(* IEC 61131-3 sources: Explicit_MPC_on_PLC/Quad-Tank/MATLAB_Files/Used Files/plcsrc, 1 file *)

(* ---- sim_mixed.st ---- *)
(*
 *
 * File: sim_mixed.st
 *
 * IEC 61131-3 Structured Text (ST) code generated for subsystem "sim_mixed/Explicit Controller"
 *
 * Model name                      : sim_mixed
 * Model version                   : 1.163
 * Model creator                   : andrewralea
 * Model last modified by          : andrewralea
 * Model last modified on          : Mon May 24 20:24:12 2021
 * Model sample time               : 0s
 * Subsystem name                  : sim_mixed/Explicit Controller
 * Subsystem sample time           : 0.01s
 * Simulink PLC Coder version      : 3.3 (R2020b) 29-Jul-2020
 * ST code generated on            : Fri May 28 16:37:33 2021
 *
 * Target IDE selection            : Beckhoff TwinCAT 3
 * Test Bench included             : No
 *
 *)
FUNCTION_BLOCK Explicit
VAR_INPUT
    ssMethodType: SINT;
    MeasuredTankOutputs: ARRAY [0..1] OF LREAL;
    ref: ARRAY [0..1] OF LREAL;
END_VAR
VAR_OUTPUT
    mv: ARRAY [0..1] OF LREAL;
END_VAR
VAR
    last_x_PreviousInput: ARRAY [0..5] OF LREAL;
    last_mv_DSTATE: ARRAY [0..1] OF LREAL;
    Explicit_b_M: ARRAY [0..11] OF LREAL := 3.14192233852028E-7,2.5115282232541673E-8,5.9723043350726878E-8,
        2.2534269604652875E-7,0.0099501247588661811,3.3026396230579933E-9,6.8756742676357756E-8,
        3.2698899289917904E-7,2.2408008895209797E-7,6.5568434535270065E-8,-3.3744504064209632E-9,
        0.0099501247490762831;
    Explicit_b_Cm: ARRAY [0..11] OF LREAL := 0.15299877600979192,0.0,0.0,0.15299877600979192,0.0,0.0,0.0,0.0,1.0,
        0.0,0.0,1.0;
    Explicit_b_thmin: ARRAY [0..9] OF LREAL := -12.5,-17.5,-3.260954352640991,-0.9466686383552787,-1.25,-1.25,-12.5,
        -17.5,-31.242868949193834,-63.580836957418676;
    Explicit_b_thmax: ARRAY [0..9] OF LREAL := 30.0,25.0,39.239045647359006,41.553331361644723,1.25,1.25,25.0,20.0,
        169.936,169.936;
    b_i1: ARRAY [0..100] OF INT := 1,25,48,71,91,114,137,158,178,199,221,242,262,283,304,324,343,364,383,403,423,
        445,467,485,506,517,537,556,577,597,616,638,656,668,689,708,727,747,767,786,807,827,847,867,886,908,927,947,
        967,989,1008,1019,1039,1055,1076,1098,1117,1136,1155,1171,1189,1211,1230,1246,1265,1284,1299,1318,1339,1357,
        1376,1396,1415,1435,1456,1476,1497,1517,1537,1556,1575,1595,1613,1633,1653,1671,1692,1711,1731,1747,1765,
        1784,1804,1823,1843,1862,1882,1902,1921,1940,1959;
    b_i2: ARRAY [0..100] OF INT := 24,47,70,90,113,136,157,177,198,220,241,261,282,303,323,342,363,382,402,422,444,
        466,484,505,516,536,555,576,596,615,637,655,667,688,707,726,746,766,785,806,826,846,866,885,907,926,946,966,
        988,1007,1018,1038,1054,1075,1097,1116,1135,1154,1170,1188,1210,1229,1245,1264,1283,1298,1317,1338,1356,
        1375,1395,1414,1434,1455,1475,1496,1516,1536,1555,1574,1594,1612,1632,1652,1670,1691,1710,1730,1746,1764,
        1783,1803,1822,1842,1861,1881,1901,1920,1939,1958,1978;
    Explicit_b_L: ARRAY [0..11] OF LREAL := 3.1403362819378811E-7,2.5755371121733541E-8,5.9629108064733625E-8,
        2.246853239956293E-7,0.0099501247588661551,3.3026395811602204E-9,6.9053788137012E-8,3.2695809528341482E-7,
        2.2372764502189584E-7,6.5377157634733646E-8,-3.3744504046873746E-9,0.0099501247490763074;
    Explicit_b_Bu: ARRAY [0..11] OF LREAL := 0.00020814878862012381,1.7089200517136452E-7,0.0,
        0.00011695983573308414,0.0,0.0,9.2113938270845919E-8,0.0002081617439639849,0.00011703862782711392,0.0,0.0,
        0.0;
    Explicit_b_A: ARRAY [0..35] OF LREAL := 0.9991963417969173,0.0,0.0,0.0,0.0,0.0,0.0,0.99932074257543357,0.0,0.0,
        0.0,0.0,0.0015722160273812986,0.0,0.99842715170590557,0.0,0.0,0.0,0.0,0.0029162188726435975,0.0,
        0.99708278976438092,0.0,0.0,0.0,0.0,0.0,0.0,1.0,0.0,0.0,0.0,0.0,0.0,0.0,1.0;
    Explicit_c_K: ARRAY [0..1977] OF LREAL := 150.27277651970425,150.27276024869144,150.1745002542759,
        150.17446124607031,0.0,0.0,0.0,0.0,30.0,25.0,39.239045647359006,41.553331361644723,1.25,1.25,25.0,20.0,12.5,
        17.5,3.260954352640991,0.9466686383552787,1.25,1.25,12.5,17.5,-150.27277651970428,150.27276094028818,
        0.00896851306694222,0.0092486718565456469,150.17446243836258,-6.9159822683988875E-7,-1.1922963395590097E-6,
        30.0,25.0,39.239045647359006,41.553331361644723,1.25,1.25,20.0,169.936,12.5,17.5,3.260954352640991,
        0.9466686383552787,1.25,1.25,12.5,17.5,-150.27276024869144,150.27277721130108,0.0089700423139607143,
        150.17450136627906,0.0092502663373971762,-6.915983020343374E-7,-1.1120067688561992E-6,30.0,25.0,
        39.239045647359006,41.553331361644723,1.25,1.25,25.0,169.936,12.5,17.5,3.260954352640991,0.9466686383552787,
        1.25,1.25,12.5,17.5,-150.1745002542759,150.30349143296371,150.27276061960174,150.25280880838065,
        -6.4025688321438744E-7,30.0,25.0,39.239045647359006,41.553331361644723,1.25,1.25,25.0,12.5,17.5,
        3.260954352640991,0.9466686383552787,1.25,1.25,17.5,63.580836957418676,0.0,150.27276024868996,
        150.17446124606624,0.0,0.0,0.0,0.0,30.0,25.0,39.239045647359006,41.553331361644723,1.25,1.25,25.0,20.0,12.5,
        17.5,3.260954352640991,0.9466686383552787,1.25,1.25,17.5,31.242868949193834,0.0,150.2727765197028,
        150.17450025427226,0.0,0.0,0.0,0.0,30.0,25.0,39.239045647359006,41.553331361644723,1.25,1.25,25.0,20.0,12.5,
        17.5,3.260954352640991,0.9466686383552787,1.25,1.25,12.5,63.580836957418676,0.0,150.27276024869022,
        150.174461246067,0.0,0.0,0.0,30.0,25.0,39.239045647359006,41.553331361644723,1.25,1.25,20.0,12.5,17.5,
        3.260954352640991,0.9466686383552787,1.25,1.25,12.5,17.5,0.0,150.27277651970292,0.0,0.0,0.0,30.0,25.0,
        39.239045647359006,41.553331361644723,1.25,1.25,25.0,12.5,17.5,3.260954352640991,0.9466686383552787,1.25,
        1.25,12.5,17.5,-150.2727772113011,-150.27276094028815,0.00899229717151725,0.0089972026991569677,
        0.0092719269187978466,30.0,25.0,39.239045647359006,41.553331361644723,1.25,1.25,169.936,169.936,12.5,17.5,
        3.260954352640991,0.9466686383552787,1.25,1.25,12.5,17.5,-0.0092486718537731459,-150.3142337225209,
        150.27276094028818,150.17446243836227,-6.91598518490273E-7,-1.1922968442958055E-6,30.0,25.0,
        39.239045647359006,41.553331361644723,1.25,1.25,25.0,20.0,169.936,12.5,17.5,3.260954352640991,
        0.9466686383552787,1.25,1.25,17.5,-150.2727765197028,12.5,-150.31423372345185,6.915984886602121E-7,
        0.010088924529484842,-2.7160393645102115E-5,30.0,25.0,39.239045647359006,41.553331361644723,1.25,1.25,20.0,
        169.936,12.5,17.5,3.260954352640991,0.9466686383552787,1.25,1.25,63.580836957418676,-150.27277651970294,
        1.192296339559001E-6,0.0089685130647667952,0.0092486718548978036,-7.9526503793109085E-7,30.0,25.0,
        39.239045647359006,41.553331361644723,1.25,1.25,169.936,12.5,17.5,3.260954352640991,0.9466686383552787,1.25,
        1.25,12.5,17.5,-150.31422855929941,-0.0089700423151911571,150.27277721130105,150.17450136627863,
        0.010090749420623041,-6.91598601136511E-7,-1.1120072501316056E-6,30.0,25.0,39.239045647359006,
        41.553331361644723,1.25,1.25,25.0,169.936,12.5,17.5,3.260954352640991,1.25,1.25,12.5,-150.27276024868993,
        -2.3784105123531843E-5,17.5,-150.314228558367,6.9159864144958721E-7,30.0,25.0,39.239045647359006,
        41.553331361644723,1.25,1.25,25.0,20.0,169.936,12.5,17.5,3.260954352640991,0.9466686383552787,1.25,1.25,
        31.242868949193834,-150.27276024869022,1.112006768856199E-6,0.0089700423159589249,0.0092502663388704057,
        -8.1826648506024674E-7,30.0,25.0,39.239045647359006,41.553331361644723,1.25,1.25,169.936,12.5,17.5,
        3.260954352640991,0.9466686383552787,1.25,1.25,12.5,17.5,-0.0084253602440059385,-0.0084317458919612974,
        150.31423400479244,150.31422879473305,30.0,25.0,39.239045647359006,41.553331361644723,1.25,1.25,25.0,20.0,
        17.5,3.260954352640991,0.9466686383552787,1.25,1.25,31.242868949193834,63.580836957418676,0.0,0.0,0.0,0.0,
        0.0,30.0,25.0,39.239045647359006,41.553331361644723,1.25,1.25,25.0,20.0,12.5,17.5,3.260954352640991,
        0.9466686383552787,1.25,1.25,31.242868949193834,63.580836957418676,0.0,0.0,150.27276024868965,0.0,30.0,25.0,
        39.239045647359006,41.553331361644723,1.25,1.25,12.5,17.5,3.260954352640991,0.9466686383552787,1.25,1.25,
        17.5,31.242868949193834,63.580836957418676,0.0,0.0,0.0,0.0,0.0,30.0,25.0,39.239045647359006,
        41.553331361644723,1.25,1.25,25.0,12.5,17.5,3.260954352640991,0.9466686383552787,1.25,1.25,17.5,
        31.242868949193834,0.0,17.5,0.0,0.0,0.0,30.0,25.0,39.239045647359006,41.553331361644723,1.25,1.25,20.0,12.5,
        17.5,3.260954352640991,0.9466686383552787,1.25,1.25,12.5,63.580836957418676,0.0,150.27277651970246,
        150.17450025427149,0.0,0.0,0.0,30.0,25.0,39.239045647359006,41.553331361644723,1.25,1.25,25.0,20.0,12.5,
        17.5,3.260954352640991,0.9466686383552787,1.25,1.25,12.5,63.580836957418676,0.0,150.27276024868988,
        150.17446124606604,0.0,0.0,0.0,30.0,25.0,39.239045647359006,41.553331361644723,1.25,1.25,20.0,169.936,12.5,
        17.5,3.260954352640991,0.9466686383552787,1.25,1.25,12.5,17.5,0.0,0.0,0.0,0.0,30.0,25.0,39.239045647359006,
        41.553331361644723,1.25,1.25,12.5,17.5,3.260954352640991,0.9466686383552787,1.25,1.25,12.5,17.5,0.0,
        150.2727765197026,150.17450025427178,0.0,0.0,0.0,30.0,25.0,39.239045647359006,41.553331361644723,1.25,1.25,
        25.0,12.5,17.5,3.260954352640991,0.9466686383552787,1.25,1.25,12.5,17.5,-150.31423409213582,
        -150.27276094028815,-0.0089922971720828356,0.0089972027095938083,0.0101105928744509,30.0,25.0,
        39.239045647359006,41.553331361644723,1.25,1.25,-0.008997202709492582,-150.27277721130102,
        -150.31422888114486,0.0089922971840448781,30.0,25.0,39.239045647359006,41.553331361644723,1.25,1.25,20.0,
        169.936,169.936,12.5,17.5,3.260954352640991,0.9466686383552787,1.25,1.25,12.5,-0.0092486718560890989,
        -150.3142337225205,1.1922968442958055E-6,-7.9526537103502364E-7,30.0,25.0,39.239045647359006,
        41.553331361644723,1.25,1.25,25.0,169.936,12.5,17.5,3.260954352640991,0.9466686383552787,1.25,1.25,17.5,
        -150.27277651970238,3.2277787241348325E-7,2.6103247877849398E-5,0.0089685130647338546,0.00924867185486637,
        30.0,25.0,39.239045647359006,41.553331361644723,1.25,1.25,169.936,12.5,17.5,3.260954352640991,
        0.9466686383552787,1.25,1.25,12.5,17.5,63.580836957418676,-150.2727765197026,7.9526503793110049E-7,
        0.0089685130647458953,0.0092486718548779323,-3.2277787241348331E-7,30.0,25.0,39.239045647359006,
        41.553331361644723,1.25,1.25,169.936,12.5,17.5,3.260954352640991,0.9466686383552787,1.25,1.25,12.5,17.5,
        -150.20363326125491,150.27277704995686,150.31422855929944,150.17450110707583,0.0084101003282759639,
        -5.3025423494204181E-7,-8.5280395478764181E-7,30.0,25.0,39.239045647359006,41.553331361644723,1.25,1.25,
        25.0,1.25,1.25,12.5,17.5,31.242868949193834,-150.3142285583674,-4.5713461310450266E-7,150.272777211301,
        150.17450136627863,-6.9159864144958721E-7,-1.1120073155610654E-6,30.0,25.0,39.239045647359006,
        41.553331361644723,1.25,1.25,25.0,20.0,169.936,12.5,17.5,3.260954352640991,0.9466686383552787,1.25,1.25,
        12.5,-150.3142285592991,-0.0089700423152055762,1.1120072501316007E-6,0.010090749420522883,
        -8.182668401829975E-7,30.0,25.0,39.239045647359006,41.553331361644723,1.25,1.25,169.936,12.5,17.5,
        3.260954352640991,1.25,1.25,12.5,-150.27276024868971,4.8112884150133535E-7,2.3255062955056014E-5,
        0.0089700423159182838,-2.4842396974108378E-5,25.0,39.239045647359006,41.553331361644723,1.25,1.25,17.5,
        31.242868949193834,-150.27276024868988,2.1668353413129541E-5,0.0089700423138394814,0.00925026633727334,
        -3.6868395525815943E-7,30.0,25.0,39.239045647359006,41.553331361644723,1.25,1.25,169.936,169.936,12.5,17.5,
        3.260954352640991,0.9466686383552787,1.25,1.25,12.5,17.5,-150.20366731447805,-0.0084317458833884553,
        150.31423400572388,150.31422879473305,0.0084253602346650771,30.0,25.0,39.239045647359006,41.553331361644723,
        1.25,1.25,20.0,12.5,17.5,3.260954352640991,0.9466686383552787,1.25,1.25,63.580836957418676,
        -150.20363403920774,-0.0084253602429266682,150.31423400479244,150.31422879566506,0.0084317458959346555,30.0,
        25.0,39.239045647359006,41.553331361644723,1.25,1.25,25.0,12.5,17.5,3.260954352640991,0.9466686383552787,
        1.25,1.25,31.242868949193834,-150.31423400479247,-4.57772250744983E-7,-3.8232338890894953E-7,
        150.31422888114494,30.0,25.0,39.239045647359006,41.553331361644723,1.25,1.25,25.0,20.0,169.936,17.5,
        3.260954352640991,0.9466686383552787,1.25,1.25,31.242868949193834,63.580836957418676,0.0,0.0,0.0,0.0,0.0,
        30.0,25.0,39.239045647359006,41.553331361644723,1.25,1.25,20.0,12.5,17.5,3.260954352640991,
        0.9466686383552787,1.25,1.25,31.242868949193834,63.580836957418676,0.0,0.0,0.0,0.0,0.0,30.0,25.0,
        39.239045647359006,41.553331361644723,1.25,1.25,25.0,12.5,17.5,3.260954352640991,1.25,1.25,
        31.242868949193834,63.580836957418676,0.0,150.27276024868991,0.0,0.0,0.0,30.0,25.0,39.239045647359006,
        41.553331361644723,1.25,1.25,25.0,20.0,12.5,17.5,3.260954352640991,0.9466686383552787,1.25,1.25,17.5,
        31.242868949193834,0.0,17.5,0.0,0.0,30.0,25.0,39.239045647359006,41.553331361644723,1.25,1.25,20.0,12.5,
        17.5,3.260954352640991,0.9466686383552787,1.25,1.25,12.5,31.242868949193834,63.580836957418676,0.0,0.0,0.0,
        0.0,0.0,30.0,25.0,39.239045647359006,41.553331361644723,1.25,1.25,25.0,12.5,17.5,3.260954352640991,
        0.9466686383552787,1.25,1.25,17.5,31.242868949193834,0.0,0.0,0.0,0.0,0.0,30.0,25.0,39.239045647359006,
        41.553331361644723,1.25,1.25,25.0,12.5,17.5,3.260954352640991,0.9466686383552787,1.25,1.25,17.5,
        31.242868949193834,0.0,0.0,0.0,0.0,30.0,25.0,39.239045647359006,41.553331361644723,1.25,1.25,169.936,12.5,
        17.5,3.260954352640991,0.9466686383552787,1.25,1.25,12.5,17.5,0.0,0.0,150.27277651970238,150.17450025427129,
        0.0,0.0,30.0,25.0,39.239045647359006,41.553331361644723,1.25,1.25,25.0,12.5,17.5,3.260954352640991,
        0.9466686383552787,1.25,1.25,12.5,17.5,63.580836957418676,0.0,0.0,0.0,0.0,30.0,25.0,39.239045647359006,
        41.553331361644723,1.25,1.25,20.0,12.5,17.5,3.260954352640991,0.9466686383552787,1.25,1.25,12.5,
        63.580836957418676,0.0,0.0,0.0,0.0,30.0,25.0,39.239045647359006,41.553331361644723,1.25,1.25,169.936,12.5,
        17.5,3.260954352640991,0.9466686383552787,1.25,1.25,12.5,17.5,63.580836957418676,0.0,0.0,0.0,0.0,30.0,25.0,
        39.239045647359006,41.553331361644723,1.25,1.25,20.0,169.936,12.5,17.5,3.260954352640991,0.9466686383552787,
        1.25,1.25,12.5,63.580836957418676,0.0,0.0,150.27276024868965,150.17446124606542,0.0,0.0,30.0,25.0,
        39.239045647359006,41.553331361644723,1.25,1.25,20.0,12.5,17.5,3.260954352640991,0.9466686383552787,1.25,
        1.25,12.5,17.5,31.242868949193834,-150.17450025427178,4.253152391505125E-7,150.30349143296283,
        150.25280880837818,-1.7296307093690735E-7,30.0,25.0,39.239045647359006,41.553331361644723,1.25,1.25,25.0,
        12.5,17.5,3.260954352640991,0.9466686383552787,1.25,1.25,17.5,-150.27276075599735,-150.20366755066993,
        150.31423409213579,0.0089899947598349236,0.00843045541435082,30.0,25.0,39.239045647359006,
        41.553331361644723,1.25,1.25,-150.27276094028815,17.5,-150.31423409120444,-150.31422888114497,30.0,25.0,
        39.239045647359006,41.553331361644723,1.25,1.25,25.0,20.0,169.936,169.936,17.5,3.260954352640991,
        0.9466686383552787,1.25,1.25,31.242868949193834,-150.27277704995686,-150.20363432127169,150.31422888207695,
        0.00898677805621705,0.0084393742662072935,30.0,25.0,39.239045647359006,41.553331361644723,1.25,1.25,169.936,
        1.25,1.25,12.5,17.5,-150.25280880838059,150.31423372252087,150.27276075599735,150.17446212183043,
        -5.0730746847704375E-7,-8.7576436608860627E-7,30.0,25.0,39.239045647359006,41.553331361644723,1.25,1.25,
        25.0,20.0,12.5,17.5,3.260954352640991,0.9466686383552787,1.25,1.25,17.5,-150.31423372252044,
        -4.57021496831135E-7,6.91598518490273E-7,-2.7160394808446411E-5,-2.7688874260814198E-5,30.0,25.0,
        39.239045647359006,41.553331361644723,1.25,1.25,25.0,20.0,169.936,17.5,3.260954352640991,0.9466686383552787,
        1.25,1.25,17.5,31.242868949193834,63.580836957418676,-150.1745002542726,6.4025688321438437E-7,
        150.303491432963,150.25280880837869,-4.2531523915050832E-7,30.0,25.0,39.239045647359006,41.553331361644723,
        1.25,1.25,25.0,12.5,17.5,3.260954352640991,0.9466686383552787,1.25,1.25,17.5,-150.30349143296283,
        -0.0092486718560926464,7.9526530580585218E-7,0.0084080843735949169,-3.2277798170283768E-7,30.0,25.0,
        39.239045647359006,41.553331361644723,1.25,1.25,169.936,12.5,17.5,3.260954352640991,0.9466686383552787,1.25,
        1.25,17.5,-150.20366653652189,5.0730744361467508E-7,150.31423372345185,0.00840878705982342,
        -1.9952445451383883E-5,30.0,25.0,39.239045647359006,41.553331361644723,1.25,1.25,20.0,12.5,17.5,
        3.260954352640991,0.9466686383552787,1.25,1.25,63.580836957418676,-150.27277651970246,4.4094945298300684E-7,
        2.7688862477194338E-5,0.0089685130647387656,-2.6103247877849368E-5,30.0,25.0,39.239045647359006,
        41.553331361644723,1.25,1.25,1.25,1.25,12.5,17.5,63.580836957418676,-150.3142337225203,
        3.2277800799099981E-7,30.0,25.0,39.239045647359006,41.553331361644723,1.25,1.25,25.0,169.936,12.5,17.5,
        3.260954352640991,0.9466686383552787,1.25,1.25,17.5,63.580836957418676,-0.0084101003242163189,
        150.27277704995686,150.31422855836743,150.17450110707577,-5.3025426854081661E-7,-8.528040093195823E-7,30.0,
        25.0,39.239045647359006,41.553331361644723,1.25,1.25,25.0,20.0,12.5,17.5,3.260954352640991,
        0.9466686383552787,1.25,1.25,12.5,63.580836957418676,-150.20363326125155,5.302542349420417E-7,
        150.31422855929904,0.0084101003218975314,-1.78419540761567E-5,30.0,25.0,39.239045647359006,
        41.553331361644723,1.25,1.25,25.0,12.5,17.5,3.260954352640991,0.9466686383552787,1.25,1.25,
        31.242868949193834,-150.2036332612509,2.8227211141446421E-7,1.9111227183265134E-5,150.31422855929898,
        0.0084101003281506683,30.0,25.0,39.239045647359006,41.553331361644723,1.25,1.25,1.25,1.25,12.5,17.5,
        31.242868949193834,-150.31422855836709,-4.5713461315188076E-7,3.7104855832596717E-9,-8.1826688808031187E-7,
        30.0,25.0,39.239045647359006,41.553331361644723,1.25,1.25,20.0,169.936,12.5,17.5,3.260954352640991,
        0.9466686383552787,1.25,1.25,12.5,-150.31422855929895,-0.0089700423152052188,4.81129049402035E-7,
        2.3255073031969076E-5,0.010090749420478901,-2.4842407822217915E-5,25.0,39.239045647359006,
        41.553331361644723,1.25,1.25,169.936,12.5,17.5,3.260954352640991,0.9466686383552787,1.25,1.25,
        31.242868949193834,-150.20363326125218,8.5280395478765081E-7,150.31422855929912,0.008410100321918695,
        -6.2813598573044263E-7,30.0,25.0,39.239045647359006,41.553331361644723,1.25,1.25,1.25,1.25,12.5,17.5,
        -150.31422855929904,-0.0089700423159724645,2.1668362719146114E-5,0.010090749414219103,
        -3.6868411405625081E-7,30.0,25.0,39.239045647359006,41.553331361644723,1.25,1.25,169.936,169.936,12.5,17.5,
        3.260954352640991,1.25,1.25,12.5,-150.27276024868965,3.6868395525815943E-7,2.2497959692190342E-9,
        0.008970042313820821,0.00925026633725427,30.0,25.0,39.239045647359006,41.553331361644723,1.25,1.25,169.936,
        12.5,17.5,3.260954352640991,0.9466686383552787,1.25,1.25,12.5,17.5,31.242868949193834,-150.20366731447808,
        -150.20363403920777,150.31423400572388,150.31422879566503,0.0084253602409406526,0.0084317458833884553,30.0,
        25.0,39.239045647359006,41.553331361644723,1.25,1.25,12.5,17.5,3.260954352640991,0.9466686383552787,1.25,
        1.25,-150.314228794733,-150.20366755066965,-0.01011239497184554,150.31423409213585,0.008430455426884231,
        30.0,25.0,39.239045647359006,41.553331361644723,1.25,1.25,20.0,169.936,12.5,17.5,3.260954352640991,
        0.9466686383552787,1.25,1.25,-0.0084087870624481986,5.0730746847704364E-7,150.31423372252041,
        -1.9952446420993245E-5,-2.0375796427188149E-5,30.0,25.0,39.239045647359006,41.553331361644723,1.25,1.25,
        25.0,20.0,17.5,3.260954352640991,0.9466686383552787,1.25,1.25,31.242868949193834,63.580836957418676,
        -150.3142340047925,-150.20363432127149,-0.010105497708264473,150.31422888207695,0.008439374278734136,30.0,
        25.0,39.239045647359006,41.553331361644723,1.25,1.25,25.0,169.936,17.5,3.260954352640991,0.9466686383552787,
        1.25,1.25,31.242868949193834,-0.0084101003242149728,5.3025426854081651E-7,150.31422855836706,
        -1.7841955234048227E-5,30.0,25.0,39.239045647359006,41.553331361644723,1.25,1.25,25.0,20.0,12.5,17.5,
        3.260954352640991,0.9466686383552787,1.25,1.25,31.242868949193834,63.580836957418676,-150.31423400572393,
        0.010105497701810977,-150.27277704995686,-0.0084393742662072935,150.31422888114494,30.0,25.0,
        39.239045647359006,41.553331361644723,1.25,1.25,20.0,169.936,12.5,17.5,3.260954352640991,0.9466686383552787,
        1.25,1.25,12.5,63.580836957418676,4.8112907714119855E-7,25.0,-150.31422855836695,3.6868413507214106E-7,30.0,
        25.0,39.239045647359006,41.553331361644723,1.25,1.25,20.0,169.936,12.5,17.5,3.260954352640991,
        0.9466686383552787,1.25,1.25,12.5,31.242868949193834,0.0,0.0,0.0,0.0,0.0,30.0,25.0,39.239045647359006,
        41.553331361644723,1.25,1.25,25.0,12.5,17.5,3.260954352640991,0.9466686383552787,1.25,1.25,17.5,
        31.242868949193834,63.580836957418676,0.0,0.0,0.0,0.0,30.0,25.0,39.239045647359006,41.553331361644723,1.25,
        1.25,169.936,12.5,17.5,3.260954352640991,0.9466686383552787,1.25,1.25,12.5,17.5,31.242868949193834,0.0,0.0,
        0.0,0.0,0.0,30.0,25.0,39.239045647359006,41.553331361644723,1.25,1.25,25.0,12.5,17.5,3.260954352640991,
        0.9466686383552787,1.25,1.25,31.242868949193834,63.580836957418676,0.0,0.0,0.0,30.0,25.0,39.239045647359006,
        41.553331361644723,1.25,1.25,25.0,12.5,17.5,3.260954352640991,0.9466686383552787,1.25,1.25,12.5,17.5,
        31.242868949193834,-0.50109411185443054,1.7296307093690733E-7,150.30349143296272,150.25280880837795,30.0,
        25.0,39.239045647359006,41.553331361644723,1.25,1.25,25.0,12.5,17.5,3.260954352640991,0.9466686383552787,
        1.25,1.25,17.5,63.580836957418676,0.0,0.0,0.0,0.0,30.0,25.0,39.239045647359006,41.553331361644723,1.25,1.25,
        169.936,169.936,12.5,17.5,3.260954352640991,0.9466686383552787,1.25,1.25,12.5,17.5,-150.25280880837818,
        5.8219085145699086E-7,150.31423372252033,-2.3636600485157802E-7,30.0,25.0,39.239045647359006,
        41.553331361644723,1.25,1.25,25.0,12.5,17.5,3.260954352640991,0.9466686383552787,1.25,1.25,17.5,
        -150.27276075599735,-0.00843045541720925,150.31423409120438,0.00898999476192504,30.0,25.0,
        39.239045647359006,41.553331361644723,1.25,1.25,25.0,169.936,12.5,17.5,3.260954352640991,0.9466686383552787,
        1.25,1.25,17.5,31.242868949193834,-150.31423409213585,-150.31422888114491,-1.2217120684816844E-6,
        -4.5846079178133877E-7,4.5800301307963309E-5,30.0,25.0,39.239045647359006,41.553331361644723,1.25,1.25,20.0,
        169.936,169.936,12.5,17.5,3.260954352640991,0.9466686383552787,1.25,1.25,-150.25280880837866,
        8.7576436608860257E-7,150.31423372252044,-5.82190851456982E-7,30.0,25.0,39.239045647359006,
        41.553331361644723,1.25,1.25,25.0,12.5,17.5,3.260954352640991,0.9466686383552787,1.25,1.25,17.5,
        -150.31423372252033,-4.5702149683232403E-7,4.4094963796295432E-7,-1.1821419161471384E-7,30.0,25.0,
        39.239045647359006,41.553331361644723,1.25,1.25,25.0,20.0,169.936,17.5,3.260954352640991,0.9466686383552787,
        1.25,1.25,17.5,31.242868949193834,63.580836957418676,-150.31423372252036,-7.6145930516505814E-7,
        3.9783223815065124E-9,-3.2277800799099981E-7,30.0,25.0,39.239045647359006,41.553331361644723,1.25,1.25,25.0,
        169.936,12.5,17.5,3.260954352640991,0.9466686383552787,1.25,1.25,17.5,-150.31423372345176,
        -0.0089685130660916157,4.4094961895705287E-7,0.010088924529470659,-2.6103257691860455E-5,30.0,25.0,
        39.239045647359006,41.553331361644723,1.25,1.25,20.0,169.936,12.5,17.5,3.260954352640991,0.9466686383552787,
        1.25,1.25,63.580836957418676,-150.20363326125141,1.657318047106699E-5,150.31422855929904,
        0.0084101003281674778,-2.8227211141446421E-7,30.0,25.0,39.239045647359006,41.553331361644723,1.25,1.25,
        169.936,1.25,1.25,12.5,17.5,-150.20363326125104,3.6877592925547954E-7,1.7841954076156706E-5,
        150.31422855929898,0.0084101003218820559,-1.9111227183265138E-5,25.0,39.239045647359006,41.553331361644723,
        1.25,1.25,12.5,17.5,3.260954352640991,0.9466686383552787,1.25,1.25,31.242868949193834,-150.31422855929895,
        -1.2188190344585731E-6,3.6868411405625075E-7,2.2497969516602169E-9,4.5713456671592212E-5,30.0,25.0,
        39.239045647359006,41.553331361644723,1.25,1.25,169.936,12.5,17.5,3.260954352640991,1.25,1.25,12.5,
        31.242868949193834,-3.8099721031245746E-7,2.8227212893007557E-7,1.7307655422208259E-9,150.31422855836695,
        30.0,25.0,39.239045647359006,41.553331361644723,1.25,1.25,20.0,12.5,17.5,3.260954352640991,
        0.9466686383552787,1.25,1.25,12.5,31.242868949193834,63.580836957418676,-0.0084101003298609166,
        8.5280400931958431E-7,150.31422855836712,-6.2813602565029217E-7,30.0,25.0,39.239045647359006,
        41.553331361644723,1.25,1.25,20.0,12.5,17.5,3.260954352640991,0.9466686383552787,1.25,1.25,12.5,
        63.580836957418676,-150.314228558367,-4.5713461315331108E-7,9.8156217007103415E-10,-3.6868413507214106E-7,
        30.0,25.0,39.239045647359006,41.553331361644723,1.25,1.25,20.0,169.936,169.936,12.5,17.5,3.260954352640991,
        0.9466686383552787,1.25,1.25,12.5,-150.314228794733,-3.8189390365081248E-7,-4.5811520781545546E-7,
        150.31423409120436,30.0,25.0,39.239045647359006,41.553331361644723,1.25,1.25,25.0,20.0,169.936,17.5,
        3.260954352640991,0.9466686383552787,1.25,1.25,31.242868949193834,-0.00840878706245568,3.22858662019215E-7,
        150.3142337225203,-1.9105604561403706E-5,30.0,25.0,39.239045647359006,41.553331361644723,1.25,1.25,25.0,
        20.0,17.5,3.260954352640991,0.9466686383552787,1.25,1.25,17.5,31.242868949193834,63.580836957418676,
        -0.00841010032985721,3.6877595237458659E-7,150.31422855836698,-1.9111228421220846E-5,30.0,25.0,
        39.239045647359006,41.553331361644723,1.25,1.25,25.0,20.0,12.5,17.5,3.260954352640991,0.9466686383552787,
        1.25,1.25,31.242868949193834,63.580836957418676,-0.75164095173259382,2.3636600485157802E-7,
        1.7304765244832798E-9,150.31423372252024,30.0,25.0,39.239045647359006,41.553331361644723,1.25,1.25,25.0,
        12.5,17.5,3.260954352640991,0.9466686383552787,1.25,1.25,17.5,63.580836957418676,-150.31422879566506,
        -0.00898999476239346,-0.0084304554265223746,150.31423409120438,0.010112394966153392,30.0,25.0,
        39.239045647359006,41.553331361644723,1.25,1.25,25.0,169.936,17.5,3.260954352640991,0.9466686383552787,1.25,
        1.25,31.242868949193834,-150.20366653652124,3.2285864617841143E-7,150.31423372345174,0.0084087870598116,
        -1.910560364578063E-5,30.0,25.0,39.239045647359006,41.553331361644723,1.25,1.25,20.0,12.5,17.5,
        3.260954352640991,0.9466686383552787,1.25,1.25,63.580836957418676,-0.0084101003298601585,
        1.657318154892557E-5,150.31422855836703,-2.8227212893007557E-7,30.0,25.0,39.239045647359006,
        41.553331361644723,1.25,1.25,20.0,169.936,12.5,17.5,3.260954352640991,0.9466686383552787,1.25,1.25,12.5,
        63.580836957418676;
    Explicit_g_H: ARRAY [0..19779] OF LREAL := -0.0029153681735618136,-3.0076549641322347E-6,-0.00485576775256503,
        -4.294484498891456E-6,0.0029153681735618136,3.0076549641322347E-6,0.00485576775256503,4.2944844988914552E-6,
        1.0,0.0,0.0,0.0,0.0,0.0,0.0,0.0,-1.0,-0.0,-0.0,-0.0,-0.0,-0.0,-0.0,-0.0,0.002915368173561814,
        -3.0076683814890018E-6,-0.10733105865380493,-0.10732396454285037,-4.29450763004578E-6,3.0076683814890018E-6,
        4.2945076300457788E-6,1.0,0.0,0.0,0.0,0.0,0.0,0.0,0.0,-1.0,-0.0,-0.0,-0.0,-0.0,-0.0,-0.0,-0.0,
        3.0076549641322347E-6,-0.0029153681735756267,-7.9117024960378933E-5,-0.0048557677525871683,
        -7.1206870222596425E-5,0.0029153681735756267,0.0048557677525871683,1.0,0.0,0.0,0.0,0.0,0.0,0.0,0.0,-1.0,
        -0.0,-0.0,-0.0,-0.0,-0.0,-0.0,-0.0,0.0048557677525650289,-0.0019439782274928883,-3.0076669572476592E-6,
        -0.0034008125243717886,4.2945052010659752E-6,1.0,0.0,0.0,0.0,0.0,0.0,0.0,-1.0,-0.0,-0.0,-0.0,-0.0,-0.0,-0.0,
        -0.0,-0.002915368173561814,-3.0076683814890018E-6,-4.29450763004578E-6,3.0076683814890018E-6,
        0.10733105865380499,0.10732396454285044,4.2945076300457788E-6,1.0,0.0,0.0,0.0,0.0,0.0,0.0,0.0,-1.0,-0.0,
        -0.0,-0.0,-0.0,-0.0,-0.0,-0.0,-3.0076549641322347E-6,-0.0029153681735756267,-0.0048557677525871683,
        0.0029153681735756267,7.9117024960378879E-5,0.0048557677525871683,7.1206870222596425E-5,1.0,0.0,0.0,0.0,0.0,
        0.0,0.0,0.0,-1.0,-0.0,-0.0,-0.0,-0.0,-0.0,-0.0,-0.0,-0.0048557677525650289,-3.0076669572476592E-6,
        -4.2945052010659761E-6,3.0076669572476592E-6,0.0034008125243717912,4.2945052010659752E-6,1.0,0.0,0.0,0.0,
        0.0,0.0,0.0,-1.0,-0.0,-0.0,-0.0,-0.0,-0.0,-0.0,-0.0,-4.294484498891456E-6,-0.0029153681735731604,
        0.0043710401679979711,3.6517411636309943E-6,0.0048557677525832323,1.0,0.0,0.0,0.0,0.0,0.0,0.0,-1.0,-0.0,
        -0.0,-0.0,-0.0,-0.0,-0.0,-0.0,0.0029153681735756276,3.0076683814890018E-6,-0.10733105865317544,
        -7.9117551884579521E-5,-0.10732396454229656,1.0,0.0,0.0,0.0,0.0,0.0,0.0,0.0,-1.0,-0.0,-0.0,-0.0,-0.0,-0.0,
        -0.0,-0.0,0.10732396454285041,0.0014580885500697777,-3.0076718320980626E-6,-4.2945136019776164E-6,
        3.0076718320980626E-6,4.2945136019776156E-6,1.0,0.0,0.0,0.0,0.0,0.0,0.0,0.0,0.0,-1.0,-0.0,-0.0,-0.0,-0.0,
        -0.0,-0.0,0.0029153681735756276,-0.0,0.0014580885008721898,-3.0076715148347656E-6,-0.10730267567315248,
        7.9117675509431345E-5,1.0,0.0,0.0,0.0,0.0,0.0,0.0,0.0,-1.0,-0.0,-0.0,-0.0,-0.0,-0.0,-0.0,
        0.0029153681735731608,-4.2945076300457788E-6,-0.10733105865319877,-0.10732396454231756,
        3.6517565921765204E-6,1.0,0.0,0.0,0.0,0.0,0.0,0.0,-1.0,-0.0,-0.0,-0.0,-0.0,-0.0,-0.0,-0.0,
        1.9335719862715687E-6,7.911702496037896E-5,-0.0029153681735782583,-0.0048557677525913855,
        -4.7481728551617291E-5,0.0029153681735782583,0.0048557677525913855,1.0,0.0,0.0,0.0,0.0,0.0,0.0,0.0,-1.0,
        -0.0,-0.0,-0.0,-0.0,-0.0,3.0076683814890014E-6,0.10733105865317549,-0.0,1.93357827010103E-6,
        -0.0029153681735784474,1.0,0.0,0.0,0.0,0.0,0.0,0.0,0.0,0.0,-1.0,-0.0,-0.0,-0.0,-0.0,-0.0,-0.0,
        3.0076669572476588E-6,-0.0048557677525871675,-7.911749629991159E-5,-7.1207351835982E-5,
        0.0034008125243881219,1.0,0.0,0.0,0.0,0.0,0.0,0.0,-1.0,-0.0,-0.0,-0.0,-0.0,-0.0,-0.0,-0.0,
        0.10730267565345167,4.7482357791108478E-5,-0.00145808855007754,-1.9335790357216359E-6,1.0,0.0,0.0,0.0,0.0,
        0.0,0.0,0.0,-0.0,-0.0,-0.0,-0.0,-0.0,-0.0,-0.0,-0.0029153681735756276,-3.0076683814890018E-6,
        7.9117551884579453E-5,0.10732396454229663,7.1207407399672182E-5,1.0,0.0,0.0,0.0,0.0,0.0,0.0,0.0,-1.0,-0.0,
        -0.0,-0.0,-0.0,-0.0,-0.0,-0.0,-0.0014580885008648144,-0.10733105865380498,-3.0076715148347656E-6,
        0.10730267567349637,1.0,0.0,0.0,0.0,0.0,0.0,-1.0,-0.0,-0.0,-0.0,-0.0,-0.0,-0.0,-0.0,-0.0,
        -0.0029153681735731608,-4.2945076300457788E-6,0.10733105865319882,3.6517565921765204E-6,0.10732396454231762,
        1.0,0.0,0.0,0.0,0.0,0.0,0.0,-1.0,-0.0,-0.0,-0.0,-0.0,-0.0,-0.0,-0.0,-1.93357760066366E-6,-0.0,
        -3.0076669572476588E-6,-0.0048557677525871675,0.0034008125243881219,1.0,0.0,0.0,0.0,0.0,0.0,0.0,-1.0,-0.0,
        -0.0,-0.0,-0.0,-0.0,-0.0,-0.0,-2.3633187068778728E-6,-0.0029153681735777726,-0.0048557677525906144,
        0.0029153681735777726,9.4939976476330723E-5,0.0048557677525906144,1.0,0.0,0.0,0.0,0.0,0.0,0.0,0.0,-1.0,-0.0,
        -0.0,-0.0,-0.0,-0.0,-0.0,-0.0,-0.10730267565385768,-3.007670044425248E-6,-4.2945105315273461E-6,
        0.001458088550069777,3.007670044425248E-6,4.2945105315273452E-6,1.0,0.0,0.0,0.0,0.0,0.0,0.0,0.0,-1.0,-0.0,
        -0.0,-0.0,-0.0,-0.0,-0.0,-0.0,-0.0048557677525832323,-4.2945052010659752E-6,0.0034008125243852232,
        3.6517549158460084E-6,1.0,0.0,0.0,0.0,0.0,0.0,-1.0,-0.0,-0.0,-0.0,-0.0,-0.0,-0.0,-0.0,
        -3.6517411636309939E-6,-0.0029153681735763757,-0.0048557677525883705,0.0029153681735763757,
        1.9335720080464048E-6,0.0048557677525883705,1.0,0.0,0.0,0.0,0.0,0.0,0.0,-1.0,-0.0,-0.0,-0.0,-0.0,-0.0,-0.0,
        -0.0,0.0014580885008721898,3.0076715148347656E-6,0.10733105865317542,-7.911767550943144E-5,
        -0.10730267567315266,1.0,0.0,0.0,0.0,0.0,0.0,7.9117675509431413E-5,0.0029153681735784474,
        1.9335782701010309E-6,-0.10733105865298566,1.0,0.0,0.0,0.0,0.0,0.0,0.0,0.0,0.0,-1.0,-0.0,-0.0,-0.0,-0.0,
        -0.0,-0.0,0.10732396454231755,0.0014580885500758141,-4.2945136019776147E-6,3.6517605334388514E-6,1.0,0.0,
        0.0,0.0,0.0,0.0,0.0,0.0,-1.0,-0.0,-0.0,-0.0,-0.0,-0.0,-0.0,0.0029153681735784474,-1.9335782701010317E-6,
        -9.4940482891343363E-5,-0.10733105865298566,-0.10732396454212995,1.0,0.0,0.0,0.0,0.0,0.0,0.0,-1.0,-0.0,-0.0,
        -0.0,-0.0,-0.0,-0.0,-0.0,-0.0,0.0029153681735763757,-3.6517565921765191E-6,-0.10733105865305877,
        -0.10732396454219448,1.9335782701010321E-6,1.0,0.0,0.0,0.0,0.0,0.0,0.0,-1.0,-0.0,-0.0,-0.0,-0.0,-0.0,-0.0,
        -0.0,4.0803944641294937E-6,-0.0029153681735761866,-1.9335719862715696E-6,-0.0048557677525880661,
        -4.7481714139195562E-5,0.0029153681735761866,0.0048557677525880661,1.0,0.0,0.0,0.0,0.0,0.0,0.0,-0.0,-0.0,
        -0.0,-0.0,-0.0,1.9335720080464023E-6,2.1510336565440439E-9,-0.0029153681735784465,-0.0048557677525916908,
        0.0029153681735784465,0.0048557677525916908,1.0,0.0,0.0,0.0,0.0,0.0,0.0,0.0,0.0,-1.0,-0.0,-0.0,-0.0,-0.0,
        -0.0,-0.0,1.9335775788885903E-6,7.9117496299911522E-5,-0.0048557677525913837,-4.7482240979621922E-5,
        0.003400812524391244,1.0,0.0,0.0,0.0,0.0,0.0,0.0,-1.0,-0.0,-0.0,-0.0,-0.0,-0.0,3.0076711049122026E-6,
        -0.0019439782275025074,-0.10732396454229662,-7.9117659047139367E-5,0.10734524358329479,0.0,0.0,0.0,0.0,0.0,
        -0.0,-0.0,3.0076700444252484E-6,-0.10730267565351387,-7.9117617963562125E-5,-7.1207475890096032E-5,
        0.0014580885500771522,1.0,0.0,0.0,0.0,0.0,0.0,0.0,0.0,-1.0,-0.0,-0.0,-0.0,-0.0,-0.0,-0.0,-0.0,
        0.0043710401680026635,4.7482344040746464E-5,-0.0014580885008725773,-1.9335788864753624E-6,
        -0.10730267565345189,1.0,0.0,0.0,0.0,0.0,0.0,0.0,-1.0,-0.0,-0.0,-0.0,-0.0,-0.0,-0.0,4.0804175883443991E-6,
        0.10730267565346296,-0.0014580885500774404,-1.9335790139465064E-6,-4.7482357791108593E-5,1.0,0.0,0.0,0.0,
        0.0,0.0,0.0,-1.0,-0.0,-0.0,-0.0,-0.0,-0.0,-0.0,0.0014580885500775395,4.8607390528308585E-6,
        2.1510651883718012E-9,-1.9335798739413384E-6,1.0,0.0,0.0,0.0,0.0,0.0,0.0,0.0,0.0,-0.0,-0.0,-0.0,-0.0,-0.0,
        -0.0,-0.0,-0.0019439782275025078,-3.0076711049122035E-6,-0.10732396454229663,0.10734524358329482,
        7.9117659047139217E-5,1.0,0.0,0.0,0.0,0.0,0.0,0.0,-1.0,-0.0,-0.0,-0.0,-0.0,-0.0,-0.0,-0.0,
        -0.0029153681735777726,-2.3633272615211667E-6,-7.1207407399672209E-5,9.49404828913434E-5,
        0.10732396454216137,1.0,0.0,0.0,0.0,0.0,0.0,0.0,-1.0,-0.0,-0.0,-0.0,-0.0,-0.0,-0.0,-0.0043710401679813533,
        -3.00766972716206E-6,3.00766972716206E-6,0.10730267565385779,4.2945099842947386E-6,1.0,0.0,0.0,0.0,0.0,0.0,
        0.0,0.0,-1.0,-0.0,-0.0,-0.0,-0.0,-0.0,-0.0,-0.0,-1.9335798739413388E-6,-0.0,-0.0014580885500771513,
        -3.0076718320980626E-6,1.0,0.0,0.0,0.0,0.0,0.0,0.0,-1.0,-0.0,-0.0,-0.0,-0.0,-0.0,-0.0,-0.0,-0.0,
        -0.0029153681735763757,-3.6517565921765191E-6,1.9335782701010321E-6,0.10733105865305884,0.10732396454219453,
        1.0,0.0,0.0,0.0,0.0,0.0,0.0,-1.0,-0.0,-0.0,-0.0,-0.0,-0.0,-0.0,-0.0,-0.0019439782275007787,
        -4.2945123409764109E-6,2.3633289900036141E-6,0.10734524358332284,3.6517597006641474E-6,1.0,0.0,0.0,0.0,0.0,
        0.0,0.0,-1.0,-0.0,-0.0,-0.0,-0.0,-0.0,-0.0,-0.0,-0.0048557677525883714,-4.7482226567215337E-5,
        1.93357760066366E-6,0.0034008125243890257,1.0,0.0,0.0,0.0,0.0,0.0,0.0,-1.0,-0.0,-0.0,-0.0,-0.0,-0.0,-0.0,
        -0.0,-1.9335720080464035E-6,-8.5991207447538975E-9,-0.0029153681735784465,-0.0048557677525916908,
        0.0029153681735784465,0.0048557677525916908,1.0,0.0,0.0,0.0,0.0,0.0,0.0,-1.0,-0.0,-0.0,-0.0,-0.0,-0.0,-0.0,
        -0.0,-0.0,-1.9335775788885911E-6,-0.0048557677525913837,0.003400812524391244,4.7482240979622037E-5,1.0,0.0,
        0.0,0.0,0.0,0.0,0.0,-1.0,-0.0,-0.0,-0.0,-0.0,-0.0,-0.0,-0.0,-1.9335790357216355E-6,-8.5991721612054924E-9,
        -4.860738314554515E-6,0.0014580885500786493,1.0,0.0,0.0,0.0,0.0,0.0,0.0,-1.0,-0.0,-0.0,-0.0,-0.0,-0.0,-0.0,
        -0.0,-0.0,-3.0076700444252484E-6,-0.10730267565351387,0.0014580885500771522,7.9117617963562058E-5,1.0,0.0,
        0.0,0.0,0.0,0.0,0.0,0.0,-1.0,-0.0,-0.0,-0.0,-0.0,-0.0,-0.0,-0.0,-0.001458088550069777,-0.10730267567349638,
        -3.0076718320980626E-6,-4.2945136019776164E-6,3.0076718320980626E-6,4.2945136019776156E-6,1.0,0.0,0.0,0.0,
        0.0,0.0,0.0,-1.0,-0.0,-0.0,-0.0,-0.0,-0.0,-0.0,-0.0,-0.0,0.0048557677525883714,-3.6517549158460076E-6,
        -0.0019439782275030254,-0.0034008125243890231,1.933577600663661E-6,1.0,0.0,0.0,0.0,0.0,0.0,0.0,-1.0,-0.0,
        -0.0,-0.0,-0.0,-0.0,-0.0,3.00766972716206E-6,0.0043710401680015594,-0.0014580885008721894,
        -7.9117605590559628E-5,-0.10730267565351385,1.0,0.0,0.0,0.0,0.0,0.0,3.0076718320980626E-6,-0.0,
        0.0014580885500786506,1.9335798739413379E-6,1.0,0.0,0.0,0.0,0.0,0.0,0.0,0.0,0.0,0.0,-0.0,-0.0,-0.0,-0.0,
        -0.0,-0.0,0.0029153681735761866,4.08041502905828E-6,-1.9335782483259365E-6,-0.1073310586530794,
        -4.7482282067983659E-5,1.0,0.0,0.0,0.0,0.0,0.0,0.0,-0.0,-0.0,-0.0,-0.0,0.0034008125243717882,
        -0.0014580885500697779,-3.007670044425248E-6,-4.2945105315273461E-6,3.007670044425248E-6,
        4.2945105315273452E-6,1.0,0.0,0.0,0.0,0.0,0.0,0.0,0.0,-1.0,-0.0,-0.0,-0.0,-0.0,-0.0,-0.0,
        0.0014580885500771524,4.8607390528298328E-6,-3.0076718320980622E-6,7.91176878824381E-5,
        7.1207546828773829E-5,1.0,0.0,0.0,0.0,0.0,0.0,0.0,0.0,0.0,-0.0,-0.0,-0.0,-0.0,-0.0,-0.0,-0.0,-0.0,
        0.0048557677525832323,-4.2945052010659752E-6,-0.0019439782275007791,-0.0034008125243852206,
        3.6517549158460084E-6,1.0,0.0,0.0,0.0,0.0,0.0,0.0,-1.0,-0.0,-0.0,-0.0,-0.0,-0.0,-0.0,0.001943978227503025,
        0.10732396454219449,-3.6517597006641465E-6,-0.10734524358314684,1.9335795383227379E-6,1.0,0.0,0.0,0.0,0.0,
        0.0,0.0,-1.0,-0.0,-0.0,-0.0,-0.0,-0.0,-0.0,0.0043710401680015594,-3.00766972716206E-6,
        -0.0014580885008721894,-0.10730267565351391,7.911760559055956E-5,1.0,0.0,0.0,0.0,0.0,0.0,0.0,-1.0,-0.0,-0.0,
        -0.0,-0.0,-0.0,-0.0,0.0029153681735777726,-2.3633272615211667E-6,-7.1207407399672209E-5,
        -0.10733105865302138,9.49404828913434E-5,1.0,0.0,0.0,0.0,0.0,0.0,-0.0,-0.0,-0.0,-0.0,-0.0,
        0.0014580885500786503,-1.9335798739413384E-6,1.0,0.0,0.0,0.0,0.0,0.0,0.0,0.0,-1.0,-0.0,-0.0,-0.0,-0.0,-0.0,
        -0.0,-0.0,4.7481714139195575E-5,-0.0029153681735763757,-1.933572008046404E-6,-0.0048557677525883705,
        0.0029153681735763757,0.0048557677525883705,1.0,0.0,0.0,0.0,0.0,0.0,0.0,0.0,-1.0,-0.0,-0.0,-0.0,-0.0,-0.0,
        -0.0,-0.0,4.08041502905828E-6,-0.0029153681735761866,-1.9335782483259365E-6,-4.7482282067983659E-5,
        0.10732396454221274,1.0,0.0,0.0,0.0,0.0,0.0,0.0,-1.0,-0.0,-0.0,-0.0,-0.0,-0.0,-0.0,4.0804203244432527E-6,
        -0.0014580885500774393,-0.10734524358317282,-1.9335798521661753E-6,-4.7482431788502411E-5,1.0,0.0,0.0,0.0,
        0.0,0.0,-0.0,-0.0,-0.0,-0.0,-0.0,1.9335776006636597E-6,2.1510568707557297E-9,-1.6202461970817254E-5,
        0.0034008125243914678,1.0,0.0,0.0,0.0,0.0,0.0,0.0,0.0,-1.0,-0.0,-0.0,-0.0,-0.0,-0.0,-0.0,
        1.9335795165475876E-6,7.9117659047139339E-5,-0.0019439782275043384,-0.10732396454214821,
        -4.7482414627862796E-5,0.10734524358308199,0.0,0.0,0.0,0.0,0.0,0.0,-1.0,-0.0,-0.0,-0.0,-0.0,-0.0,-0.0,
        4.0804128508300446E-6,-0.0048557677525880643,-1.9335775788885915E-6,-4.748222656721529E-5,
        0.0034008125243888041,1.0,0.0,0.0,0.0,0.0,0.0,-0.0,-0.0,-0.0,-0.0,1.933579013946506E-6,
        7.9117617963562125E-5,-0.10730267565342244,-4.74823722035114E-5,0.0014580885500785517,1.0,0.0,0.0,0.0,0.0,
        0.0,0.0,0.0,-1.0,-0.0,-0.0,-0.0,-0.0,-0.0,3.0076718320980626E-6,-0.0014580885500771511,
        -9.7214812475719144E-6,-7.9117687882438126E-5,-7.12075468287738E-5,1.0,0.0,0.0,0.0,0.0,0.0,0.0,-1.0,-0.0,
        -0.0,-0.0,-0.0,-0.0,-0.0,-0.0,-0.0,0.0043710401680023868,4.0804171032462154E-6,-0.0014580885008724769,
        -1.9335788647002392E-6,-0.10730267565346287,-4.7482344040746457E-5,1.0,0.0,0.0,0.0,0.0,0.0,-1.0,-0.0,-0.0,
        -0.0,-0.0,-0.0,1.9335788864753615E-6,0.0043710401680056906,4.7482358453149714E-5,-0.001458088500873688,
        -0.1073026756534111,1.0,0.0,0.0,0.0,0.0,0.0,0.0,0.0,-1.0,-0.0,-0.0,-0.0,-0.0,-0.0,0.10730267565351388,
        -3.0076700444252476E-6,-0.0014580885500771531,7.9117617963562058E-5,7.1207475890096072E-5,1.0,0.0,0.0,0.0,
        0.0,0.0,0.0,0.0,-0.0,-0.0,-0.0,-0.0,-0.0,-0.0,-0.0,0.0014580885500774415,4.0804203244432527E-6,
        0.10730267567310167,-1.9335798521661745E-6,-4.7482431788502546E-5,1.0,0.0,0.0,0.0,0.0,0.0,0.0,0.0,-0.0,-0.0,
        -0.0,-0.0,-0.0,-0.0,4.7482282067983856E-5,-0.0029153681735763757,-1.9335782701010321E-6,0.10732396454219453,
        1.0,0.0,0.0,0.0,0.0,0.0,0.0,0.0,-1.0,-0.0,-0.0,-0.0,-0.0,-0.0,-0.0,-0.0,0.0014580885008725769,
        -0.10730267567309039,0.0029153681735763757,4.7482282067983849E-5,-1.9335782701010313E-6,1.0,0.0,0.0,0.0,0.0,
        0.0,0.0,0.0,-1.0,-0.0,-0.0,-0.0,-0.0,-0.0,-0.0,-0.0,-0.0019439782275044689,0.0,1.9335798739413379E-6,
        -0.001458088550078649,1.0,0.0,0.0,0.0,0.0,0.0,0.0,0.0,-1.0,-0.0,-0.0,-0.0,-0.0,-0.0,-0.0,-0.0,
        -0.0029153681735784474,-1.9335782701010317E-6,-9.4940482891343363E-5,0.10733105865298573,
        0.10732396454213002,1.0,0.0,0.0,0.0,0.0,0.0,0.0,-1.0,-0.0,-0.0,-0.0,-0.0,-0.0,-0.0,-0.0,-0.0,
        -0.0014580885500775386,-9.7214812475745351E-6,-2.1510651883718012E-9,1.9335798739413392E-6,1.0,0.0,0.0,0.0,
        0.0,0.0,0.0,-1.0,-0.0,-0.0,-0.0,-0.0,-0.0,-0.0,-0.0,-0.0,-0.0019439782275039968,-2.3633289900036145E-6,
        -7.1207517308923953E-5,0.10734524358310082,9.4940584559599059E-5,1.0,0.0,0.0,0.0,0.0,0.0,0.0,-1.0,-0.0,-0.0,
        -0.0,-0.0,-0.0,-0.0,-0.0,-4.0804128508300438E-6,-0.0048557677525880643,1.9335775788885924E-6,1.0,0.0,0.0,
        0.0,0.0,0.0,0.0,-1.0,-0.0,-0.0,-0.0,-0.0,-0.0,-0.0,-0.0,-0.0,1.6202461970817257E-5,-1.93357760066366E-6,
        -0.0019439782275044698,-0.0034008125243914626,1.0,0.0,0.0,0.0,0.0,0.0,0.0,-1.0,-0.0,-0.0,-0.0,-0.0,-0.0,
        -0.0,-0.0,-0.10730267565345171,-4.748235779110858E-5,0.001458088550077539,1.9335790357216359E-6,1.0,0.0,0.0,
        0.0,0.0,0.0,0.0,0.0,-1.0,-0.0,-0.0,-0.0,-0.0,-0.0,-0.0,-0.0,0.0034008125243890218,-3.651758466558632E-6,
        -0.00145808855007754,1.9335790357216364E-6,1.0,0.0,0.0,0.0,0.0,0.0,0.0,-1.0,-0.0,-0.0,-0.0,-0.0,-0.0,-0.0,
        3.0076700444252484E-6,0.10730267565351383,-0.0014580885500771531,-7.9117617963562125E-5,1.0,0.0,0.0,0.0,0.0,
        0.0,0.0,0.0,-1.0,-0.0,-0.0,-0.0,-0.0,-0.0,-0.0,-0.0,0.0014580885008736878,1.9335797246950135E-6,
        1.4582219314857481E-5,2.1510655448475862E-9,-0.00048607385598572941,1.0,0.0,0.0,0.0,0.0,0.0,0.0,0.0,0.0,
        -1.0,-0.0,-0.0,-0.0,-0.0,-0.0,0.0034008125243852206,-4.2945105315273461E-6,-0.0014580885500758134,
        3.6517584665586341E-6,1.0,0.0,0.0,0.0,0.0,0.0,0.0,-1.0,-0.0,-0.0,-0.0,-0.0,-0.0,-0.0,0.0014580885500782884,
        4.8607390528328906E-6,-2.3633294499635062E-6,4.299588718831751E-7,1.0,0.0,0.0,0.0,0.0,0.0,0.0,0.0,0.0,-0.0,
        -0.0,-0.0,-0.0,-0.0,-0.0,-0.0,-0.0,0.0014580885500775395,9.7214812475745182E-6,-1.8267965878074558E-8,
        1.9335798739413384E-6,1.0,0.0,0.0,0.0,0.0,0.0,0.0,0.0,-1.0,-0.0,-0.0,-0.0,-0.0,-0.0,-0.0,
        0.0014580885008733254,0.10733105865302135,-2.3633292478225708E-6,-0.10730267567306921,9.4940600341471287E-5,
        1.0,0.0,0.0,0.0,0.0,0.0,0.0,0.0,-1.0,-0.0,-0.0,-0.0,-0.0,-0.0,-0.0,4.0804175883444E-6,-0.10730267565346309,
        -1.9335790139465055E-6,-4.748235779110841E-5,0.0014580885500774404,1.0,0.0,0.0,0.0,0.0,0.0,0.0,-0.0,-0.0,
        -0.0,-0.0,4.0804192061118553E-6,-0.0019439782275028953,-0.10732396454221274,-1.9335795165475888E-6,
        -4.7482400215460934E-5,0.10734524358317275,0.0,0.0,0.0,0.0,0.0,-1.0,-0.0,-0.0,-0.0,-0.0,-0.0,-0.0,
        1.9335798521661749E-6,1.0750244040852593E-8,-0.0014580885500785506,-9.7214812475805728E-6,
        -2.1510659495834055E-7,1.0,0.0,0.0,0.0,0.0,0.0,0.0,-1.0,-0.0,-0.0,-0.0,-0.0,-0.0,-0.0,2.1510651883718025E-9,
        -0.0014580885500775382,-9.7214812475745487E-6,-1.9335798739413375E-6,1.0,0.0,0.0,0.0,0.0,0.0,0.0,-1.0,-0.0,
        -0.0,-0.0,-0.0,-0.0,-0.0,-0.0,-0.0,4.7482226567215236E-5,-0.0048557677525883714,-1.9335776006636593E-6,
        0.0034008125243890257,1.0,0.0,0.0,0.0,0.0,0.0,0.0,-1.0,-0.0,-0.0,-0.0,-0.0,-0.0,-0.0,-0.0,
        1.9335790357216347E-6,2.151062815512053E-9,-4.8607383145545141E-6,0.0014580885500786495,1.0,0.0,0.0,0.0,0.0,
        0.0,0.0,0.0,0.0,-1.0,-0.0,-0.0,-0.0,-0.0,-0.0,-0.0,1.9335790357216347E-6,4.8607383145545243E-6,
        2.1510628155120546E-9,-0.001458088550078651,1.0,0.0,0.0,0.0,0.0,0.0,0.0,0.0,0.0,-0.0,-0.0,-0.0,-0.0,-0.0,
        -0.0,0.10730267565343037,-2.3633283044492367E-6,-0.0014580885500782882,9.49405441466369E-5,1.0,0.0,0.0,0.0,
        0.0,0.0,0.0,0.0,-0.0,-0.0,-0.0,-0.0,-0.0,-0.0,-0.0,-0.0,4.7482400215460934E-5,-0.001943978227503025,
        -1.933579538322737E-6,0.10734524358314687,1.0,0.0,0.0,0.0,0.0,0.0,0.0,0.0,-1.0,-0.0,-0.0,-0.0,-0.0,-0.0,
        -0.0,-0.0,1.7012593526672186E-5,-1.9335790357216355E-6,-8.5991721612054841E-9,-0.0014580885500786501,1.0,
        0.0,0.0,0.0,0.0,0.0,0.0,-1.0,-0.0,-0.0,-0.0,-0.0,-0.0,-0.0,-0.0,1.933579013946506E-6,7.9117617963562125E-5,
        0.10730267565342247,-0.0014580885500785515,-4.7482372203511207E-5,1.0,0.0,0.0,0.0,0.0,0.0,0.0,0.0,-0.0,-0.0,
        -0.0,-0.0,-0.0,-0.0,0.0043710401680047061,-2.3633281023083708E-6,-0.0014580885008733248,
        -0.10730267565343046,9.494053246254531E-5,1.0,0.0,0.0,0.0,0.0,0.0,0.0,-1.0,-0.0,-0.0,-0.0,-0.0,-0.0,-0.0,
        4.7482357791108451E-5,-0.10730267565345164,-1.9335790357216359E-6,0.0014580885500775384,1.0,0.0,0.0,0.0,0.0,
        0.0,0.0,0.0,-1.0,-0.0,-0.0,-0.0,-0.0,-0.0,-0.0,-0.0,-5.5781067902885632E-6,-0.0029166379626661808,
        -7.9656733204749716E-6,-0.0048578821565158263,5.5781067902885632E-6,0.0029166379626661808,
        7.9656733204749716E-6,0.0048578821565158263,0.0,1.0,0.0,0.0,0.0,0.0,0.0,0.0,-0.0,-1.0,-0.0,-0.0,-0.0,-0.0,
        -0.0,-0.0,5.5781067902885632E-6,-0.002916637962691824,-0.00014679953284411136,-0.00013212894189010106,
        -0.0048578821565599525,0.002916637962691824,0.0048578821565599525,0.0,1.0,0.0,0.0,0.0,0.0,0.0,0.0,-0.0,-1.0,
        -0.0,-0.0,-0.0,-0.0,-0.0,-0.0,0.0029166379626661808,-5.57812021349215E-6,-0.10736632614517246,
        -7.9656949033694517E-6,-0.10736031682307962,5.57812021349215E-6,7.9656949033694517E-6,0.0,1.0,0.0,0.0,0.0,
        0.0,0.0,0.0,-0.0,-1.0,-0.0,-0.0,-0.0,-0.0,-0.0,-0.0,7.96567332047497E-6,-4.3826144576171757E-6,
        -0.0029166379626858318,-6.7727808307423184E-6,0.00485788215654968,0.0,1.0,0.0,0.0,0.0,0.0,0.0,-0.0,-1.0,
        -0.0,-0.0,-0.0,-0.0,-0.0,-0.0,-5.5781067902885632E-6,-0.002916637962691824,-0.0048578821565599525,
        0.002916637962691824,0.00014679953284411142,0.00013212894189010114,0.0048578821565599525,0.0,1.0,0.0,0.0,
        0.0,0.0,0.0,0.0,-0.0,-1.0,-0.0,-0.0,-0.0,-0.0,-0.0,-0.0,-0.0029166379626661808,-5.57812021349215E-6,
        -7.9656949033694517E-6,5.57812021349215E-6,0.10736632614517246,7.9656949033694517E-6,0.10736031682307967,
        0.0,1.0,0.0,0.0,0.0,0.0,0.0,0.0,-0.0,-1.0,-0.0,-0.0,-0.0,-0.0,-0.0,-0.0,-7.96567332047497E-6,
        -0.0029166379626858318,-0.00485788215654968,0.0029166379626858318,6.7727808307423209E-6,0.00485788215654968,
        0.0,1.0,0.0,0.0,0.0,0.0,0.0,-0.0,-1.0,-0.0,-0.0,-0.0,-0.0,-0.0,-0.0,-0.0048578821565158281,
        -5.5781196549432766E-6,7.5683539998422573E-6,0.0034022935815205772,7.96569403167477E-6,0.0,1.0,0.0,0.0,0.0,
        0.0,0.0,-0.0,-1.0,-0.0,-0.0,-0.0,-0.0,-0.0,-0.0,5.5781202134921511E-6,0.0029166379626918235,
        -0.00014679999446733945,-0.10736632614478582,-0.00013212939324542828,0.0,1.0,0.0,0.0,0.0,0.0,0.0,0.0,-0.0,
        -1.0,-0.0,-0.0,-0.0,-0.0,-0.0,-0.0,0.00013212894189010104,3.5853869352593028E-6,-0.0029166379626963646,
        -0.0048578821565677952,0.0029166379626963646,0.0048578821565677952,0.0,1.0,0.0,0.0,0.0,0.0,0.0,0.0,0.0,-0.0,
        -1.0,-0.0,-0.0,-0.0,-0.0,-0.0,5.5781202134921511E-6,-0.0,3.5853940506334835E-6,-0.0029166379626961035,
        -8.8129233469058372E-5,0.10736632614469463,0.0,1.0,0.0,0.0,0.0,0.0,0.0,0.0,-0.0,-1.0,-0.0,-0.0,-0.0,-0.0,
        -0.0,5.5781196549432774E-6,-0.0048578821565599534,-0.00014679997713426275,-0.00013212937592219681,
        0.00340229358155005,0.0,1.0,0.0,0.0,0.0,0.0,0.0,-0.0,-1.0,-0.0,-0.0,-0.0,-0.0,-0.0,-0.0,
        0.0014587235451840523,0.10736632614517241,-5.5781237935757988E-6,-7.9657006639635273E-6,
        -0.10734228894828789,5.5781237935757988E-6,7.9657006639635273E-6,0.0,1.0,0.0,0.0,0.0,0.0,0.0,0.0,-0.0,-1.0,
        -0.0,-0.0,-0.0,-0.0,0.0029166379626918244,0.00014679999446733951,-0.0,0.0014587235944407036,
        -5.5781242224138721E-6,0.0,1.0,0.0,0.0,0.0,0.0,0.0,0.0,0.0,-0.0,-1.0,-0.0,-0.0,-0.0,-0.0,-0.0,
        0.0029166379626858318,-7.96569490336945E-6,-0.10736632614482629,-0.10736031682276148,6.7727967124435443E-6,
        0.0,1.0,0.0,0.0,0.0,0.0,0.0,-0.0,-1.0,-0.0,-0.0,-0.0,-0.0,-0.0,-0.0,8.8129282461975545E-5,
        0.1073422889303401,-3.5853953767303946E-6,-0.0014587235944407545,0.0,1.0,0.0,0.0,0.0,0.0,0.0,0.0,-1.0,-0.0,
        -0.0,-0.0,-0.0,-0.0,-0.0,-5.5781202134921511E-6,-0.0029166379626918235,0.10736632614478582,
        0.00013212939324542836,0.1073603168227252,0.0,1.0,0.0,0.0,0.0,0.0,0.0,0.0,-0.0,-1.0,-0.0,-0.0,-0.0,-0.0,
        -0.0,-0.0,-3.5853868948616202E-6,-0.00014679953284411131,-0.0029166379626961044,8.8128812909480433E-5,0.0,
        1.0,0.0,0.0,0.0,0.0,-0.0,-1.0,-0.0,-0.0,-0.0,-0.0,-0.0,-0.0,-0.0,-5.5781196549432774E-6,
        -0.0048578821565599534,0.0001467999771342628,0.00340229358155005,0.00013212937592219689,0.0,1.0,0.0,0.0,0.0,
        0.0,0.0,-0.0,-1.0,-0.0,-0.0,-0.0,-0.0,-0.0,-0.0,-0.0014587235944378964,-0.0,-0.0029166379626858318,
        -7.96569490336945E-6,6.7727967124435443E-6,0.0,1.0,0.0,0.0,0.0,0.0,0.0,-0.0,-1.0,-0.0,-0.0,-0.0,-0.0,-0.0,
        -0.0,-0.0019448249244416718,-5.5781234578900866E-6,-7.96570013580131E-6,5.5781234578900866E-6,
        0.10737834481916497,7.96570013580131E-6,0.0,1.0,0.0,0.0,0.0,0.0,0.0,0.0,-0.0,-1.0,-0.0,-0.0,-0.0,-0.0,-0.0,
        -0.0,-8.8128786203203676E-5,-0.0029166379626919731,-0.0048578821565602656,3.5853869352593007E-6,
        0.0029166379626919731,0.0048578821565602656,0.0,1.0,0.0,0.0,0.0,0.0,0.0,0.0,-0.0,-1.0,-0.0,-0.0,-0.0,-0.0,
        -0.0,-0.0,-7.9656940316747675E-6,-0.00485788215654968,6.772796075194699E-6,0.0034022935815431017,0.0,1.0,
        0.0,0.0,0.0,0.0,-0.0,-1.0,-0.0,-0.0,-0.0,-0.0,-0.0,-0.0,-0.0034022935815205789,-5.5781226566483114E-6,
        -7.96569884454493E-6,5.5781226566483114E-6,0.0014587235944287249,7.96569884454493E-6,0.0,1.0,0.0,0.0,0.0,
        0.0,0.0,-0.0,-1.0,-0.0,-0.0,-0.0,-0.0,-0.0,-0.0,3.5853940506334839E-6,0.0029166379626961035,
        0.00014679999446733945,-0.10736632614469459,-8.8129233469058183E-5,0.0,1.0,0.0,0.0,0.0,0.0,
        0.10736632614469463,5.578124222413873E-6,0.0014587235944407021,-0.00014680013327850644,0.0,1.0,0.0,0.0,0.0,
        0.0,0.0,0.0,0.0,-0.0,-1.0,-0.0,-0.0,-0.0,-0.0,-0.0,0.00013212937592219689,3.5853937677987673E-6,
        -0.0048578821565677943,0.0034022935815552356,0.0,1.0,0.0,0.0,0.0,0.0,0.0,0.0,-0.0,-1.0,-0.0,-0.0,-0.0,-0.0,
        -0.0,5.578124222413873E-6,-0.0014587235944407021,-0.10737834481871872,-0.00014680013327850644,
        -0.00013212952863946446,0.0,1.0,0.0,0.0,0.0,0.0,0.0,-0.0,-1.0,-0.0,-0.0,-0.0,-0.0,-0.0,-0.0,-0.0,
        5.5781226566483131E-6,-0.0034022935815500518,-0.00014680007971837686,-0.00013212947610804457,
        0.0014587235944407036,0.0,1.0,0.0,0.0,0.0,0.0,0.0,-0.0,-1.0,-0.0,-0.0,-0.0,-0.0,-0.0,-0.0,
        0.0043729436145978759,-5.5781222278103542E-6,-0.0014587235451840519,-7.9656981485267E-6,
        -0.10734228893062275,5.5781222278103542E-6,7.9656981485267E-6,0.0,1.0,0.0,0.0,0.0,0.0,0.0,-0.0,-0.0,-0.0,
        -0.0,-0.0,0.001458723594428726,4.8628574262462892E-6,-5.5781242224138721E-6,-7.96570135998195E-6,
        5.5781242224138721E-6,7.96570135998195E-6,0.0,1.0,0.0,0.0,0.0,0.0,0.0,0.0,0.0,-0.0,-1.0,-0.0,-0.0,-0.0,-0.0,
        -0.0,0.0014587235451932238,0.10736632614482625,-7.9657006639635256E-6,-0.10734228894806333,
        6.7728009630617377E-6,0.0,1.0,0.0,0.0,0.0,0.0,0.0,-0.0,-1.0,-0.0,-0.0,-0.0,-0.0,0.0029166379626951724,
        -4.3826237958274972E-6,-0.00013212939324542831,-0.10736632614470672,0.0001761469804713228,1.0,0.0,0.0,0.0,
        0.0,-0.0,-0.0,0.0029166379626919727,-8.81292067627653E-5,-0.10736632614473689,-0.10736031682267945,
        3.5853940910313566E-6,0.0,1.0,0.0,0.0,0.0,0.0,0.0,0.0,-0.0,-1.0,-0.0,-0.0,-0.0,-0.0,-0.0,-0.0,
        7.5683583927445344E-6,0.1073422889303461,-3.5853953363324838E-6,-0.0014587235944406305,
        -8.8129282461975368E-5,0.0,1.0,0.0,0.0,0.0,0.0,0.0,-0.0,-1.0,-0.0,-0.0,-0.0,-0.0,-0.0,0.0043729436146373712,
        8.81292687047112E-5,-3.5853951531698713E-6,-0.0014587235451960796,-0.10734228893034015,0.0,1.0,0.0,0.0,0.0,
        0.0,0.0,-0.0,-1.0,-0.0,-0.0,-0.0,-0.0,-0.0,3.5853953767303946E-6,3.9921984431992029E-9,
        4.8628566874294387E-6,-0.0014587235944428152,0.0,1.0,0.0,0.0,0.0,0.0,0.0,0.0,0.0,-1.0,-0.0,-0.0,-0.0,-0.0,
        -0.0,-0.0,-4.382623795827498E-6,-0.0029166379626951715,-0.00013212939324542831,0.0001761469804713228,
        0.10736632614470674,0.0,1.0,0.0,0.0,0.0,0.0,0.0,-0.0,-1.0,-0.0,-0.0,-0.0,-0.0,-0.0,-0.0,
        -5.5781234578900866E-6,-0.00194482492445803,-0.10736031682272522,0.10737834481871866,0.00013212950321312466,
        0.0,1.0,0.0,0.0,0.0,0.0,0.0,-0.0,-1.0,-0.0,-0.0,-0.0,-0.0,-0.0,-7.5683351098736605E-6,
        -0.0029166379626917129,0.0029166379626917129,8.812878620320373E-5,0.0048578821565598181,0.0,1.0,0.0,0.0,0.0,
        0.0,0.0,0.0,-0.0,-1.0,-0.0,-0.0,-0.0,-0.0,-0.0,-0.0,-0.0014587235944428139,-0.0,-3.5853940910313566E-6,
        -0.0029166379626963642,0.0,1.0,0.0,0.0,0.0,0.0,0.0,-0.0,-1.0,-0.0,-0.0,-0.0,-0.0,-0.0,-0.0,-0.0,
        -5.5781226566483131E-6,-0.0034022935815500518,0.0014587235944407036,0.00014680007971837694,
        0.00013212947610804465,0.0,1.0,0.0,0.0,0.0,0.0,0.0,-0.0,-1.0,-0.0,-0.0,-0.0,-0.0,-0.0,-0.0,
        -4.382623394054422E-6,-0.0048578821565657317,0.0019448249244601577,0.00017614696311855576,
        0.0034022935815538713,0.0,1.0,0.0,0.0,0.0,0.0,0.0,-0.0,-1.0,-0.0,-0.0,-0.0,-0.0,-0.0,-0.0,
        -7.9656988445449321E-6,-0.10734228893039816,0.0014587235944378966,6.7727996274547443E-6,0.0,1.0,0.0,0.0,0.0,
        0.0,0.0,-0.0,-1.0,-0.0,-0.0,-0.0,-0.0,-0.0,-0.0,-0.001458723594428726,-9.7257170977077227E-6,
        -5.5781242224138721E-6,-7.96570135998195E-6,5.5781242224138721E-6,7.96570135998195E-6,0.0,1.0,0.0,0.0,0.0,
        0.0,0.0,-0.0,-1.0,-0.0,-0.0,-0.0,-0.0,-0.0,-0.0,-0.0,-0.0014587235451932238,-7.9657006639635256E-6,
        6.7728009630617377E-6,0.10734228894806358,0.0,1.0,0.0,0.0,0.0,0.0,0.0,-0.0,-1.0,-0.0,-0.0,-0.0,-0.0,-0.0,
        -0.0,-0.0014587235944407539,-9.7257170977957972E-6,-3.9921988676707509E-9,3.5853962153152245E-6,0.0,1.0,0.0,
        0.0,0.0,0.0,0.0,-0.0,-1.0,-0.0,-0.0,-0.0,-0.0,-0.0,-0.0,-0.0,-0.0029166379626919727,-8.81292067627653E-5,
        3.5853940910313566E-6,0.10736632614473689,0.0,1.0,0.0,0.0,0.0,0.0,0.0,0.0,-0.0,-1.0,-0.0,-0.0,-0.0,-0.0,
        -0.0,-0.0,-3.5853869352593015E-6,-8.8128812909480257E-5,-0.0029166379626963646,-0.0048578821565677952,
        0.0029166379626963646,0.0048578821565677952,0.0,1.0,0.0,0.0,0.0,0.0,0.0,-0.0,-1.0,-0.0,-0.0,-0.0,-0.0,-0.0,
        -0.0,-0.0,7.9656988445449321E-6,-0.0034022935815431021,-4.3826254890315264E-6,-6.7727996274547417E-6,
        0.0014587235944378966,0.0,1.0,0.0,0.0,0.0,0.0,0.0,-0.0,-1.0,-0.0,-0.0,-0.0,-0.0,-0.0,0.0029166379626917134,
        7.5683547934316421E-6,-3.5853940506334814E-6,-0.10736632614474596,-8.8129206762765054E-5,0.0,1.0,0.0,0.0,
        0.0,0.0,0.0029166379626963642,-0.0,3.5853962153152266E-6,0.0014587235944428139,0.0,1.0,0.0,0.0,0.0,0.0,0.0,
        0.0,0.0,0.0,-1.0,-0.0,-0.0,-0.0,-0.0,-0.0,5.578122227810355E-6,0.0043729436146371257,-0.0014587235451960297,
        -0.00014680006459902122,-0.10734228893037383,0.0,1.0,0.0,0.0,0.0,0.0,0.0,-0.0,-0.0,-0.0,-0.0,
        6.7727808307423184E-6,-3.5853869352593024E-6,-0.0029166379626919731,-0.0048578821565602656,
        0.0029166379626919731,0.0048578821565602656,0.0,1.0,0.0,0.0,0.0,0.0,0.0,0.0,-0.0,-1.0,-0.0,-0.0,-0.0,-0.0,
        -0.0,3.585394091031357E-6,3.9921950140726025E-9,-0.0029166379626963637,0.10736632614468547,
        0.10736031682263265,0.0,1.0,0.0,0.0,0.0,0.0,0.0,0.0,0.0,-1.0,-0.0,-0.0,-0.0,-0.0,-0.0,-0.0,-0.0,
        7.9656940316747675E-6,-0.00485788215654968,-4.3826233940544228E-6,-6.7727960751946965E-6,
        0.0034022935815431017,0.0,1.0,0.0,0.0,0.0,0.0,0.0,-0.0,-1.0,-0.0,-0.0,-0.0,-0.0,-0.0,4.3826254890315255E-6,
        0.00013212947610804468,-0.0034022935815538747,-0.00017614707050012452,0.0014587235944422637,0.0,1.0,0.0,0.0,
        0.0,0.0,0.0,-0.0,-1.0,-0.0,-0.0,-0.0,-0.0,-0.0,7.5683547934316421E-6,-0.0029166379626917125,
        -3.5853940506334814E-6,-8.8129206762765257E-5,0.10736632614474599,0.0,1.0,0.0,0.0,0.0,0.0,0.0,-0.0,-1.0,
        -0.0,-0.0,-0.0,-0.0,-0.0,5.5781234578900866E-6,-0.00194482492445803,-0.10736031682272522,
        -0.00014680010716724076,0.10737834481871866,0.0,1.0,0.0,0.0,0.0,0.0,-0.0,-0.0,-0.0,-0.0,-0.0,
        3.5853962153152266E-6,-0.001458723594442813,0.0,1.0,0.0,0.0,0.0,0.0,0.0,0.0,-0.0,-1.0,-0.0,-0.0,-0.0,-0.0,
        -0.0,-0.0,0.10734228893062278,-5.5781226566483114E-6,-0.0014587235944287249,-7.96569884454493E-6,
        5.5781226566483114E-6,7.96569884454493E-6,0.0,1.0,0.0,0.0,0.0,0.0,0.0,0.0,-0.0,-1.0,-0.0,-0.0,-0.0,-0.0,
        -0.0,-0.0,0.0043729436146371257,-5.5781222278103542E-6,-0.0014587235451960297,-0.10734228893037363,
        0.00013212946132927787,0.0,1.0,0.0,0.0,0.0,0.0,0.0,-0.0,-1.0,-0.0,-0.0,-0.0,-0.0,-0.0,0.0043729436146440828,
        -3.5853951531698696E-6,-0.00017614705469946,-0.0014587235451981424,-0.10734228893030787,0.0,1.0,0.0,0.0,0.0,
        0.0,-0.0,-0.0,-0.0,-0.0,-0.0,0.0014587235944378964,4.8628574262843667E-6,-2.6579519435852128E-8,
        6.7728014725786294E-6,0.0,1.0,0.0,0.0,0.0,0.0,0.0,0.0,-0.0,-1.0,-0.0,-0.0,-0.0,-0.0,-0.0,
        0.0014587235451975907,0.10736632614470673,-4.3826262842811432E-6,-0.00013212951386069361,
        -0.10734228894798679,0.00017614711031739875,1.0,0.0,0.0,0.0,0.0,0.0,-0.0,-1.0,-0.0,-0.0,-0.0,-0.0,-0.0,
        0.0043729436146279586,-7.9656981485266989E-6,-0.0014587235451932229,-0.1073422889303981,
        6.772799117937994E-6,0.0,1.0,0.0,0.0,0.0,0.0,-0.0,-0.0,-0.0,-0.0,0.0014587235451960802,0.10736632614473685,
        -8.8129318150789929E-5,-0.10734228894800538,3.5853959917546394E-6,0.0,1.0,0.0,0.0,0.0,0.0,0.0,0.0,-0.0,-1.0,
        -0.0,-0.0,-0.0,-0.0,0.0029166379626963642,-3.5853940910313553E-6,-1.5952356250788457E-8,
        -0.10736632614468547,-0.10736031682263257,0.0,1.0,0.0,0.0,0.0,0.0,0.0,-0.0,-1.0,-0.0,-0.0,-0.0,-0.0,-0.0,
        -0.0,-0.0,7.5683577588589512E-6,0.0043729436146369739,-3.5853951127719673E-6,-0.0014587235451959575,
        -8.8129268704711E-5,-0.10734228893034628,0.0,1.0,0.0,0.0,0.0,0.0,-0.0,-1.0,-0.0,-0.0,-0.0,-0.0,
        0.0014587235944406316,7.5683606848681651E-6,0.1073422889480115,-3.5853961749172934E-6,
        -8.8129331908057959E-5,0.0,1.0,0.0,0.0,0.0,0.0,0.0,0.0,-0.0,-1.0,-0.0,-0.0,-0.0,-0.0,8.8129206762765474E-5,
        -0.0029166379626919727,-3.5853940910313579E-6,0.10736632614473685,0.10736031682267955,0.0,1.0,0.0,0.0,0.0,
        0.0,0.0,0.0,-1.0,-0.0,-0.0,-0.0,-0.0,-0.0,-0.0,3.5853951531698713E-6,0.0043729436146440846,
        8.8129295411006457E-5,-0.0014587235451981398,-0.10734228893030738,0.0,1.0,0.0,0.0,0.0,0.0,0.0,0.0,-1.0,-0.0,
        -0.0,-0.0,-0.0,-0.0,0.10734228893037383,-5.5781226566483106E-6,-0.0014587235944407036,
        0.00013212947610804473,0.0,1.0,0.0,0.0,0.0,0.0,0.0,0.0,-0.0,-1.0,-0.0,-0.0,-0.0,-0.0,-0.0,-0.0,
        3.5853953363324867E-6,-8.8129309168270936E-5,5.5781226566483131E-6,0.10734228893037383,
        -0.0014587235944407036,0.0,1.0,0.0,0.0,0.0,0.0,0.0,0.0,-0.0,-1.0,-0.0,-0.0,-0.0,-0.0,-0.0,-0.0,
        -4.3826265793617967E-6,0.0,0.0014587235944428149,-3.5853962153152249E-6,0.0,1.0,0.0,0.0,0.0,0.0,0.0,0.0,
        -0.0,-1.0,-0.0,-0.0,-0.0,-0.0,-0.0,-0.0,-5.578124222413873E-6,-0.0014587235944407021,-0.10737834481871872,
        0.00014680013327850652,0.00013212952863946454,0.0,1.0,0.0,0.0,0.0,0.0,0.0,-0.0,-1.0,-0.0,-0.0,-0.0,-0.0,
        -0.0,-0.0,-0.0,-3.5853953767303937E-6,-1.5952364404071241E-8,-4.8628566874294387E-6,0.0014587235944428152,
        0.0,1.0,0.0,0.0,0.0,0.0,0.0,-0.0,-1.0,-0.0,-0.0,-0.0,-0.0,-0.0,-0.0,-0.0,-4.3826260449574541E-6,
        -0.0019448249244601575,-0.10736031682265219,0.00017614709863668606,0.10737834481862853,0.0,1.0,0.0,0.0,0.0,
        0.0,0.0,-0.0,-1.0,-0.0,-0.0,-0.0,-0.0,-0.0,-0.0,-0.0043729436146279586,-7.9656981485266989E-6,
        0.0014587235451932229,0.0,1.0,0.0,0.0,0.0,0.0,0.0,-0.0,-1.0,-0.0,-0.0,-0.0,-0.0,-0.0,-0.0,-0.0,
        2.6579519435852128E-8,-0.0014587235944378964,-4.3826265793617976E-6,-6.7728014725786269E-6,0.0,1.0,0.0,0.0,
        0.0,0.0,0.0,-0.0,-1.0,-0.0,-0.0,-0.0,-0.0,-0.0,-0.0,-8.8129282461975545E-5,-0.10734228893034033,
        3.5853953767303929E-6,0.0014587235944407545,0.0,1.0,0.0,0.0,0.0,0.0,0.0,0.0,-0.0,-1.0,-0.0,-0.0,-0.0,-0.0,
        -0.0,-0.0,6.7727996274547409E-6,-0.0034022935815501616,-3.5853953767303946E-6,0.0014587235944407543,0.0,1.0,
        0.0,0.0,0.0,0.0,0.0,-0.0,-1.0,-0.0,-0.0,-0.0,-0.0,-0.0,0.0029166379626919727,8.81292067627653E-5,
        -3.5853940910313583E-6,-0.10736632614473689,0.0,1.0,0.0,0.0,0.0,0.0,0.0,0.0,-0.0,-1.0,-0.0,-0.0,-0.0,-0.0,
        -0.0,-0.0,3.5853961749172947E-6,0.0014587235944426909,1.9944569314633716E-8,4.8628574263039366E-6,
        -3.9922002781882362E-7,0.0,1.0,0.0,0.0,0.0,0.0,0.0,0.0,0.0,-0.0,-1.0,-0.0,-0.0,-0.0,-0.0,
        6.7727960751946948E-6,-0.0048578821565602656,-3.5853937677987677E-6,0.0034022935815501611,0.0,1.0,0.0,0.0,
        0.0,0.0,0.0,-0.0,-1.0,-0.0,-0.0,-0.0,-0.0,-0.0,3.5853958053010422E-6,3.99219962433586E-9,
        -0.001944824924460911,0.00048628580559873565,0.0,1.0,0.0,0.0,0.0,0.0,0.0,0.0,0.0,-1.0,-0.0,-0.0,-0.0,-0.0,
        -0.0,-0.0,-0.0,3.5853953767303946E-6,1.5952364404071224E-8,-1.7020005141606009E-5,0.0014587235944428134,0.0,
        1.0,0.0,0.0,0.0,0.0,0.0,0.0,-0.0,-1.0,-0.0,-0.0,-0.0,-0.0,-0.0,3.5853957649031212E-6,0.00014680010716724078,
        -0.0019448249244607453,-8.8129335242261085E-5,0.10737834481861454,0.0,1.0,0.0,0.0,0.0,0.0,0.0,0.0,-0.0,-1.0,
        -0.0,-0.0,-0.0,-0.0,-0.0,0.00437294361463737,-8.81292687047114E-5,-0.0014587235451960804,
        -0.10734228893034034,3.5853951531698705E-6,0.0,1.0,0.0,0.0,0.0,0.0,0.0,-0.0,-0.0,-0.0,-0.0,
        0.0043729436146422536,-4.3826251939509524E-6,-0.0001321294613292779,-0.00145872354519759,
        -0.10734228893032162,0.00017614705469946011,1.0,0.0,0.0,0.0,0.0,-0.0,-1.0,-0.0,-0.0,-0.0,-0.0,-0.0,
        0.0014587235451981413,1.4588573537945144E-5,-3.5853959917546364E-6,-1.5952368010052985E-8,
        -0.0004862856933051914,0.0,1.0,0.0,0.0,0.0,0.0,0.0,-0.0,-1.0,-0.0,-0.0,-0.0,-0.0,-0.0,4.8628566874294463E-6,
        -3.5853953767303925E-6,-1.5952364404071234E-8,-0.0014587235944428143,0.0,1.0,0.0,0.0,0.0,0.0,0.0,-0.0,-1.0,
        -0.0,-0.0,-0.0,-0.0,-0.0,-0.0,-0.0,0.10734228893039793,-7.9656988445449321E-6,-0.0014587235944378966,
        6.7727996274547443E-6,0.0,1.0,0.0,0.0,0.0,0.0,0.0,-0.0,-1.0,-0.0,-0.0,-0.0,-0.0,-0.0,-0.0,
        0.0014587235944407541,4.8628574262962057E-6,-3.9921988676707517E-9,3.5853962153152254E-6,0.0,1.0,0.0,0.0,
        0.0,0.0,0.0,0.0,0.0,-0.0,-1.0,-0.0,-0.0,-0.0,-0.0,-0.0,0.0014587235944407539,3.99219886767076E-9,
        4.862857426296204E-6,-3.5853962153152254E-6,0.0,1.0,0.0,0.0,0.0,0.0,0.0,0.0,0.0,-1.0,-0.0,-0.0,-0.0,-0.0,
        -0.0,8.8129308535964311E-5,-0.0019448249244580964,-3.5853958053010409E-6,0.10737834481866426,0.0,1.0,0.0,
        0.0,0.0,0.0,0.0,0.0,-1.0,-0.0,-0.0,-0.0,-0.0,-0.0,-0.0,-0.0,0.10734228893032166,-4.3826254890315247E-6,
        -0.001458723594442264,0.0001761470705001243,0.0,1.0,0.0,0.0,0.0,0.0,0.0,0.0,-0.0,-1.0,-0.0,-0.0,-0.0,-0.0,
        -0.0,-0.0,3.3880996868665913E-8,-0.0014587235944407532,-9.725717097795804E-6,-3.5853962153152254E-6,0.0,1.0,
        0.0,0.0,0.0,0.0,0.0,-0.0,-1.0,-0.0,-0.0,-0.0,-0.0,-0.0,-0.0,0.0014587235451960802,0.10736632614473685,
        8.8129318150790078E-5,-3.58539599175464E-6,-0.10734228894800538,0.0,1.0,0.0,0.0,0.0,0.0,0.0,0.0,-1.0,-0.0,
        -0.0,-0.0,-0.0,-0.0,7.5683595662360549E-6,-0.0019448249244579309,-3.5853957649031187E-6,
        -8.8129308535964148E-5,0.10737834481867461,0.0,1.0,0.0,0.0,0.0,0.0,0.0,-0.0,-1.0,-0.0,-0.0,-0.0,-0.0,-0.0,
        0.10734228893034023,-8.8129282461975639E-5,-0.0014587235944407545,3.5853953767303946E-6,0.0,1.0,0.0,0.0,0.0,
        0.0,0.0,0.0,-0.0,-1.0,-0.0,-0.0,-0.0,-0.0,-0.0,-0.0,-1.0694098357603545E-5,-1.2158262884725835E-8,
        -1.90851108625298E-5,-1.7891460877206116E-8,1.0694098357603545E-5,1.2158262884725835E-8,1.90851108625298E-5,
        1.7891460877206119E-8,0.0,0.0,1.0,0.0,0.0,0.0,0.0,0.0,-0.0,-0.0,-1.0,-0.0,-0.0,-0.0,-0.0,-0.0,
        1.0694098357603547E-5,-1.2158312102019979E-8,-0.00045000707549025732,-0.00046403965892872541,
        -1.7891545726468563E-8,1.2158312102019979E-8,1.7891545726468567E-8,0.0,0.0,1.0,0.0,0.0,0.0,0.0,0.0,-0.0,
        -0.0,-1.0,-0.0,-0.0,-0.0,-0.0,-0.0,1.2158262884725835E-8,-1.0694098357659397E-5,-3.482890192621146E-7,
        -1.9085110862619308E-5,-3.1720226087564254E-7,1.0694098357659397E-5,1.9085110862619308E-5,0.0,0.0,1.0,0.0,
        0.0,0.0,0.0,0.0,-0.0,-0.0,-1.0,-0.0,-0.0,-0.0,-0.0,-0.0,1.9085110862529796E-5,-6.4936804961928115E-6,
        -1.215831002246988E-8,-1.2220370768088023E-5,1.7891542245038322E-8,0.0,0.0,1.0,0.0,0.0,0.0,0.0,-0.0,-0.0,
        -1.0,-0.0,-0.0,-0.0,-0.0,-0.0,-1.0694098357603547E-5,-1.2158312102019979E-8,-1.7891545726468563E-8,
        1.2158312102019979E-8,0.00045000707549025732,0.00046403965892872568,1.7891545726468567E-8,0.0,0.0,1.0,0.0,
        0.0,0.0,0.0,0.0,-0.0,-0.0,-1.0,-0.0,-0.0,-0.0,-0.0,-0.0,-1.2158262884725835E-8,-1.0694098357659397E-5,
        -1.9085110862619308E-5,1.0694098357659397E-5,3.482890192621146E-7,1.9085110862619308E-5,
        3.1720226087564292E-7,0.0,0.0,1.0,0.0,0.0,0.0,0.0,0.0,-0.0,-0.0,-1.0,-0.0,-0.0,-0.0,-0.0,-0.0,
        -1.9085110862529796E-5,-1.215831002246988E-8,-1.7891542245038319E-8,1.215831002246988E-8,
        1.2220370768088023E-5,1.7891542245038322E-8,0.0,0.0,1.0,0.0,0.0,0.0,0.0,-0.0,-0.0,-1.0,-0.0,-0.0,-0.0,-0.0,
        -0.0,-1.7891460877206123E-8,-1.0694098357650832E-5,1.6798000806374784E-5,1.4858518965579076E-8,
        1.908511086260566E-5,0.0,0.0,1.0,0.0,0.0,0.0,0.0,-0.0,-0.0,-1.0,-0.0,-0.0,-0.0,-0.0,-0.0,
        1.0694098357659397E-5,1.2158312102019977E-8,-0.00045000707548754654,-3.4829095211474026E-7,
        -0.00046403965892620019,0.0,0.0,1.0,0.0,0.0,0.0,0.0,0.0,-0.0,-0.0,-1.0,-0.0,-0.0,-0.0,-0.0,-0.0,
        0.00046403965892872562,4.5837370187707789E-6,-1.2158326735673334E-8,-1.7891571051804073E-8,
        1.2158326735673334E-8,1.7891571051804076E-8,0.0,0.0,1.0,0.0,0.0,0.0,0.0,0.0,0.0,-0.0,-0.0,-1.0,-0.0,-0.0,
        -0.0,-0.0,1.0694098357659397E-5,-0.0,4.583736786695908E-6,-1.2158325239203021E-8,-0.00050612620476577636,
        3.482914704367846E-7,0.0,0.0,1.0,0.0,0.0,0.0,0.0,0.0,-0.0,-0.0,-1.0,-0.0,-0.0,-0.0,-0.0,
        1.0694098357650832E-5,-1.7891545726468567E-8,-0.00045000707548770532,-0.00046403965892636103,
        1.4858575560277749E-8,0.0,0.0,1.0,0.0,0.0,0.0,0.0,-0.0,-0.0,-1.0,-0.0,-0.0,-0.0,-0.0,-0.0,
        7.4296346241351735E-9,3.4828901926211455E-7,-1.0694098357670986E-5,-1.9085110862637885E-5,
        -2.2396290183101041E-7,1.0694098357670986E-5,1.9085110862637885E-5,0.0,0.0,1.0,0.0,0.0,0.0,0.0,0.0,-0.0,
        -0.0,-1.0,-0.0,-0.0,-0.0,1.2158312102019979E-8,0.00045000707548754654,-0.0,7.4296576972040107E-9,
        -1.0694098357671877E-5,0.0,0.0,1.0,0.0,0.0,0.0,0.0,0.0,0.0,-0.0,-0.0,-1.0,-0.0,-0.0,-0.0,-0.0,
        1.215831002246988E-8,-1.90851108626193E-5,-3.4829087181474928E-7,-3.1720415380863539E-7,
        1.222037076815406E-5,0.0,0.0,1.0,0.0,0.0,0.0,0.0,-0.0,-0.0,-1.0,-0.0,-0.0,-0.0,-0.0,-0.0,
        0.00050612623031172149,2.2396533833596886E-7,-4.5837370188029509E-6,-7.4296618647694421E-9,0.0,0.0,1.0,0.0,
        0.0,0.0,0.0,0.0,-0.0,-1.0,-0.0,-0.0,-0.0,-0.0,-0.0,-1.0694098357659397E-5,-1.2158312102019977E-8,
        3.4829095211474026E-7,0.00046403965892620046,3.1720423133770447E-7,0.0,0.0,1.0,0.0,0.0,0.0,0.0,0.0,-0.0,
        -0.0,-1.0,-0.0,-0.0,-0.0,-0.0,-0.0,-4.5837367866660932E-6,-0.00045000707549025721,-1.2158325239203022E-8,
        0.000506126204767691,0.0,0.0,1.0,0.0,0.0,0.0,-0.0,-0.0,-1.0,-0.0,-0.0,-0.0,-0.0,-0.0,-0.0,
        -1.0694098357650832E-5,-1.7891545726468567E-8,0.00045000707548770532,1.4858575560277749E-8,
        0.0004640396589263613,0.0,0.0,1.0,0.0,0.0,0.0,0.0,-0.0,-0.0,-1.0,-0.0,-0.0,-0.0,-0.0,-0.0,
        -7.4296567080780895E-9,-0.0,-1.215831002246988E-8,-1.90851108626193E-5,1.222037076815406E-5,0.0,0.0,1.0,0.0,
        0.0,0.0,0.0,-0.0,-0.0,-1.0,-0.0,-0.0,-0.0,-0.0,-0.0,-9.2877109939620273E-9,-1.0694098357668958E-5,
        -1.9085110862634669E-5,1.0694098357668958E-5,4.1047291851531906E-7,1.9085110862634669E-5,0.0,0.0,1.0,0.0,
        0.0,0.0,0.0,0.0,-0.0,-0.0,-1.0,-0.0,-0.0,-0.0,-0.0,-0.0,-0.00050612623031389846,-1.2158321115834916E-8,
        -1.7891561399347412E-8,4.58373701877078E-6,1.2158321115834916E-8,1.7891561399347416E-8,0.0,0.0,1.0,0.0,0.0,
        0.0,0.0,0.0,-0.0,-0.0,-1.0,-0.0,-0.0,-0.0,-0.0,-0.0,-1.9085110862605657E-5,-1.7891542245038322E-8,
        1.2220370768144006E-5,1.4858573017288605E-8,0.0,0.0,1.0,0.0,0.0,0.0,-0.0,-0.0,-1.0,-0.0,-0.0,-0.0,-0.0,-0.0,
        -1.4858518965579084E-8,-1.0694098357663917E-5,-1.9085110862626572E-5,1.0694098357663917E-5,
        7.42963472685374E-9,1.9085110862626572E-5,0.0,0.0,1.0,0.0,0.0,0.0,0.0,-0.0,-0.0,-1.0,-0.0,-0.0,-0.0,-0.0,
        -0.0,4.583736786695908E-6,1.2158325239203021E-8,0.00045000707548754654,-3.4829147043678449E-7,
        -0.00050612620476577636,0.0,0.0,1.0,0.0,0.0,0.0,3.482914704367846E-7,1.0694098357671877E-5,
        7.4296576972040074E-9,-0.00045000707548677323,0.0,0.0,1.0,0.0,0.0,0.0,0.0,0.0,0.0,-0.0,-0.0,-1.0,-0.0,-0.0,
        -0.0,-0.0,0.00046403965892636114,4.5837370187959315E-6,-1.7891571051804073E-8,1.4858592273877606E-8,0.0,0.0,
        1.0,0.0,0.0,0.0,0.0,0.0,-0.0,-0.0,-1.0,-0.0,-0.0,-0.0,-0.0,1.0694098357671877E-5,-7.42965769720401E-9,
        -4.1047477613646406E-7,-0.00045000707548677323,-0.000464039658925489,0.0,0.0,1.0,0.0,0.0,0.0,0.0,-0.0,-0.0,
        -1.0,-0.0,-0.0,-0.0,-0.0,-0.0,-0.0,1.0694098357663919E-5,-1.4858575560277748E-8,-0.00045000707548710468,
        -0.00046403965892580158,7.4296576972040115E-9,0.0,0.0,1.0,0.0,0.0,0.0,0.0,-0.0,-0.0,-1.0,-0.0,-0.0,-0.0,
        -0.0,-0.0,1.6881176041613733E-8,-1.0694098357663022E-5,-7.4296346241351752E-9,-1.9085110862625132E-5,
        -2.2396285275354031E-7,1.0694098357663022E-5,1.9085110862625132E-5,0.0,0.0,1.0,0.0,0.0,0.0,0.0,-0.0,-0.0,
        -0.0,-0.0,-0.0,7.4296347268537432E-9,1.0146044686053521E-11,-1.0694098357671876E-5,-1.9085110862639325E-5,
        1.0694098357671876E-5,1.9085110862639325E-5,0.0,0.0,1.0,0.0,0.0,0.0,0.0,0.0,0.0,-0.0,-0.0,-1.0,-0.0,-0.0,
        -0.0,-0.0,7.4296566053585975E-9,3.4829087181474923E-7,-1.9085110862637885E-5,-2.239649158778049E-7,
        1.2220370768167794E-5,0.0,0.0,1.0,0.0,0.0,0.0,0.0,-0.0,-0.0,-1.0,-0.0,-0.0,-0.0,1.2158323877361851E-8,
        -6.4936804962317056E-6,-0.00046403965892620024,-3.482914154565164E-7,0.00042193634306069019,0.0,1.0,0.0,0.0,
        0.0,-0.0,-0.0,1.2158321115834916E-8,-0.0005061262303119843,-3.4829130899681562E-7,-3.1720459958052633E-7,
        4.5837370188005953E-6,0.0,0.0,1.0,0.0,0.0,0.0,0.0,0.0,-0.0,-0.0,-1.0,-0.0,-0.0,-0.0,-0.0,-0.0,
        1.6798000806393893E-5,2.2396527347813675E-7,-4.583736786698261E-6,-7.4296611608032738E-9,
        -0.0005061262303117203,0.0,0.0,1.0,0.0,0.0,0.0,0.0,-0.0,-0.0,-1.0,-0.0,-0.0,-0.0,-0.0,1.6881265332338726E-8,
        0.00050612623031177472,-4.5837370188024867E-6,-7.4296617620497334E-9,-2.2396533833596886E-7,0.0,0.0,1.0,0.0,
        0.0,0.0,0.0,-0.0,-0.0,-1.0,-0.0,-0.0,-0.0,-0.0,4.5837370188029534E-6,2.2927176733783571E-8,
        1.0146164063978877E-11,-7.4296644998485515E-9,0.0,0.0,1.0,0.0,0.0,0.0,0.0,0.0,0.0,-0.0,-1.0,-0.0,-0.0,-0.0,
        -0.0,-0.0,-6.4936804962317056E-6,-1.2158323877361849E-8,-0.0004640396589262003,0.00042193634306069067,
        3.4829141545651656E-7,0.0,0.0,1.0,0.0,0.0,0.0,0.0,-0.0,-0.0,-1.0,-0.0,-0.0,-0.0,-0.0,-0.0,
        -1.0694098357668962E-5,-9.2877423739426452E-9,-3.1720423133770447E-7,4.1047477613646422E-7,
        0.00046403965892562475,0.0,0.0,1.0,0.0,0.0,0.0,0.0,-0.0,-0.0,-1.0,-0.0,-0.0,-0.0,-0.0,
        -1.6798000806305527E-5,-1.2158319619365041E-8,1.2158319619365041E-8,0.00050612623031389889,
        1.7891558818155705E-8,0.0,0.0,1.0,0.0,0.0,0.0,0.0,0.0,-0.0,-0.0,-1.0,-0.0,-0.0,-0.0,-0.0,-0.0,
        -7.4296644998485515E-9,-0.0,-4.5837370188005944E-6,-1.2158326735673331E-8,0.0,0.0,1.0,0.0,0.0,0.0,0.0,-0.0,
        -0.0,-1.0,-0.0,-0.0,-0.0,-0.0,-0.0,-0.0,-1.0694098357663919E-5,-1.4858575560277748E-8,7.4296576972040115E-9,
        0.00045000707548710468,0.00046403965892580185,0.0,0.0,1.0,0.0,0.0,0.0,0.0,-0.0,-0.0,-1.0,-0.0,-0.0,-0.0,
        -0.0,-0.0,-6.4936804962256934E-6,-1.7891566095252494E-8,9.28774984743106E-9,0.00042193634306084149,
        1.4858589000533567E-8,0.0,0.0,1.0,0.0,0.0,0.0,0.0,-0.0,-0.0,-1.0,-0.0,-0.0,-0.0,-0.0,-0.0,
        -1.9085110862626568E-5,-2.2396486680039542E-7,7.4296567080780895E-9,1.2220370768159488E-5,0.0,0.0,1.0,0.0,
        0.0,0.0,0.0,-0.0,-0.0,-1.0,-0.0,-0.0,-0.0,-0.0,-0.0,-7.4296347268537432E-9,-3.7178292219660892E-11,
        -1.0694098357671876E-5,-1.9085110862639325E-5,1.0694098357671876E-5,1.9085110862639325E-5,0.0,0.0,1.0,0.0,
        0.0,0.0,0.0,-0.0,-0.0,-1.0,-0.0,-0.0,-0.0,-0.0,-0.0,-0.0,-7.4296566053585975E-9,-1.9085110862637885E-5,
        1.2220370768167794E-5,2.2396491587780615E-7,0.0,0.0,1.0,0.0,0.0,0.0,0.0,-0.0,-0.0,-1.0,-0.0,-0.0,-0.0,-0.0,
        -0.0,-7.4296618647694413E-9,-3.7178490738895427E-11,-2.2927174412894674E-8,4.58373701880722E-6,0.0,0.0,1.0,
        0.0,0.0,0.0,0.0,-0.0,-0.0,-1.0,-0.0,-0.0,-0.0,-0.0,-0.0,-0.0,-1.2158321115834916E-8,-0.0005061262303119843,
        4.5837370188005953E-6,3.4829130899681562E-7,0.0,0.0,1.0,0.0,0.0,0.0,0.0,0.0,-0.0,-0.0,-1.0,-0.0,-0.0,-0.0,
        -0.0,-0.0,-4.5837370187707789E-6,-0.00050612620476769106,-1.2158326735673334E-8,-1.7891571051804073E-8,
        1.2158326735673334E-8,1.7891571051804076E-8,0.0,0.0,1.0,0.0,0.0,0.0,0.0,-0.0,-0.0,-1.0,-0.0,-0.0,-0.0,-0.0,
        -0.0,-0.0,1.9085110862626568E-5,-1.4858573017288606E-8,-6.4936804962348371E-6,-1.2220370768159488E-5,
        7.429656708078092E-9,0.0,0.0,1.0,0.0,0.0,0.0,0.0,-0.0,-0.0,-1.0,-0.0,-0.0,-0.0,-0.0,1.2158319619365039E-8,
        1.6798000806387232E-5,-4.5837367866959046E-6,-3.4829125063572129E-7,-0.00050612623031198246,0.0,0.0,1.0,0.0,
        0.0,0.0,1.2158326735673331E-8,-0.0,4.5837370188072216E-6,7.4296644998485515E-9,0.0,0.0,1.0,0.0,0.0,0.0,0.0,
        0.0,0.0,0.0,-0.0,-1.0,-0.0,-0.0,-0.0,-0.0,1.0694098357663024E-5,1.688125147749625E-8,-7.4296575944844856E-9,
        -0.00045000707548718789,-2.2396493601855318E-7,0.0,0.0,1.0,0.0,0.0,0.0,0.0,-0.0,-0.0,-0.0,-0.0,
        1.2220370768088018E-5,-4.58373701877078E-6,-1.2158321115834916E-8,-1.7891561399347412E-8,
        1.2158321115834916E-8,1.7891561399347416E-8,0.0,0.0,1.0,0.0,0.0,0.0,0.0,0.0,-0.0,-0.0,-1.0,-0.0,-0.0,-0.0,
        -0.0,4.5837370188005944E-6,2.2927176733777311E-8,-1.2158326735673331E-8,3.48291528797896E-7,
        3.1720482258753326E-7,0.0,0.0,1.0,0.0,0.0,0.0,0.0,0.0,0.0,-0.0,-1.0,-0.0,-0.0,-0.0,-0.0,-0.0,-0.0,
        1.9085110862605657E-5,-1.7891542245038322E-8,-6.4936804962256925E-6,-1.2220370768144006E-5,
        1.4858573017288605E-8,0.0,0.0,1.0,0.0,0.0,0.0,0.0,-0.0,-0.0,-1.0,-0.0,-0.0,-0.0,-0.0,6.4936804962348362E-6,
        0.00046403965892580164,-1.4858589000533565E-8,-0.00042193634306016711,7.4296631806500488E-9,0.0,0.0,1.0,0.0,
        0.0,0.0,0.0,-0.0,-0.0,-1.0,-0.0,-0.0,-0.0,-0.0,1.6798000806387232E-5,-1.2158319619365039E-8,
        -4.5837367866959046E-6,-0.00050612623031198365,3.4829125063572129E-7,0.0,0.0,1.0,0.0,0.0,0.0,0.0,-0.0,-0.0,
        -1.0,-0.0,-0.0,-0.0,-0.0,1.0694098357668962E-5,-9.2877423739426452E-9,-3.1720423133770447E-7,
        -0.00045000707548691982,4.1047477613646422E-7,0.0,0.0,1.0,0.0,0.0,0.0,-0.0,-0.0,-0.0,-0.0,-0.0,
        4.5837370188072216E-6,-7.4296644998485515E-9,0.0,0.0,1.0,0.0,0.0,0.0,0.0,0.0,-0.0,-0.0,-1.0,-0.0,-0.0,-0.0,
        -0.0,-0.0,2.2396285275353962E-7,-1.0694098357663917E-5,-7.4296347268537432E-9,-1.9085110862626572E-5,
        1.0694098357663917E-5,1.9085110862626572E-5,0.0,0.0,1.0,0.0,0.0,0.0,0.0,0.0,-0.0,-0.0,-1.0,-0.0,-0.0,-0.0,
        -0.0,-0.0,1.688125147749625E-8,-1.0694098357663024E-5,-7.4296575944844856E-9,-2.2396493601855318E-7,
        0.000464039658925878,0.0,0.0,1.0,0.0,0.0,0.0,0.0,-0.0,-0.0,-1.0,-0.0,-0.0,-0.0,-0.0,1.688127393370768E-8,
        -4.5837370188024859E-6,-0.00042193634306026285,-7.4296643971287352E-9,-2.2396557095858857E-7,0.0,0.0,1.0,
        0.0,0.0,0.0,-0.0,-0.0,-0.0,-0.0,-0.0,7.4296567080780878E-9,1.0146135927197276E-11,-6.3682160827337868E-8,
        1.2220370768168861E-5,0.0,0.0,1.0,0.0,0.0,0.0,0.0,0.0,-0.0,-0.0,-1.0,-0.0,-0.0,-0.0,-0.0,
        7.4296630779302881E-9,3.4829141545651646E-7,-6.493680496239771E-6,-0.00046403965892556534,
        -2.2396549593349934E-7,0.00042193634305989894,0.0,1.0,0.0,0.0,0.0,0.0,-0.0,-0.0,-1.0,-0.0,-0.0,-0.0,-0.0,
        1.6881248308706442E-8,-1.9085110862625125E-5,-7.4296566053585983E-9,-2.2396486680039341E-7,
        1.2220370768158434E-5,0.0,0.0,1.0,0.0,0.0,0.0,-0.0,-0.0,-0.0,-0.0,7.4296617620497334E-9,
        3.4829130899681573E-7,-0.00050612623031152687,-2.2396538741336503E-7,4.5837370188067541E-6,0.0,0.0,1.0,0.0,
        0.0,0.0,0.0,0.0,-0.0,-0.0,-1.0,-0.0,-0.0,-0.0,1.2158326735673331E-8,-4.5837370188005944E-6,
        -3.8211718654778936E-8,-3.4829152879789592E-7,-3.1720482258753289E-7,0.0,0.0,1.0,0.0,0.0,0.0,0.0,-0.0,-0.0,
        -1.0,-0.0,-0.0,-0.0,-0.0,-0.0,-0.0,1.6798000806392572E-5,1.6881263044223225E-8,-4.5837367866978011E-6,
        -7.4296610580835949E-9,-0.00050612623031177516,-2.2396527347813746E-7,0.0,0.0,1.0,0.0,0.0,0.0,-0.0,-0.0,
        -1.0,-0.0,-0.0,-0.0,7.4296611608032722E-9,1.6798000806405521E-5,2.2396532255553607E-7,
        -4.5837367867025318E-6,-0.000506126230311472,0.0,0.0,1.0,0.0,0.0,0.0,0.0,0.0,-0.0,-0.0,-1.0,-0.0,-0.0,-0.0,
        0.00050612623031198343,-1.2158321115834914E-8,-4.5837370188005944E-6,3.4829130899681573E-7,
        3.1720459958052686E-7,0.0,0.0,1.0,0.0,0.0,0.0,0.0,0.0,-0.0,-1.0,-0.0,-0.0,-0.0,-0.0,-0.0,
        4.5837370188024867E-6,1.688127393370768E-8,0.00050612620476556743,-7.4296643971287319E-9,
        -2.2396557095858762E-7,0.0,0.0,1.0,0.0,0.0,0.0,0.0,0.0,-0.0,-1.0,-0.0,-0.0,-0.0,-0.0,2.2396493601855255E-7,
        -1.0694098357663915E-5,-7.4296576972040082E-9,0.000464039658925802,0.0,0.0,1.0,0.0,0.0,0.0,0.0,0.0,-0.0,
        -0.0,-1.0,-0.0,-0.0,-0.0,-0.0,-0.0,4.5837367866982678E-6,-0.00050612620476551441,1.0694098357663919E-5,
        2.2396493601855321E-7,-7.4296576972040082E-9,0.0,0.0,1.0,0.0,0.0,0.0,0.0,0.0,-0.0,-0.0,-1.0,-0.0,-0.0,-0.0,
        -0.0,-0.0,-6.4936804962403843E-6,0.0,7.4296644998485506E-9,-4.5837370188072174E-6,0.0,0.0,1.0,0.0,0.0,0.0,
        0.0,0.0,-0.0,-0.0,-1.0,-0.0,-0.0,-0.0,-0.0,-0.0,-1.0694098357671877E-5,-7.42965769720401E-9,
        -4.1047477613646406E-7,0.00045000707548677323,0.00046403965892548928,0.0,0.0,1.0,0.0,0.0,0.0,0.0,-0.0,-0.0,
        -1.0,-0.0,-0.0,-0.0,-0.0,-0.0,-0.0,-4.5837370188029534E-6,-3.821171865479442E-8,-1.0146164063978909E-11,
        7.4296644998485515E-9,0.0,0.0,1.0,0.0,0.0,0.0,0.0,-0.0,-0.0,-1.0,-0.0,-0.0,-0.0,-0.0,-0.0,-0.0,
        -6.4936804962383413E-6,-9.28774984743106E-9,-3.1720470655542463E-7,0.00042193634305996963,
        4.1047521572237433E-7,0.0,0.0,1.0,0.0,0.0,0.0,0.0,-0.0,-0.0,-1.0,-0.0,-0.0,-0.0,-0.0,-0.0,
        -1.6881248308706442E-8,-1.9085110862625125E-5,7.4296566053585983E-9,0.0,0.0,1.0,0.0,0.0,0.0,0.0,-0.0,-0.0,
        -1.0,-0.0,-0.0,-0.0,-0.0,-0.0,-0.0,6.3682160827337868E-8,-7.4296567080780911E-9,-6.4936804962403843E-6,
        -1.2220370768168856E-5,0.0,0.0,1.0,0.0,0.0,0.0,0.0,-0.0,-0.0,-1.0,-0.0,-0.0,-0.0,-0.0,-0.0,
        -0.00050612623031172257,-2.2396533833597008E-7,4.5837370188029509E-6,7.4296618647694454E-9,0.0,0.0,1.0,0.0,
        0.0,0.0,0.0,0.0,-0.0,-0.0,-1.0,-0.0,-0.0,-0.0,-0.0,-0.0,1.2220370768159481E-5,-1.4858585776305598E-8,
        -4.5837370188029509E-6,7.4296618647694413E-9,0.0,0.0,1.0,0.0,0.0,0.0,0.0,-0.0,-0.0,-1.0,-0.0,-0.0,-0.0,-0.0,
        1.2158321115834916E-8,0.00050612623031198322,-4.5837370188005953E-6,-3.4829130899681562E-7,0.0,0.0,1.0,0.0,
        0.0,0.0,0.0,0.0,-0.0,-0.0,-1.0,-0.0,-0.0,-0.0,-0.0,-0.0,4.5837367867025351E-6,7.4296637958821772E-9,
        6.113889073992857E-8,1.0146164889050167E-11,-2.292717440851893E-6,0.0,0.0,1.0,0.0,0.0,0.0,0.0,0.0,0.0,-0.0,
        -0.0,-1.0,-0.0,-0.0,-0.0,1.2220370768144007E-5,-1.7891561399347416E-8,-4.5837370187959307E-6,
        1.4858585776305595E-8,0.0,0.0,1.0,0.0,0.0,0.0,0.0,-0.0,-0.0,-1.0,-0.0,-0.0,-0.0,-0.0,4.5837370188056546E-6,
        2.2927176733790933E-8,-9.2877516553713879E-9,1.8589253148948242E-9,0.0,0.0,1.0,0.0,0.0,0.0,0.0,0.0,0.0,-0.0,
        -1.0,-0.0,-0.0,-0.0,-0.0,-0.0,-0.0,4.5837370188029534E-6,3.821171865479442E-8,-7.433024541721736E-11,
        7.4296644998485481E-9,0.0,0.0,1.0,0.0,0.0,0.0,0.0,0.0,-0.0,-0.0,-1.0,-0.0,-0.0,-0.0,-0.0,
        4.5837367867009707E-6,0.00045000707548692004,-9.2877507019112439E-9,-0.00050612620476536555,
        4.104752685697449E-7,0.0,0.0,1.0,0.0,0.0,0.0,0.0,0.0,-0.0,-0.0,-1.0,-0.0,-0.0,-0.0,-0.0,
        1.6881265332338726E-8,-0.00050612623031177624,-7.4296617620497334E-9,-2.2396533833596814E-7,
        4.58373701880249E-6,0.0,0.0,1.0,0.0,0.0,0.0,0.0,-0.0,-0.0,-0.0,-0.0,1.6881269537940858E-8,
        -6.4936804962342221E-6,-0.000464039658925878,-7.4296630779302831E-9,-2.2396544685610481E-7,
        0.00042193634306026236,0.0,1.0,0.0,0.0,0.0,-0.0,-0.0,-1.0,-0.0,-0.0,-0.0,-0.0,7.4296643971287361E-9,
        4.7324675836111347E-11,-4.5837370188067558E-6,-3.8211718654817105E-8,-1.0146166798111696E-9,0.0,0.0,1.0,0.0,
        0.0,0.0,0.0,-0.0,-0.0,-1.0,-0.0,-0.0,-0.0,-0.0,1.0146164063978886E-11,-4.5837370188029492E-6,
        -3.8211718654794447E-8,-7.4296644998485515E-9,0.0,0.0,1.0,0.0,0.0,0.0,0.0,-0.0,-0.0,-1.0,-0.0,-0.0,-0.0,
        -0.0,-0.0,-0.0,2.239648668003942E-7,-1.9085110862626568E-5,-7.4296567080780895E-9,1.2220370768159488E-5,0.0,
        0.0,1.0,0.0,0.0,0.0,0.0,-0.0,-0.0,-1.0,-0.0,-0.0,-0.0,-0.0,-0.0,7.4296618647694421E-9,
        1.0146157288894191E-11,-2.2927174412894667E-8,4.5837370188072208E-6,0.0,0.0,1.0,0.0,0.0,0.0,0.0,0.0,0.0,
        -0.0,-0.0,-1.0,-0.0,-0.0,-0.0,-0.0,7.4296618647694413E-9,2.2927174412894674E-8,1.014615728889418E-11,
        -4.58373701880722E-6,0.0,0.0,1.0,0.0,0.0,0.0,0.0,0.0,0.0,-0.0,-1.0,-0.0,-0.0,-0.0,-0.0,
        0.00050612623031157176,-9.28774805426214E-9,-4.5837370188056563E-6,4.1047511029324503E-7,0.0,0.0,1.0,0.0,
        0.0,0.0,0.0,0.0,-0.0,-1.0,-0.0,-0.0,-0.0,-0.0,-0.0,-0.0,2.239654468561051E-7,-6.4936804962348328E-6,
        -7.4296631806500431E-9,0.00042193634306016646,0.0,0.0,1.0,0.0,0.0,0.0,0.0,0.0,-0.0,-0.0,-1.0,-0.0,-0.0,-0.0,
        -0.0,-0.0,6.11325085205292E-8,-7.4296618647694372E-9,-3.7178490738895453E-11,-4.58373701880722E-6,0.0,0.0,
        1.0,0.0,0.0,0.0,0.0,-0.0,-0.0,-1.0,-0.0,-0.0,-0.0,-0.0,-0.0,7.4296617620497334E-9,3.4829130899681578E-7,
        0.00050612623031152644,-4.5837370188067532E-6,-2.2396538741336503E-7,0.0,0.0,1.0,0.0,0.0,0.0,0.0,0.0,-0.0,
        -1.0,-0.0,-0.0,-0.0,-0.0,1.6798000806401259E-5,-9.2877471008022732E-9,-4.5837367867009664E-6,
        -0.00050612623031157425,4.1047505518161023E-7,0.0,0.0,1.0,0.0,0.0,0.0,0.0,-0.0,-0.0,-1.0,-0.0,-0.0,-0.0,
        -0.0,2.2396533833596926E-7,-0.00050612623031172279,-7.4296618647694454E-9,4.5837370188029509E-6,0.0,0.0,1.0,
        0.0,0.0,0.0,0.0,0.0,-0.0,-0.0,-1.0,-0.0,-0.0,-0.0,-0.0,-0.0,-4.1765326688254592E-8,-1.9820056068025643E-5,
        -6.1465931801342287E-8,-3.536830828564795E-5,4.1765326688254592E-8,1.9820056068025643E-5,
        6.1465931801342287E-8,3.536830828564795E-5,0.0,0.0,0.0,1.0,0.0,0.0,0.0,0.0,-0.0,-0.0,-0.0,-1.0,-0.0,-0.0,
        -0.0,-0.0,4.1765326688254592E-8,-1.9820056068217665E-5,-1.1968732734248517E-6,-1.0900855640273811E-6,
        -3.5368308285978367E-5,1.9820056068217665E-5,3.5368308285978367E-5,0.0,0.0,0.0,1.0,0.0,0.0,0.0,0.0,-0.0,
        -0.0,-0.0,-1.0,-0.0,-0.0,-0.0,-0.0,1.9820056068025643E-5,-4.1765417905831474E-8,-0.00083380391301686875,
        -6.1466078468218222E-8,-0.00085976636245109277,4.1765417905831474E-8,6.1466078468218222E-8,0.0,0.0,0.0,1.0,
        0.0,0.0,0.0,0.0,-0.0,-0.0,-0.0,-1.0,-0.0,-0.0,-0.0,-0.0,6.1465931801342287E-8,-3.1901445693811346E-8,
        -1.98200560681773E-5,-5.1041750564472194E-8,3.5368308285909229E-5,0.0,0.0,0.0,1.0,0.0,0.0,0.0,-0.0,-0.0,
        -0.0,-1.0,-0.0,-0.0,-0.0,-0.0,-4.1765326688254592E-8,-1.9820056068217665E-5,-3.5368308285978367E-5,
        1.9820056068217665E-5,1.1968732734248517E-6,1.0900855640273817E-6,3.5368308285978367E-5,0.0,0.0,0.0,1.0,0.0,
        0.0,0.0,0.0,-0.0,-0.0,-0.0,-1.0,-0.0,-0.0,-0.0,-0.0,-1.9820056068025643E-5,-4.1765417905831474E-8,
        -6.1466078468218222E-8,4.1765417905831474E-8,0.0008338039130168682,6.1466078468218222E-8,
        0.00085976636245109321,0.0,0.0,0.0,1.0,0.0,0.0,0.0,0.0,-0.0,-0.0,-0.0,-1.0,-0.0,-0.0,-0.0,-0.0,
        -6.1465931801342287E-8,-1.98200560681773E-5,-3.5368308285909229E-5,1.98200560681773E-5,
        5.1041750564472194E-8,3.5368308285909229E-5,0.0,0.0,0.0,1.0,0.0,0.0,0.0,-0.0,-0.0,-0.0,-1.0,-0.0,-0.0,-0.0,
        -0.0,-3.5368308285647957E-5,-4.1765420350690029E-8,5.7993732762902535E-8,2.2650033355952723E-5,
        6.1466082591352316E-8,0.0,0.0,0.0,1.0,0.0,0.0,0.0,-0.0,-0.0,-0.0,-1.0,-0.0,-0.0,-0.0,-0.0,
        4.1765417905831474E-8,1.9820056068217662E-5,-1.196876410390218E-6,-0.00083380391301358513,
        -1.0900886312173043E-6,0.0,0.0,0.0,1.0,0.0,0.0,0.0,0.0,-0.0,-0.0,-0.0,-1.0,-0.0,-0.0,-0.0,-0.0,
        1.0900855640273813E-6,2.5517427762228991E-8,-1.982005606825484E-5,-3.5368308286042586E-5,
        1.982005606825484E-5,3.5368308286042586E-5,0.0,0.0,0.0,1.0,0.0,0.0,0.0,0.0,0.0,-0.0,-0.0,-0.0,-1.0,-0.0,
        -0.0,-0.0,4.1765417905831474E-8,-0.0,2.5517476036470872E-8,-1.9820056068252563E-5,-7.698100353892288E-7,
        0.00083380391301294166,0.0,0.0,0.0,1.0,0.0,0.0,0.0,0.0,-0.0,-0.0,-0.0,-1.0,-0.0,-0.0,-0.0,
        4.1765420350690029E-8,-3.536830828597836E-5,-1.1968765081235836E-6,-1.0900887240413872E-6,
        2.2650033356173453E-5,0.0,0.0,0.0,1.0,0.0,0.0,0.0,-0.0,-0.0,-0.0,-1.0,-0.0,-0.0,-0.0,-0.0,
        8.4971497353658268E-6,0.00083380391301686864,-4.176544570866186E-8,-6.1466123204832153E-8,
        -0.00093763620100816871,4.176544570866186E-8,6.1466123204832153E-8,0.0,0.0,0.0,1.0,0.0,0.0,0.0,0.0,-0.0,
        -0.0,-0.0,-0.0,-0.0,-0.0,1.9820056068217665E-5,1.1968764103902187E-6,-0.0,8.49715016563479E-6,
        -4.1765449454567667E-8,0.0,0.0,0.0,1.0,0.0,0.0,0.0,0.0,0.0,-0.0,-0.0,-0.0,-1.0,-0.0,-0.0,-0.0,
        1.9820056068177296E-5,-6.1466078468218208E-8,-0.000833803913014142,-0.00085976636244831472,
        5.1041858488805809E-8,0.0,0.0,0.0,1.0,0.0,0.0,0.0,-0.0,-0.0,-0.0,-1.0,-0.0,-0.0,-0.0,-0.0,
        7.6981056413003323E-7,0.00093763624831117744,-2.5517488218346108E-8,-8.497150165637417E-6,0.0,0.0,0.0,1.0,
        0.0,0.0,0.0,0.0,-0.0,-0.0,-1.0,-0.0,-0.0,-0.0,-0.0,-4.1765417905831474E-8,-1.9820056068217662E-5,
        0.00083380391301358459,1.0900886312173049E-6,0.00085976636244771917,0.0,0.0,0.0,1.0,0.0,0.0,0.0,0.0,-0.0,
        -0.0,-0.0,-1.0,-0.0,-0.0,-0.0,-0.0,-2.55174274093182E-8,-1.1968732734248508E-6,-1.9820056068252566E-5,
        7.6980717747168429E-7,0.0,0.0,0.0,1.0,0.0,0.0,-0.0,-0.0,-0.0,-1.0,-0.0,-0.0,-0.0,-0.0,-0.0,
        -4.1765420350690029E-8,-3.536830828597836E-5,1.1968765081235836E-6,2.2650033356173453E-5,
        1.0900887240413878E-6,0.0,0.0,0.0,1.0,0.0,0.0,0.0,-0.0,-0.0,-0.0,-1.0,-0.0,-0.0,-0.0,-0.0,
        -8.497150165615882E-6,-0.0,-1.9820056068177296E-5,-6.1466078468218208E-8,5.1041858488805809E-8,0.0,0.0,0.0,
        1.0,0.0,0.0,0.0,-0.0,-0.0,-0.0,-1.0,-0.0,-0.0,-0.0,-0.0,-1.2036826344670679E-5,-4.1765443887723989E-8,
        -6.1466120370748321E-8,4.1765443887723989E-8,0.00078187032238078932,6.1466120370748321E-8,0.0,0.0,0.0,1.0,
        0.0,0.0,0.0,0.0,-0.0,-0.0,-0.0,-1.0,-0.0,-0.0,-0.0,-0.0,-7.6980700903258931E-7,-1.9820056068223588E-5,
        -3.5368308285989006E-5,2.5517427762228988E-8,1.9820056068223588E-5,3.5368308285989006E-5,0.0,0.0,0.0,1.0,
        0.0,0.0,0.0,0.0,-0.0,-0.0,-0.0,-1.0,-0.0,-0.0,-0.0,-0.0,-6.14660825913523E-8,-3.5368308285909229E-5,
        5.10418615532681E-8,2.2650033356126544E-5,0.0,0.0,0.0,1.0,0.0,0.0,-0.0,-0.0,-0.0,-1.0,-0.0,-0.0,-0.0,-0.0,
        -2.2650033355952723E-5,-4.17654403338918E-8,-6.1466114631994E-8,4.17654403338918E-8,8.4971501655451073E-6,
        6.1466114631994E-8,0.0,0.0,0.0,1.0,0.0,0.0,0.0,-0.0,-0.0,-0.0,-1.0,-0.0,-0.0,-0.0,-0.0,
        2.5517476036470879E-8,1.9820056068252563E-5,1.1968764103902182E-6,-0.0008338039130129422,
        -7.698100353892288E-7,0.0,0.0,0.0,1.0,0.0,0.0,0.00083380391301294231,4.1765449454567667E-8,
        8.4971501656347844E-6,-1.19687750304504E-6,0.0,0.0,0.0,1.0,0.0,0.0,0.0,0.0,0.0,-0.0,-0.0,-0.0,-1.0,-0.0,
        -0.0,-0.0,1.0900887240413874E-6,2.5517477507231932E-8,-3.5368308286042579E-5,2.2650033356215906E-5,0.0,0.0,
        0.0,1.0,0.0,0.0,0.0,0.0,-0.0,-0.0,-0.0,-1.0,-0.0,-0.0,-0.0,4.1765449454567667E-8,-8.4971501656347912E-6,
        -0.00078187032237773848,-1.19687750304504E-6,-1.0900896970047281E-6,0.0,0.0,0.0,1.0,0.0,0.0,0.0,-0.0,-0.0,
        -0.0,-1.0,-0.0,-0.0,-0.0,-0.0,-0.0,4.1765440333891803E-8,-2.2650033356173436E-5,-1.1968771910546153E-6,
        -1.0900893910065394E-6,8.4971501656347962E-6,0.0,0.0,0.0,1.0,0.0,0.0,0.0,-0.0,-0.0,-0.0,-1.0,-0.0,-0.0,-0.0,
        -0.0,3.1130989737343496E-5,-4.1765436587986837E-8,-8.4971497353658251E-6,-6.1466108552265955E-8,
        -0.0009376362483148144,4.1765436587986837E-8,6.1466108552265955E-8,0.0,0.0,0.0,1.0,0.0,0.0,0.0,-0.0,-0.0,
        -0.0,-0.0,-0.0,8.4971501655450988E-6,4.2477118830459293E-8,-4.1765449454567654E-8,-6.1466129284561547E-8,
        4.1765449454567654E-8,6.1466129284561547E-8,0.0,0.0,0.0,1.0,0.0,0.0,0.0,0.0,0.0,-0.0,-0.0,-0.0,-1.0,-0.0,
        -0.0,-0.0,8.4971497354366032E-6,0.00083380391301414187,-6.146612320483214E-8,-0.00093763620100534772,
        5.1041891498988872E-8,0.0,0.0,0.0,1.0,0.0,0.0,0.0,-0.0,-0.0,-0.0,-0.0,-0.0,-0.0,1.9820056068245295E-5,
        -3.1901509151756582E-8,-1.0900886312173043E-6,-0.00083380391301303479,1.4104940601734428E-6,0.0,0.0,1.0,0.0,
        0.0,-0.0,-0.0,1.9820056068223584E-5,-7.6980986695002329E-7,-0.00083380391301339193,-0.00085976636244754082,
        2.551747638938298E-8,0.0,0.0,0.0,1.0,0.0,0.0,0.0,0.0,-0.0,-0.0,-0.0,-1.0,-0.0,-0.0,-0.0,-0.0,
        5.7993762007698894E-8,0.00093763624831123013,-2.5517487865433698E-8,-8.49715016563634E-6,
        -7.6981056413003673E-7,0.0,0.0,0.0,1.0,0.0,0.0,0.0,-0.0,-0.0,-0.0,-1.0,-0.0,-0.0,-0.0,3.1130989737646618E-5,
        7.6981044396015579E-7,-2.5517486265542115E-8,-8.4971497354581415E-6,-0.00093763624831117646,0.0,0.0,0.0,1.0,
        0.0,0.0,0.0,-0.0,-0.0,-0.0,-1.0,-0.0,-0.0,-0.0,2.5517488218346114E-8,3.4871908529920814E-11,
        4.2477114526910954E-8,-8.497150165652074E-6,0.0,0.0,0.0,1.0,0.0,0.0,0.0,0.0,0.0,-0.0,-0.0,-1.0,-0.0,-0.0,
        -0.0,-0.0,-3.1901509151756582E-8,-1.9820056068245292E-5,-1.0900886312173045E-6,1.4104940601734428E-6,
        0.00083380391301303457,0.0,0.0,0.0,1.0,0.0,0.0,0.0,-0.0,-0.0,-0.0,-1.0,-0.0,-0.0,-0.0,-0.0,
        -4.1765443887724E-8,-1.2036826344793178E-5,-0.000859766362447719,0.00078187032237773848,
        1.0900895118641057E-6,0.0,0.0,0.0,1.0,0.0,0.0,0.0,-0.0,-0.0,-0.0,-0.0,-0.0,-0.0,-0.0,-5.799359523255268E-8,
        -1.9820056068221311E-5,1.9820056068221311E-5,7.6980700903258868E-7,3.5368308285985096E-5,0.0,0.0,0.0,1.0,
        0.0,0.0,0.0,0.0,-0.0,-0.0,-0.0,-1.0,-0.0,-0.0,-0.0,-0.0,-8.49715016565208E-6,-0.0,-2.5517476389382974E-8,
        -1.9820056068254836E-5,0.0,0.0,0.0,1.0,0.0,0.0,0.0,-0.0,-0.0,-0.0,-1.0,-0.0,-0.0,-0.0,-0.0,-0.0,
        -4.1765440333891803E-8,-2.2650033356173436E-5,8.4971501656347962E-6,1.1968771910546153E-6,
        1.09008939100654E-6,0.0,0.0,0.0,1.0,0.0,0.0,0.0,-0.0,-0.0,-0.0,-1.0,-0.0,-0.0,-0.0,-0.0,
        -3.1901510756457431E-8,-3.5368308286026065E-5,1.2036826344810729E-5,1.4104941677273269E-6,
        2.265003335620498E-5,0.0,0.0,0.0,1.0,0.0,0.0,0.0,-0.0,-0.0,-0.0,-1.0,-0.0,-0.0,-0.0,-0.0,
        -6.1466114631994E-8,-0.0009376362483119971,8.49715016561588E-6,5.1041885201670711E-8,0.0,0.0,0.0,1.0,0.0,
        0.0,0.0,-0.0,-0.0,-0.0,-1.0,-0.0,-0.0,-0.0,-0.0,-8.4971501655451073E-6,-7.0817347532925277E-8,
        -4.1765449454567654E-8,-6.1466129284561547E-8,4.1765449454567654E-8,6.1466129284561547E-8,0.0,0.0,0.0,1.0,
        0.0,0.0,0.0,-0.0,-0.0,-0.0,-1.0,-0.0,-0.0,-0.0,-0.0,-0.0,-8.4971497354366082E-6,-6.146612320483214E-8,
        5.1041891498988872E-8,0.00093763620100535141,0.0,0.0,0.0,1.0,0.0,0.0,0.0,-0.0,-0.0,-0.0,-1.0,-0.0,-0.0,-0.0,
        -0.0,-8.497150165637417E-6,-7.0817347533601024E-8,-3.4871908656977404E-11,2.5517493103151746E-8,0.0,0.0,0.0,
        1.0,0.0,0.0,0.0,-0.0,-0.0,-0.0,-1.0,-0.0,-0.0,-0.0,-0.0,-0.0,-1.9820056068223584E-5,-7.6980986695002329E-7,
        2.551747638938298E-8,0.00083380391301339138,0.0,0.0,0.0,1.0,0.0,0.0,0.0,0.0,-0.0,-0.0,-0.0,-1.0,-0.0,-0.0,
        -0.0,-0.0,-2.5517427762228991E-8,-7.698071774716863E-7,-1.982005606825484E-5,-3.5368308286042586E-5,
        1.982005606825484E-5,3.5368308286042586E-5,0.0,0.0,0.0,1.0,0.0,0.0,0.0,-0.0,-0.0,-0.0,-1.0,-0.0,-0.0,-0.0,
        -0.0,-0.0,6.1466114631994E-8,-2.2650033356126568E-5,-3.1901524703314204E-8,-5.1041885201670711E-8,
        8.49715016561588E-6,0.0,0.0,0.0,1.0,0.0,0.0,0.0,-0.0,-0.0,-0.0,-1.0,-0.0,-0.0,-0.0,1.9820056068221311E-5,
        5.7993728992459593E-8,-2.5517476036470872E-8,-0.000833803913013453,-7.698098669500217E-7,0.0,0.0,0.0,1.0,
        0.0,0.0,1.9820056068254836E-5,-0.0,2.5517493103151756E-8,8.497150165652074E-6,0.0,0.0,0.0,1.0,0.0,0.0,0.0,
        0.0,0.0,0.0,-0.0,-0.0,-1.0,-0.0,-0.0,-0.0,4.1765436587986837E-8,3.1130989737637409E-5,-8.497149735455514E-6,
        -1.196877058986831E-6,-0.00093763624831128293,0.0,0.0,0.0,1.0,0.0,0.0,0.0,-0.0,-0.0,-0.0,-0.0,
        5.1041750564472187E-8,-2.5517427762228988E-8,-1.9820056068223588E-5,-3.5368308285989006E-5,
        1.9820056068223588E-5,3.5368308285989006E-5,0.0,0.0,0.0,1.0,0.0,0.0,0.0,0.0,-0.0,-0.0,-0.0,-1.0,-0.0,-0.0,
        -0.0,2.5517476389382974E-8,3.4871876948106349E-11,-1.9820056068254836E-5,0.00083380391301288072,
        0.00085976636244701075,0.0,0.0,0.0,1.0,0.0,0.0,0.0,0.0,0.0,-0.0,-0.0,-1.0,-0.0,-0.0,-0.0,-0.0,-0.0,
        6.14660825913523E-8,-3.5368308285909229E-5,-3.1901510756457437E-8,-5.10418615532681E-8,
        2.2650033356126544E-5,0.0,0.0,0.0,1.0,0.0,0.0,0.0,-0.0,-0.0,-0.0,-1.0,-0.0,-0.0,-0.0,3.1901524703314204E-8,
        1.0900893910065396E-6,-2.2650033356204976E-5,-1.410494882596244E-6,8.4971501656476779E-6,0.0,0.0,0.0,1.0,
        0.0,0.0,0.0,-0.0,-0.0,-0.0,-1.0,-0.0,-0.0,-0.0,5.7993728992459593E-8,-1.9820056068221311E-5,
        -2.5517476036470872E-8,-7.6980986695002339E-7,0.00083380391301345242,0.0,0.0,0.0,1.0,0.0,0.0,0.0,-0.0,-0.0,
        -0.0,-1.0,-0.0,-0.0,-0.0,4.1765443887724E-8,-1.2036826344793178E-5,-0.000859766362447719,
        -1.1968773129171683E-6,0.00078187032237773848,0.0,0.0,0.0,1.0,0.0,0.0,-0.0,-0.0,-0.0,-0.0,-0.0,
        2.551749310315175E-8,-8.4971501656520791E-6,0.0,0.0,0.0,1.0,0.0,0.0,0.0,0.0,-0.0,-0.0,-0.0,-1.0,-0.0,-0.0,
        -0.0,-0.0,0.00093763624831481461,-4.17654403338918E-8,-8.4971501655451E-6,-6.1466114631994E-8,
        4.17654403338918E-8,6.1466114631994E-8,0.0,0.0,0.0,1.0,0.0,0.0,0.0,0.0,-0.0,-0.0,-0.0,-1.0,-0.0,-0.0,-0.0,
        -0.0,3.1130989737637409E-5,-4.1765436587986837E-8,-8.49714973545552E-6,-0.00093763624831128434,
        1.0900892619138097E-6,0.0,0.0,0.0,1.0,0.0,0.0,0.0,-0.0,-0.0,-0.0,-1.0,-0.0,-0.0,-0.0,3.1130989737694391E-5,
        -2.5517486265542115E-8,-1.4104947445772003E-6,-8.4971497354728E-6,-0.00093763624831059631,0.0,0.0,0.0,1.0,
        0.0,0.0,-0.0,-0.0,-0.0,-0.0,-0.0,8.4971501656158752E-6,4.2477118830753141E-8,-2.0509684008155004E-10,
        5.1041895949625119E-8,0.0,0.0,0.0,1.0,0.0,0.0,0.0,0.0,-0.0,-0.0,-0.0,-1.0,-0.0,-0.0,-0.0,
        8.4971497354683957E-6,0.000833803913013035,-3.190152847701862E-8,-1.0900895679119706E-6,
        -0.0009376362010041088,1.4104950685543477E-6,0.0,0.0,1.0,0.0,0.0,0.0,-0.0,-0.0,-0.0,-1.0,-0.0,-0.0,-0.0,
        3.1130989737575678E-5,-6.1466108552265942E-8,-8.4971497354366E-6,-0.00093763624831199243,
        5.104188075103547E-8,0.0,0.0,0.0,1.0,0.0,0.0,-0.0,-0.0,-0.0,-0.0,8.4971497354581364E-6,
        0.00083380391301339182,-7.69810731986199E-7,-0.00093763620100453034,2.5517491150347323E-8,0.0,0.0,0.0,1.0,
        0.0,0.0,0.0,0.0,-0.0,-0.0,-0.0,-0.0,-0.0,-0.0,1.9820056068254836E-5,-2.5517476389382974E-8,
        -1.277382313185378E-10,-0.00083380391301288148,-0.00085976636244701,0.0,0.0,0.0,1.0,0.0,0.0,0.0,-0.0,-0.0,
        -0.0,-1.0,-0.0,-0.0,-0.0,-0.0,-0.0,5.7993756470700329E-8,3.1130989737643142E-5,-2.5517485912629755E-8,
        -8.4971497354570641E-6,-7.6981044396015589E-7,-0.00093763624831123,0.0,0.0,0.0,1.0,0.0,0.0,-0.0,-0.0,-0.0,
        -1.0,-0.0,-0.0,8.49715016563634E-6,5.7993775359452931E-8,0.00093763620100458347,-2.5517492750239208E-8,
        -7.6981085215610214E-7,0.0,0.0,0.0,1.0,0.0,0.0,0.0,0.0,-0.0,-0.0,-0.0,-1.0,-0.0,-0.0,7.6980986695002191E-7,
        -1.9820056068223584E-5,-2.5517476389382977E-8,0.00083380391301339106,0.00085976636244754147,0.0,0.0,0.0,1.0,
        0.0,0.0,0.0,0.0,-0.0,-0.0,-1.0,-0.0,-0.0,-0.0,-0.0,2.5517486265542121E-8,3.1130989737694391E-5,
        7.6981061239938575E-7,-8.4971497354728E-6,-0.000937636248310597,0.0,0.0,0.0,1.0,0.0,0.0,0.0,0.0,-0.0,-0.0,
        -1.0,-0.0,-0.0,-0.0,0.00093763624831128423,-4.1765440333891803E-8,-8.49715016563479E-6,
        1.0900893910065396E-6,0.0,0.0,0.0,1.0,0.0,0.0,0.0,0.0,-0.0,-0.0,-0.0,-1.0,-0.0,-0.0,-0.0,-0.0,
        2.5517487865433692E-8,-7.6981073256926574E-7,4.1765440333891803E-8,0.00093763624831128293,
        -8.49715016563479E-6,0.0,0.0,0.0,1.0,0.0,0.0,0.0,0.0,-0.0,-0.0,-0.0,-1.0,-0.0,-0.0,-0.0,-0.0,
        -3.1901531054551724E-8,0.0,8.4971501656520723E-6,-2.5517493103151746E-8,0.0,0.0,0.0,1.0,0.0,0.0,0.0,0.0,
        -0.0,-0.0,-0.0,-1.0,-0.0,-0.0,-0.0,-0.0,-4.1765449454567667E-8,-8.4971501656347912E-6,
        -0.00078187032237773848,1.19687750304504E-6,1.0900896970047287E-6,0.0,0.0,0.0,1.0,0.0,0.0,0.0,-0.0,-0.0,
        -0.0,-1.0,-0.0,-0.0,-0.0,-0.0,-0.0,-2.5517488218346114E-8,-1.277383057996246E-10,-4.247711452691102E-8,
        8.497150165652074E-6,0.0,0.0,0.0,1.0,0.0,0.0,0.0,-0.0,-0.0,-0.0,-1.0,-0.0,-0.0,-0.0,-0.0,-0.0,
        -3.1901527163311865E-8,-1.2036826344810729E-5,-0.000859766362447167,1.410495006469129E-6,
        0.00078187032237720321,0.0,0.0,0.0,1.0,0.0,0.0,0.0,-0.0,-0.0,-0.0,-1.0,-0.0,-0.0,-0.0,-0.0,
        -3.1130989737575671E-5,-6.1466108552265942E-8,8.4971497354366065E-6,0.0,0.0,0.0,1.0,0.0,0.0,0.0,-0.0,-0.0,
        -0.0,-1.0,-0.0,-0.0,-0.0,-0.0,-0.0,2.0509684008155004E-10,-8.4971501656158769E-6,-3.190153105455173E-8,
        -5.1041895949625119E-8,0.0,0.0,0.0,1.0,0.0,0.0,0.0,-0.0,-0.0,-0.0,-1.0,-0.0,-0.0,-0.0,-0.0,
        -7.6981056413003482E-7,-0.00093763624831118091,2.5517488218346108E-8,8.4971501656374237E-6,0.0,0.0,0.0,1.0,
        0.0,0.0,0.0,0.0,-0.0,-0.0,-0.0,-1.0,-0.0,-0.0,-0.0,-0.0,5.1041885201670717E-8,-2.2650033356179762E-5,
        -2.5517488218346114E-8,8.4971501656374153E-6,0.0,0.0,0.0,1.0,0.0,0.0,0.0,-0.0,-0.0,-0.0,-1.0,-0.0,-0.0,-0.0,
        1.9820056068223584E-5,7.698098669500217E-7,-2.551747638938298E-8,-0.00083380391301339193,0.0,0.0,0.0,1.0,
        0.0,0.0,0.0,0.0,-0.0,-0.0,-0.0,-1.0,-0.0,-0.0,-0.0,-0.0,2.5517492750239191E-8,8.4971501656510034E-6,
        1.6261024964684152E-10,4.24771188308966E-8,-3.4871918040629871E-9,0.0,0.0,0.0,1.0,0.0,0.0,0.0,0.0,0.0,-0.0,
        -0.0,-0.0,-1.0,-0.0,-0.0,5.10418615532681E-8,-3.5368308285989013E-5,-2.5517477507231932E-8,
        2.2650033356179769E-5,0.0,0.0,0.0,1.0,0.0,0.0,0.0,-0.0,-0.0,-0.0,-1.0,-0.0,-0.0,-0.0,2.5517490117652923E-8,
        3.4871913868165703E-11,-1.2036826344816765E-5,3.5408670177694587E-6,0.0,0.0,0.0,1.0,0.0,0.0,0.0,0.0,0.0,
        -0.0,-0.0,-1.0,-0.0,-0.0,-0.0,-0.0,-0.0,2.5517488218346121E-8,1.2773830579962463E-10,-1.1330700156807837E-7,
        8.49715016565208E-6,0.0,0.0,0.0,1.0,0.0,0.0,0.0,0.0,-0.0,-0.0,-0.0,-1.0,-0.0,-0.0,-0.0,
        2.5517489764740457E-8,1.1968773129171688E-6,-1.2036826344815318E-5,-7.6981085041259112E-7,
        0.00078187032237712168,0.0,0.0,0.0,1.0,0.0,0.0,0.0,0.0,-0.0,-0.0,-0.0,-1.0,-0.0,-0.0,-0.0,
        3.1130989737646625E-5,-7.6981044396015907E-7,-8.497149735458128E-6,-0.000937636248311175,
        2.5517486265542121E-8,0.0,0.0,0.0,1.0,0.0,0.0,0.0,-0.0,-0.0,-0.0,-0.0,3.1130989737679734E-5,
        -3.1901522125781676E-8,-1.0900892619138103E-6,-8.49714973546839E-6,-0.00093763624831075709,
        1.4104947445771984E-6,0.0,0.0,1.0,0.0,0.0,-0.0,-0.0,-0.0,-1.0,-0.0,-0.0,-0.0,8.4971497354728E-6,
        1.1329445775040093E-7,-2.5517491150347306E-8,-1.2773832264066022E-10,-4.2477114522334114E-6,0.0,0.0,0.0,1.0,
        0.0,0.0,0.0,-0.0,-0.0,-0.0,-0.0,-0.0,-0.0,-0.0,4.2477114526910973E-8,-2.5517488218346111E-8,
        -1.2773830579962473E-10,-8.497150165652074E-6,0.0,0.0,0.0,1.0,0.0,0.0,0.0,-0.0,-0.0,-0.0,-1.0,-0.0,-0.0,
        -0.0,-0.0,-0.0,0.00093763624831199373,-6.1466114631994E-8,-8.49715016561588E-6,5.1041885201670711E-8,0.0,
        0.0,0.0,1.0,0.0,0.0,0.0,-0.0,-0.0,-0.0,-1.0,-0.0,-0.0,-0.0,-0.0,8.49715016563741E-6,4.2477118830842364E-8,
        -3.4871908656977475E-11,2.551749310315175E-8,0.0,0.0,0.0,1.0,0.0,0.0,0.0,0.0,0.0,-0.0,-0.0,-0.0,-1.0,-0.0,
        -0.0,-0.0,8.49715016563741E-6,3.4871908656977404E-11,4.2477118830842358E-8,-2.5517493103151746E-8,0.0,0.0,
        0.0,1.0,0.0,0.0,0.0,0.0,0.0,-0.0,-0.0,-1.0,-0.0,-0.0,-0.0,7.69810681973355E-7,-1.2036826344796725E-5,
        -2.5517490117652913E-8,0.00078187032237752294,0.0,0.0,0.0,1.0,0.0,0.0,0.0,0.0,-0.0,-0.0,-1.0,-0.0,-0.0,-0.0,
        -0.0,-0.0,0.00093763624831075753,-3.1901524703314204E-8,-8.4971501656476711E-6,1.4104948825962408E-6,0.0,
        0.0,0.0,1.0,0.0,0.0,0.0,0.0,-0.0,-0.0,-0.0,-1.0,-0.0,-0.0,-0.0,-0.0,2.5533751784128415E-10,
        -8.4971501656374136E-6,-7.0817347533601E-8,-2.5517493103151753E-8,0.0,0.0,0.0,1.0,0.0,0.0,0.0,-0.0,-0.0,
        -0.0,-1.0,-0.0,-0.0,-0.0,-0.0,8.4971497354581364E-6,0.00083380391301339182,7.6981073198619664E-7,
        -2.5517491150347313E-8,-0.00093763620100453034,0.0,0.0,0.0,1.0,0.0,0.0,0.0,0.0,-0.0,-0.0,-1.0,-0.0,-0.0,
        -0.0,5.7993767214186308E-8,-1.2036826344795277E-5,-2.5517489764740444E-8,-7.6981068197335755E-7,
        0.00078187032237758355,0.0,0.0,0.0,1.0,0.0,0.0,0.0,-0.0,-0.0,-0.0,-1.0,-0.0,-0.0,-0.0,
        0.00093763624831117646,-7.6981056413003651E-7,-8.4971501656374034E-6,2.5517488218346118E-8,0.0,0.0,0.0,1.0,
        0.0,0.0,0.0,0.0,-0.0,-0.0,-0.0,-1.0,-0.0,-0.0,-0.0,-0.0,-0.019090619134681356,-1.9698708193212854E-5,
        -0.031801144962260629,-2.8128608814077069E-5,0.019090619134681356,1.9698708193212854E-5,
        0.031801144962260622,2.8128608814077069E-5,0.0,0.0,0.0,0.0,1.0,0.0,0.0,0.0,-0.0,-0.0,-0.0,-0.0,-1.0,-0.0,
        -0.0,-0.0,0.019090619134681356,-1.9698796053693104E-5,-0.70302132668970185,-0.70302198987546416,
        -2.812876028313039E-5,1.9698796053693104E-5,2.812876028313039E-5,0.0,0.0,0.0,0.0,1.0,0.0,0.0,0.0,-0.0,-0.0,
        -0.0,-0.0,-1.0,-0.0,-0.0,-0.0,1.9698708193212854E-5,-0.019090619134771825,-0.00051827419652806573,
        -0.031801144962405631,-0.00046646943475609973,0.019090619134771825,0.031801144962405624,0.0,0.0,0.0,0.0,1.0,
        0.0,0.0,0.0,-0.0,-0.0,-0.0,-0.0,-1.0,-0.0,-0.0,-0.0,0.031801144962260629,-0.012727560925437413,
        -1.9698786737908893E-5,-0.022268586633773707,2.8128744395695976E-5,0.0,0.0,0.0,0.0,1.0,0.0,0.0,-0.0,-0.0,
        -0.0,-0.0,-1.0,-0.0,-0.0,-0.0,-0.019090619134681356,-1.9698796053693104E-5,-2.812876028313039E-5,
        1.9698796053693104E-5,0.70302132668970185,0.70302198987546416,2.812876028313039E-5,0.0,0.0,0.0,0.0,1.0,0.0,
        0.0,0.0,-0.0,-0.0,-0.0,-0.0,-1.0,-0.0,-0.0,-0.0,-1.9698708193212854E-5,-0.019090619134771825,
        -0.031801144962405631,0.019090619134771825,0.00051827419652806551,0.031801144962405624,0.0004664694347561,
        0.0,0.0,0.0,0.0,1.0,0.0,0.0,0.0,-0.0,-0.0,-0.0,-0.0,-1.0,-0.0,-0.0,-0.0,-0.031801144962260615,
        -1.9698786737908893E-5,-2.8128744395695976E-5,1.9698786737908893E-5,0.022268586633773728,
        2.8128744395695976E-5,0.0,0.0,0.0,0.0,1.0,0.0,0.0,-0.0,-0.0,-0.0,-0.0,-1.0,-0.0,-0.0,-0.0,
        -2.8128608814077076E-5,-0.019090619134755675,0.028625312286987122,2.3917489470357002E-5,
        0.031801144962379853,0.0,0.0,0.0,0.0,1.0,0.0,0.0,-0.0,-0.0,-0.0,-0.0,-1.0,-0.0,-0.0,-0.0,
        0.019090619134771832,1.96987960536931E-5,-0.70302132668557837,-0.00051827764697021269,-0.703021989871836,
        0.0,0.0,0.0,0.0,1.0,0.0,0.0,0.0,-0.0,-0.0,-0.0,-0.0,-1.0,-0.0,-0.0,-0.0,0.70302198987546416,
        0.0095453969111649866,-1.969881865583273E-5,-2.8128799400406096E-5,1.969881865583273E-5,
        2.8128799400406096E-5,0.0,0.0,0.0,0.0,1.0,0.0,0.0,0.0,0.0,-0.0,-0.0,-0.0,-0.0,-1.0,-0.0,-0.0,
        0.019090619134771832,-0.0,0.0095453965888329766,-1.9698816577192295E-5,-0.70302389915642427,
        0.00051827845671632378,0.0,0.0,0.0,0.0,1.0,0.0,0.0,0.0,-0.0,-0.0,-0.0,-0.0,-1.0,-0.0,-0.0,
        0.019090619134755678,-2.8128760283130393E-5,-0.70302132668573147,-0.70302198987197362,2.391759050064508E-5,
        0.0,0.0,0.0,0.0,1.0,0.0,0.0,-0.0,-0.0,-0.0,-0.0,-1.0,-0.0,-0.0,-0.0,1.2662680587240977E-5,
        0.00051827419652806562,-0.019090619134789062,-0.031801144962433255,-0.00031109000754501613,
        0.019090619134789062,0.031801144962433248,0.0,0.0,0.0,0.0,1.0,0.0,0.0,0.0,-0.0,-0.0,-0.0,-1.0,-0.0,-0.0,
        1.96987960536931E-5,0.70302132668557837,-0.0,1.2662721735532011E-5,-0.0190906191347903,0.0,0.0,0.0,0.0,1.0,
        0.0,0.0,0.0,0.0,-0.0,-0.0,-0.0,-0.0,-1.0,-0.0,-0.0,1.9698786737908893E-5,-0.031801144962405617,
        -0.00051827728340074172,-0.00046647258891376628,0.02226858663388067,0.0,0.0,0.0,0.0,1.0,0.0,0.0,-0.0,-0.0,
        -0.0,-0.0,-1.0,-0.0,-0.0,-0.0,0.70302389911323138,0.00031109412840517645,-0.0095453969112158227,
        -1.2662726753574502E-5,0.0,0.0,0.0,0.0,1.0,0.0,0.0,0.0,-0.0,-0.0,-0.0,-1.0,-0.0,-0.0,-0.0,
        -0.019090619134771832,-1.96987960536931E-5,0.00051827764697021247,0.703021989871836,0.00046647295233684589,
        0.0,0.0,0.0,0.0,1.0,0.0,0.0,0.0,-0.0,-0.0,-0.0,-0.0,-1.0,-0.0,-0.0,-0.0,-0.0095453965887846749,
        -0.70302132668970174,-1.9698816577192298E-5,0.70302389915867736,0.0,0.0,0.0,0.0,1.0,0.0,-0.0,-0.0,-0.0,-0.0,
        -1.0,-0.0,-0.0,-0.0,-0.0,-0.019090619134755678,-2.8128760283130393E-5,0.70302132668573147,
        2.391759050064508E-5,0.70302198987197362,0.0,0.0,0.0,0.0,1.0,0.0,0.0,-0.0,-0.0,-0.0,-0.0,-1.0,-0.0,-0.0,
        -0.0,-1.2662717356786931E-5,-0.0,-1.9698786737908893E-5,-0.031801144962405617,0.02226858663388067,0.0,0.0,
        0.0,0.0,1.0,0.0,0.0,-0.0,-0.0,-0.0,-0.0,-1.0,-0.0,-0.0,-0.0,-1.5477721799550191E-5,-0.019090619134785883,
        -0.0318011449624282,0.019090619134785883,0.00062190102317909439,0.031801144962428196,0.0,0.0,0.0,0.0,1.0,
        0.0,0.0,0.0,-0.0,-0.0,-0.0,-0.0,-1.0,-0.0,-0.0,-0.0,-0.703023899115892,-1.9698806952807862E-5,
        -2.8128779299660833E-5,0.0095453969111649849,1.9698806952807862E-5,2.8128779299660833E-5,0.0,0.0,0.0,0.0,
        1.0,0.0,0.0,0.0,-0.0,-0.0,-0.0,-0.0,-1.0,-0.0,-0.0,-0.0,-0.031801144962379846,-2.8128744395695979E-5,
        0.0222685866338617,2.3917579535657793E-5,0.0,0.0,0.0,0.0,1.0,0.0,-0.0,-0.0,-0.0,-0.0,-1.0,-0.0,-0.0,-0.0,
        -2.3917489470357002E-5,-0.019090619134776735,-0.031801144962413506,0.019090619134776735,
        1.2662680729905015E-5,0.0318011449624135,0.0,0.0,0.0,0.0,1.0,0.0,0.0,-0.0,-0.0,-0.0,-0.0,-1.0,-0.0,-0.0,
        -0.0,0.0095453965888329766,1.9698816577192295E-5,0.70302132668557837,-0.000518278456716324,
        -0.70302389915642427,0.0,0.0,0.0,0.0,1.0,0.0,0.000518278456716324,0.0190906191347903,1.2662721735532009E-5,
        -0.70302132668433548,0.0,0.0,0.0,0.0,1.0,0.0,0.0,0.0,0.0,-0.0,-0.0,-0.0,-0.0,-1.0,-0.0,-0.0,
        0.70302198987197362,0.009545396911204521,-2.8128799400406096E-5,2.3917616316653218E-5,0.0,0.0,0.0,0.0,1.0,
        0.0,0.0,0.0,-0.0,-0.0,-0.0,-0.0,-1.0,-0.0,-0.0,0.0190906191347903,-1.2662721735532011E-5,
        -0.00062190433932153262,-0.70302132668433548,-0.70302198987074482,0.0,0.0,0.0,0.0,1.0,0.0,0.0,-0.0,-0.0,
        -0.0,-0.0,-1.0,-0.0,-0.0,-0.0,-0.0,0.019090619134776735,-2.3917590500645084E-5,-0.70302132668481432,
        -0.70302198987116749,1.2662721735532018E-5,0.0,0.0,0.0,0.0,1.0,0.0,0.0,-0.0,-0.0,-0.0,-0.0,-1.0,-0.0,-0.0,
        -0.0,2.6725935706809509E-5,-0.019090619134775496,-1.266268058724098E-5,-0.031801144962411515,
        -0.00031108991318128158,0.019090619134775496,0.031801144962411508,0.0,0.0,0.0,0.0,1.0,0.0,0.0,-1.0,-0.0,
        -0.0,-0.0,-0.0,1.2662680729905011E-5,1.409310690356228E-8,-0.0190906191347903,-0.031801144962435253,
        0.0190906191347903,0.031801144962435246,0.0,0.0,0.0,0.0,1.0,0.0,0.0,0.0,0.0,-0.0,-0.0,-0.0,-0.0,-1.0,-0.0,
        -0.0,1.266271721412136E-5,0.00051827728340074139,-0.031801144962433241,-0.00031109336351220344,
        0.022268586633901109,0.0,0.0,0.0,0.0,1.0,0.0,0.0,-0.0,-0.0,-0.0,-1.0,-0.0,-0.0,1.9698813893384417E-5,
        -0.012727560925500418,-0.703021989871836,-0.00051827834893492582,0.70301996014609,0.0,0.0,0.0,1.0,0.0,-0.0,
        -0.0,1.9698806952807862E-5,-0.70302389911363883,-0.00051827808005669451,-0.00046647340122252029,
        0.0095453969112132882,0.0,0.0,0.0,0.0,1.0,0.0,0.0,0.0,-0.0,-0.0,-0.0,-0.0,-1.0,-0.0,-0.0,-0.0,
        0.028625312287017864,0.00031109403831578147,-0.00954539658883551,-1.2662725775745235E-5,
        -0.70302389911323138,0.0,0.0,0.0,0.0,1.0,0.0,0.0,-0.0,-0.0,-0.0,-0.0,-1.0,-0.0,-0.0,2.672608714538138E-5,
        0.70302389911330532,-0.0095453969112151774,-1.2662726610908533E-5,-0.00031109412840517672,0.0,0.0,0.0,0.0,
        1.0,0.0,0.0,-0.0,-0.0,-0.0,-0.0,-1.0,-0.0,-0.0,0.0095453969112158244,3.1846509886780489E-5,
        1.409331339493356E-8,-1.2662732240991401E-5,0.0,0.0,0.0,0.0,1.0,0.0,0.0,0.0,0.0,-0.0,-0.0,-0.0,-1.0,-0.0,
        -0.0,-0.0,-0.012727560925500423,-1.9698813893384417E-5,-0.703021989871836,0.70301996014609,
        0.00051827834893492571,0.0,0.0,0.0,0.0,1.0,0.0,0.0,-0.0,-0.0,-0.0,-0.0,-1.0,-0.0,-0.0,-0.0,
        -0.019090619134785883,-1.5477777817667707E-5,-0.00046647295233684589,0.00062190433932153241,
        0.70302198987094966,0.0,0.0,0.0,0.0,1.0,0.0,0.0,-0.0,-0.0,-0.0,-1.0,-0.0,-0.0,-0.0,-0.028625312286878282,
        -1.9698804874168142E-5,1.9698804874168142E-5,0.70302389911589191,2.8128775714311272E-5,0.0,0.0,0.0,0.0,1.0,
        0.0,0.0,0.0,-0.0,-0.0,-0.0,-0.0,-1.0,-0.0,-0.0,-0.0,-1.2662732240991405E-5,-0.0,-0.0095453969112132848,
        -1.9698818655832726E-5,0.0,0.0,0.0,0.0,1.0,0.0,0.0,-0.0,-0.0,-0.0,-0.0,-1.0,-0.0,-0.0,-0.0,-0.0,
        -0.019090619134776735,-2.3917590500645084E-5,1.2662721735532018E-5,0.70302132668481432,0.70302198987116749,
        0.0,0.0,0.0,0.0,1.0,0.0,0.0,-0.0,-0.0,-0.0,-0.0,-1.0,-0.0,-0.0,-0.0,-0.0127275609254891,
        -2.8128791141921728E-5,1.5477789140033363E-5,0.70301996014627421,2.3917610862687858E-5,0.0,0.0,0.0,0.0,1.0,
        0.0,0.0,-0.0,-0.0,-0.0,-0.0,-1.0,-0.0,-0.0,-0.0,-0.0318011449624135,-0.00031109326914857016,
        1.266271735678693E-5,0.022268586633886613,0.0,0.0,0.0,0.0,1.0,0.0,0.0,-0.0,-0.0,-0.0,-0.0,-1.0,-0.0,-0.0,
        -0.0,-1.2662680729905011E-5,-5.6328242201916585E-8,-0.0190906191347903,-0.031801144962435253,
        0.0190906191347903,0.031801144962435246,0.0,0.0,0.0,0.0,1.0,0.0,0.0,-0.0,-0.0,-0.0,-0.0,-1.0,-0.0,-0.0,-0.0,
        -0.0,-1.2662717214121362E-5,-0.031801144962433241,0.022268586633901109,0.0003110933635122049,0.0,0.0,0.0,
        0.0,1.0,0.0,0.0,-0.0,-0.0,-0.0,-0.0,-1.0,-0.0,-0.0,-0.0,-1.2662726753574496E-5,-5.6328578923948309E-8,
        -3.1846505053644177E-5,0.0095453969112230981,0.0,0.0,0.0,0.0,1.0,0.0,0.0,-0.0,-0.0,-0.0,-0.0,-1.0,-0.0,-0.0,
        -0.0,-0.0,-1.9698806952807862E-5,-0.70302389911363883,0.0095453969112132882,0.00051827808005669429,0.0,0.0,
        0.0,0.0,1.0,0.0,0.0,0.0,-0.0,-0.0,-0.0,-0.0,-1.0,-0.0,-0.0,-0.0,-0.0095453969111649849,-0.70302389915867736,
        -1.969881865583273E-5,-2.8128799400406096E-5,1.969881865583273E-5,2.8128799400406096E-5,0.0,0.0,0.0,0.0,1.0,
        0.0,0.0,-0.0,-0.0,-0.0,-0.0,-1.0,-0.0,-0.0,-0.0,-0.0,0.031801144962413513,-2.39175795356578E-5,
        -0.012727560925503808,-0.022268586633886582,1.2662717356786931E-5,0.0,0.0,0.0,0.0,1.0,0.0,0.0,-0.0,-0.0,
        -0.0,-0.0,-1.0,-0.0,-0.0,1.9698804874168138E-5,0.028625312287010624,-0.0095453965888329748,
        -0.00051827799899146088,-0.70302389911363883,0.0,0.0,0.0,0.0,1.0,0.0,1.9698818655832726E-5,-0.0,
        0.0095453969112231,1.2662732240991401E-5,0.0,0.0,0.0,0.0,1.0,0.0,0.0,0.0,0.0,0.0,-0.0,-0.0,-0.0,-1.0,-0.0,
        -0.0,0.019090619134775496,2.672607037152409E-5,-1.2662721592866277E-5,-0.70302132668494977,
        -0.00031109363213255683,0.0,0.0,0.0,0.0,1.0,0.0,0.0,-1.0,-0.0,-0.0,-0.0,0.0222685866337737,
        -0.0095453969111649849,-1.9698806952807862E-5,-2.8128779299660833E-5,1.9698806952807862E-5,
        2.8128779299660833E-5,0.0,0.0,0.0,0.0,1.0,0.0,0.0,0.0,-0.0,-0.0,-0.0,-0.0,-1.0,-0.0,-0.0,
        0.009545396911213283,3.1846509886773774E-5,-1.9698818655832726E-5,0.00051827853778158494,
        0.00046647386562355766,0.0,0.0,0.0,0.0,1.0,0.0,0.0,0.0,0.0,-0.0,-0.0,-0.0,-1.0,-0.0,-0.0,-0.0,-0.0,
        0.031801144962379853,-2.8128744395695979E-5,-0.012727560925489097,-0.022268586633861678,
        2.3917579535657793E-5,0.0,0.0,0.0,0.0,1.0,0.0,0.0,-0.0,-0.0,-0.0,-0.0,-1.0,-0.0,-0.0,0.012727560925503811,
        0.70302198987116749,-2.3917610862687861E-5,-0.703019960145122,1.2662730042975289E-5,0.0,0.0,0.0,0.0,1.0,0.0,
        0.0,-0.0,-0.0,-0.0,-0.0,-1.0,-0.0,-0.0,0.028625312287010627,-1.9698804874168145E-5,-0.0095453965888329714,
        -0.70302389911363894,0.00051827799899146034,0.0,0.0,0.0,0.0,1.0,0.0,0.0,-0.0,-0.0,-0.0,-0.0,-1.0,-0.0,-0.0,
        0.019090619134785883,-1.5477777817667707E-5,-0.00046647295233684589,-0.70302132668456918,
        0.00062190433932153241,0.0,0.0,0.0,0.0,1.0,0.0,-1.0,-0.0,-0.0,-0.0,-0.0,0.0095453969112231016,
        -1.2662732240991405E-5,0.0,0.0,0.0,0.0,1.0,0.0,0.0,0.0,-0.0,-0.0,-0.0,-0.0,-1.0,-0.0,-0.0,-0.0,
        0.00031108991318128088,-0.019090619134776735,-1.2662680729905008E-5,-0.031801144962413506,
        0.019090619134776735,0.0318011449624135,0.0,0.0,0.0,0.0,1.0,0.0,0.0,0.0,-0.0,-0.0,-0.0,-0.0,-1.0,-0.0,-0.0,
        -0.0,2.672607037152409E-5,-0.019090619134775496,-1.2662721592866277E-5,-0.00031109363213255683,
        0.70302198987128661,0.0,0.0,0.0,0.0,1.0,0.0,0.0,-0.0,-0.0,-0.0,-0.0,-1.0,-0.0,-0.0,2.6726105057290468E-5,
        -0.0095453969112151756,-0.70301996014529189,-1.2662732098325213E-5,-0.00031109461283014187,0.0,0.0,0.0,0.0,
        1.0,0.0,-1.0,-0.0,-0.0,-0.0,-0.0,1.266271735678693E-5,1.4093258936886059E-8,-0.00010611233241278757,
        0.022268586633902576,0.0,0.0,0.0,0.0,1.0,0.0,0.0,0.0,-0.0,-0.0,-0.0,-0.0,-1.0,-0.0,-0.0,
        1.2662729900309189E-5,0.00051827834893492593,-0.012727560925512416,-0.703021989870864,
        -0.00031109450041720229,0.70301996014469514,0.0,0.0,0.0,1.0,0.0,0.0,-0.0,-0.0,-0.0,-0.0,-1.0,-0.0,-0.0,
        2.6726056124045137E-5,-0.0318011449624115,-1.2662717214121353E-5,-0.00031109326914856815,
        0.022268586633885149,0.0,0.0,0.0,0.0,1.0,0.0,-1.0,-0.0,-0.0,-0.0,1.2662726610908526E-5,
        0.00051827808005669429,-0.70302389911304008,-0.0003110942227687848,0.0095453969112224563,0.0,0.0,0.0,0.0,
        1.0,0.0,0.0,0.0,-0.0,-0.0,-0.0,-1.0,-0.0,-0.0,1.9698818655832726E-5,-0.009545396911213283,
        -6.3667426064628618E-5,-0.00051827853778158516,-0.00046647386562355717,0.0,0.0,0.0,0.0,1.0,0.0,0.0,-0.0,
        -0.0,-0.0,-0.0,-1.0,-0.0,-0.0,-0.0,-0.0,0.028625312287016046,2.67260839671231E-5,-0.0095453965888348622,
        -1.2662725633079306E-5,-0.70302389911330532,-0.00031109403831578217,0.0,0.0,0.0,0.0,1.0,0.0,-0.0,-0.0,-0.0,
        -0.0,-1.0,-0.0,1.2662725775745226E-5,0.028625312287037685,0.00031109413267939307,-0.0095453965888427882,
        -0.703023899112966,0.0,0.0,0.0,0.0,1.0,0.0,0.0,0.0,-0.0,-0.0,-0.0,-0.0,-1.0,-0.0,0.70302389911363894,
        -1.9698806952807862E-5,-0.009545396911213283,0.00051827808005669386,0.00046647340122252039,0.0,0.0,0.0,0.0,
        1.0,0.0,0.0,0.0,-0.0,-0.0,-0.0,-1.0,-0.0,-0.0,-0.0,0.0095453969112151774,2.6726105057290468E-5,
        0.70302389915609076,-1.2662732098325213E-5,-0.00031109461283014155,0.0,0.0,0.0,0.0,1.0,0.0,0.0,0.0,-0.0,
        -0.0,-0.0,-1.0,-0.0,-0.0,0.000311093632132556,-0.019090619134776735,-1.2662721735532011E-5,
        0.70302198987116749,0.0,0.0,0.0,0.0,1.0,0.0,0.0,0.0,-0.0,-0.0,-0.0,-0.0,-1.0,-0.0,-0.0,-0.0,
        0.0095453965888355127,-0.70302389915601671,0.019090619134776735,0.00031109363213255607,
        -1.2662721735532011E-5,0.0,0.0,0.0,0.0,1.0,0.0,0.0,0.0,-0.0,-0.0,-0.0,-0.0,-1.0,-0.0,-0.0,-0.0,
        -0.012727560925513264,0.0,1.26627322409914E-5,-0.0095453969112230929,0.0,0.0,0.0,0.0,1.0,0.0,0.0,0.0,-0.0,
        -0.0,-0.0,-0.0,-1.0,-0.0,-0.0,-0.0,-0.0190906191347903,-1.2662721735532011E-5,-0.00062190433932153262,
        0.70302132668433548,0.70302198987074482,0.0,0.0,0.0,0.0,1.0,0.0,0.0,-0.0,-0.0,-0.0,-0.0,-1.0,-0.0,-0.0,-0.0,
        -0.0,-0.0095453969112158244,-6.3667426064645816E-5,-1.4093313394933593E-8,1.2662732240991405E-5,0.0,0.0,0.0,
        0.0,1.0,0.0,0.0,-0.0,-0.0,-0.0,-0.0,-1.0,-0.0,-0.0,-0.0,-0.0,-0.012727560925510174,-1.5477789140033356E-5,
        -0.00046647367229367192,0.7030199601448206,0.00062190500529599364,0.0,0.0,0.0,0.0,1.0,0.0,0.0,-0.0,-0.0,
        -0.0,-0.0,-1.0,-0.0,-0.0,-0.0,-2.6726056124045134E-5,-0.0318011449624115,1.266271721412136E-5,0.0,0.0,0.0,
        0.0,1.0,0.0,0.0,-0.0,-0.0,-0.0,-0.0,-1.0,-0.0,-0.0,-0.0,-0.0,0.00010611233241278759,-1.266271735678693E-5,
        -0.012727560925513267,-0.022268586633902566,0.0,0.0,0.0,0.0,1.0,0.0,0.0,-0.0,-0.0,-0.0,-0.0,-1.0,-0.0,-0.0,
        -0.0,-0.70302389911323138,-0.00031109412840517781,0.0095453969112158227,1.2662726753574506E-5,0.0,0.0,0.0,
        0.0,1.0,0.0,0.0,0.0,-0.0,-0.0,-0.0,-0.0,-1.0,-0.0,-0.0,-0.0,0.022268586633886586,-2.3917602785793205E-5,
        -0.0095453969112158227,1.2662726753574504E-5,0.0,0.0,0.0,0.0,1.0,0.0,0.0,-0.0,-0.0,-0.0,-0.0,-1.0,-0.0,-0.0,
        1.9698806952807862E-5,0.70302389911363883,-0.0095453969112132882,-0.00051827808005669451,0.0,0.0,0.0,0.0,
        1.0,0.0,0.0,0.0,-0.0,-0.0,-0.0,-0.0,-1.0,-0.0,-0.0,-0.0,0.0095453965888427916,1.2662731263161793E-5,
        9.5513929494329763E-5,1.4093315727616534E-8,-0.0031846506656924463,0.0,0.0,0.0,0.0,1.0,0.0,0.0,0.0,0.0,-0.0,
        -0.0,-0.0,-0.0,-1.0,-0.0,0.022268586633861689,-2.8128779299660836E-5,-0.00954539691120452,
        2.3917602785793216E-5,0.0,0.0,0.0,0.0,1.0,0.0,0.0,-0.0,-0.0,-0.0,-0.0,-1.0,-0.0,-0.0,0.0095453969112207285,
        3.1846509886793804E-5,-1.5477792152379083E-5,2.81643067314548E-6,0.0,0.0,0.0,0.0,1.0,0.0,0.0,0.0,0.0,-0.0,
        -0.0,-0.0,-1.0,-0.0,-0.0,-0.0,-0.0,0.0095453969112158244,6.3667426064645748E-5,-1.1964809706348631E-7,
        1.2662732240991401E-5,0.0,0.0,0.0,0.0,1.0,0.0,0.0,0.0,-0.0,-0.0,-0.0,-0.0,-1.0,-0.0,-0.0,
        0.0095453965888404185,0.70302132668456918,-1.5477790827995437E-5,-0.703023899155877,0.00062190510862303544,
        0.0,0.0,0.0,0.0,1.0,0.0,0.0,0.0,-0.0,-0.0,-0.0,-0.0,-1.0,-0.0,-0.0,2.6726087145381383E-5,
        -0.70302389911330532,-1.2662726610908526E-5,-0.00031109412840517521,0.0095453969112151774,0.0,0.0,0.0,0.0,
        1.0,0.0,0.0,-1.0,-0.0,-0.0,-0.0,2.6726097733171875E-5,-0.01272756092550296,-0.70302198987128661,
        -1.2662729900309186E-5,-0.00031109440605359812,0.70301996014529189,0.0,0.0,0.0,1.0,0.0,-0.0,-0.0,-0.0,-0.0,
        -1.0,-0.0,-0.0,1.2662732098325213E-5,7.0421936123401543E-8,-0.0095453969112224528,-6.3667426064685376E-5,
        -1.4093318379358016E-6,0.0,0.0,0.0,0.0,1.0,0.0,0.0,-0.0,-0.0,-0.0,-1.0,-0.0,-0.0,-0.0,1.4093313394933583E-8,
        -0.00954539691121582,-6.3667426064645857E-5,-1.2662732240991394E-5,0.0,0.0,0.0,0.0,1.0,0.0,0.0,-0.0,-0.0,
        -0.0,-0.0,-1.0,-0.0,-0.0,-0.0,-0.0,0.0003110932691485688,-0.0318011449624135,-1.2662717356786933E-5,
        0.022268586633886613,0.0,0.0,0.0,0.0,1.0,0.0,0.0,-0.0,-0.0,-0.0,-0.0,-1.0,-0.0,-0.0,-0.0,
        1.2662726753574494E-5,1.4093297863266229E-8,-3.184650505364419E-5,0.0095453969112231033,0.0,0.0,0.0,0.0,1.0,
        0.0,0.0,0.0,0.0,-0.0,-0.0,-0.0,-0.0,-1.0,-0.0,-0.0,1.2662726753574494E-5,3.1846505053644244E-5,
        1.4093297863266219E-8,-0.0095453969112230981,0.0,0.0,0.0,0.0,1.0,0.0,0.0,0.0,0.0,-0.0,-0.0,-0.0,-1.0,-0.0,
        -0.0,0.70302389911309171,-1.5477784653254034E-5,-0.009545396911220725,0.00062190474080434219,0.0,0.0,0.0,
        0.0,1.0,0.0,0.0,0.0,-0.0,-0.0,-0.0,-1.0,-0.0,-0.0,-0.0,-0.0,0.00031109440605359866,-0.012727560925503811,
        -1.2662730042975288E-5,0.703019960145122,0.0,0.0,0.0,0.0,1.0,0.0,0.0,0.0,-0.0,-0.0,-0.0,-0.0,-1.0,-0.0,-0.0,
        -0.0,0.00011139879369970853,-1.2662726753574502E-5,-5.6328578923948216E-8,-0.0095453969112230981,0.0,0.0,
        0.0,0.0,1.0,0.0,0.0,-0.0,-0.0,-0.0,-0.0,-1.0,-0.0,-0.0,-0.0,1.266272661090853E-5,0.00051827808005669429,
        0.70302389911304008,-0.0095453969112224545,-0.0003110942227687848,0.0,0.0,0.0,0.0,1.0,0.0,0.0,0.0,-0.0,-0.0,
        -0.0,-1.0,-0.0,-0.0,0.028625312287031243,-1.5477783328870845E-5,-0.0095453965888404081,-0.70302389911309171,
        0.0006219046642527053,0.0,0.0,0.0,0.0,1.0,0.0,0.0,-0.0,-0.0,-0.0,-0.0,-1.0,-0.0,-0.0,0.00031109412840517629,
        -0.70302389911323138,-1.2662726753574499E-5,0.0095453969112158261,0.0,0.0,0.0,0.0,1.0,0.0,0.0,0.0,-0.0,-0.0,
        -0.0,-0.0,-1.0,-0.0,-0.0,-0.0,-3.6522249178886062E-5,-0.019093388890196454,-5.2157458590361115E-5,
        -0.031805094384842234,3.6522249178886062E-5,0.019093388890196454,5.2157458590361115E-5,0.031805094384842227,
        0.0,0.0,0.0,0.0,0.0,1.0,0.0,0.0,-0.0,-0.0,-0.0,-0.0,-0.0,-1.0,-0.0,-0.0,3.6522249178886062E-5,
        -0.019093388890364354,-0.00096130880269788594,-0.00086525886760264287,-0.031805094385131148,
        0.019093388890364354,0.031805094385131141,0.0,0.0,0.0,0.0,0.0,1.0,0.0,0.0,-0.0,-0.0,-0.0,-0.0,-0.0,-1.0,
        -0.0,-0.0,0.019093388890196458,-3.652233705213242E-5,-0.70301893050798425,-5.2157599879956529E-5,
        -0.70301941044164273,3.652233705213242E-5,5.2157599879956529E-5,0.0,0.0,0.0,0.0,0.0,1.0,0.0,0.0,-0.0,-0.0,
        -0.0,-0.0,-0.0,-1.0,-0.0,-0.0,5.2157458590361109E-5,-2.8693453280709772E-5,-0.019093388890325125,
        -4.43447971709128E-5,0.0318050943850639,0.0,0.0,0.0,0.0,0.0,1.0,0.0,-0.0,-0.0,-0.0,-0.0,-0.0,-1.0,-0.0,-0.0,
        -3.6522249178886062E-5,-0.019093388890364354,-0.031805094385131148,0.019093388890364354,
        0.00096130880269788594,0.00086525886760264342,0.031805094385131141,0.0,0.0,0.0,0.0,0.0,1.0,0.0,0.0,-0.0,
        -0.0,-0.0,-0.0,-0.0,-1.0,-0.0,-0.0,-0.019093388890196458,-3.652233705213242E-5,-5.2157599879956529E-5,
        3.652233705213242E-5,0.70301893050798425,5.2157599879956529E-5,0.70301941044164273,0.0,0.0,0.0,0.0,0.0,1.0,
        0.0,0.0,-0.0,-0.0,-0.0,-0.0,-0.0,-1.0,-0.0,-0.0,-5.2157458590361109E-5,-0.019093388890325125,
        -0.03180509438506391,0.019093388890325125,4.43447971709128E-5,0.0318050943850639,0.0,0.0,0.0,0.0,0.0,1.0,
        0.0,-0.0,-0.0,-0.0,-0.0,-0.0,-1.0,-0.0,-0.0,-0.031805094384842234,-3.6522333405210253E-5,
        4.9555278001043236E-5,0.022271948633834655,5.2157594188888043E-5,0.0,0.0,0.0,0.0,0.0,1.0,0.0,-0.0,-0.0,-0.0,
        -0.0,-0.0,-1.0,-0.0,-0.0,3.6522337052132434E-5,0.019093388890364351,-0.00096131182465395966,
        -0.703018930505452,-0.00086526182234124684,0.0,0.0,0.0,0.0,0.0,1.0,0.0,0.0,-0.0,-0.0,-0.0,-0.0,-0.0,-1.0,
        -0.0,-0.0,0.00086525886760264266,2.3473029391852623E-5,-0.019093388890394088,-0.0318050943851825,
        0.019093388890394088,0.031805094385182496,0.0,0.0,0.0,0.0,0.0,1.0,0.0,0.0,0.0,-0.0,-0.0,-0.0,-0.0,-0.0,-1.0,
        -0.0,3.6522337052132434E-5,-0.0,2.3473075971598973E-5,-0.019093388890392377,-0.00057718804917542433,
        0.70301893050485509,0.0,0.0,0.0,0.0,0.0,1.0,0.0,0.0,-0.0,-0.0,-0.0,-0.0,-0.0,-1.0,-0.0,3.652233340521026E-5,
        -0.031805094385131134,-0.00096131171151488386,-0.00086526170925901034,0.022271948634027636,0.0,0.0,0.0,0.0,
        0.0,1.0,0.0,-0.0,-0.0,-0.0,-0.0,-0.0,-1.0,-0.0,-0.0,0.00954717826758235,0.70301893050798414,
        -3.65223604939942E-5,-5.2157637599480248E-5,-0.70302082402767729,3.65223604939942E-5,5.2157637599480248E-5,
        0.0,0.0,0.0,0.0,0.0,1.0,0.0,0.0,-0.0,-0.0,-0.0,-0.0,-1.0,-0.0,0.019093388890364354,0.00096131182465395966,
        -0.0,0.00954717859018078,-3.6522363302599261E-5,0.0,0.0,0.0,0.0,0.0,1.0,0.0,0.0,0.0,-0.0,-0.0,-0.0,-0.0,
        -0.0,-1.0,-0.0,0.019093388890325125,-5.2157599879956516E-5,-0.70301893050571762,-0.70301941043955929,
        4.43449011383923E-5,0.0,0.0,0.0,0.0,0.0,1.0,0.0,-0.0,-0.0,-0.0,-0.0,-0.0,-1.0,-0.0,-0.0,
        0.00057718837020061448,0.70302082398273624,-2.3473084657567242E-5,-0.0095471785901811157,0.0,0.0,0.0,0.0,
        0.0,1.0,0.0,0.0,-0.0,-0.0,-0.0,-0.0,-1.0,-0.0,-0.0,-3.6522337052132434E-5,-0.019093388890364351,
        0.703018930505452,0.00086526182234124727,0.7030194104393207,0.0,0.0,0.0,0.0,0.0,1.0,0.0,0.0,-0.0,-0.0,-0.0,
        -0.0,-0.0,-1.0,-0.0,-0.0,-2.347302912727454E-5,-0.00096130880269788583,-0.019093388890392381,
        0.00057718529603716312,0.0,0.0,0.0,0.0,0.0,1.0,-0.0,-0.0,-0.0,-0.0,-0.0,-1.0,-0.0,-0.0,-0.0,
        -3.652233340521026E-5,-0.031805094385131134,0.00096131171151488386,0.022271948634027636,
        0.00086526170925901077,0.0,0.0,0.0,0.0,0.0,1.0,0.0,-0.0,-0.0,-0.0,-0.0,-0.0,-1.0,-0.0,-0.0,
        -0.0095471785901624015,-0.0,-0.019093388890325125,-5.2157599879956516E-5,4.43449011383923E-5,0.0,0.0,0.0,
        0.0,0.0,1.0,0.0,-0.0,-0.0,-0.0,-0.0,-0.0,-1.0,-0.0,-0.0,-0.012729738255777539,-3.6522358297177071E-5,
        -5.2157634143092755E-5,3.6522358297177071E-5,0.70301795752567109,5.2157634143092755E-5,0.0,0.0,0.0,0.0,0.0,
        1.0,0.0,0.0,-0.0,-0.0,-0.0,-0.0,-0.0,-1.0,-0.0,-0.0,-0.00057718512122799316,-0.019093388890365336,
        -0.031805094385133209,2.3473029391852627E-5,0.019093388890365336,0.0318050943851332,0.0,0.0,0.0,0.0,0.0,1.0,
        0.0,0.0,-0.0,-0.0,-0.0,-0.0,-0.0,-1.0,-0.0,-0.0,-5.2157594188888036E-5,-0.0318050943850639,
        4.4344896978036783E-5,0.022271948633982117,0.0,0.0,0.0,0.0,0.0,1.0,-0.0,-0.0,-0.0,-0.0,-0.0,-1.0,-0.0,-0.0,
        -0.022271948633834648,-3.6522353054843289E-5,-5.2157625694692722E-5,3.6522353054843289E-5,
        0.009547178590102354,5.2157625694692722E-5,0.0,0.0,0.0,0.0,0.0,1.0,0.0,-0.0,-0.0,-0.0,-0.0,-0.0,-1.0,-0.0,
        -0.0,2.3473075971598973E-5,0.019093388890392377,0.00096131182465395988,-0.70301893050485509,
        -0.00057718804917542433,0.0,0.0,0.0,0.0,0.0,1.0,0.703018930504855,3.6522363302599275E-5,
        0.009547178590180774,-0.00096131273359152409,0.0,0.0,0.0,0.0,0.0,1.0,0.0,0.0,0.0,-0.0,-0.0,-0.0,-0.0,-0.0,
        -1.0,-0.0,0.000865261709259011,2.3473074125247875E-5,-0.031805094385182496,0.02227194863406157,0.0,0.0,0.0,
        0.0,0.0,1.0,0.0,0.0,-0.0,-0.0,-0.0,-0.0,-0.0,-1.0,-0.0,3.6522363302599275E-5,-0.009547178590180774,
        -0.70301795752274809,-0.00096131273359152409,-0.00086526270890343563,0.0,0.0,0.0,0.0,0.0,1.0,0.0,-0.0,-0.0,
        -0.0,-0.0,-0.0,-1.0,-0.0,-0.0,-0.0,3.6522353054843289E-5,-0.022271948634027618,-0.00096131238304662065,
        -0.00086526236509131883,0.0095471785901807826,0.0,0.0,0.0,0.0,0.0,1.0,0.0,-0.0,-0.0,-0.0,-0.0,-0.0,-1.0,
        -0.0,-0.0,0.028629066348924127,-3.6522350246238987E-5,-0.0095471782675823486,-5.2157621136234768E-5,
        -0.70302082398458909,3.6522350246238987E-5,5.2157621136234768E-5,0.0,0.0,0.0,0.0,0.0,1.0,0.0,-0.0,-1.0,-0.0,
        -0.0,-0.0,0.009547178590102354,3.18484920381726E-5,-3.6522363302599268E-5,-5.2157642157939449E-5,
        3.6522363302599268E-5,5.2157642157939449E-5,0.0,0.0,0.0,0.0,0.0,1.0,0.0,0.0,0.0,-0.0,-0.0,-0.0,-0.0,-0.0,
        -1.0,-0.0,0.0095471782676424029,0.70301893050571751,-5.2157637599480228E-5,-0.70302082402620258,
        4.43449289708158E-5,0.0,0.0,0.0,0.0,0.0,1.0,0.0,-0.0,-0.0,-0.0,-0.0,-1.0,-0.0,0.019093388890386278,
        -2.8693514412082078E-5,-0.000865261822341247,-0.70301893050493458,0.001153449694857952,0.0,0.0,0.0,0.0,1.0,
        -0.0,-0.0,0.019093388890365333,-0.0005771878743661479,-0.703018930505132,-0.703019410439022,
        2.347307623617832E-5,0.0,0.0,0.0,0.0,0.0,1.0,0.0,0.0,-0.0,-0.0,-0.0,-0.0,-0.0,-1.0,-0.0,-0.0,
        4.9555306757672129E-5,0.7030208239827761,-2.3473084392987648E-5,-0.0095471785901803125,
        -0.00057718837020061221,0.0,0.0,0.0,0.0,0.0,1.0,0.0,-0.0,-0.0,-0.0,-0.0,-0.0,-1.0,-0.0,0.028629066349182733,
        0.00057718828009965415,-2.3473083193394028E-5,-0.00954717826766111,-0.70302082398273624,0.0,0.0,0.0,0.0,0.0,
        1.0,0.0,-0.0,-0.0,-0.0,-0.0,-0.0,-1.0,-0.0,2.3473084657567229E-5,2.6146252961331178E-8,
        3.1848487202701323E-5,-0.0095471785901946049,0.0,0.0,0.0,0.0,0.0,1.0,0.0,0.0,0.0,-0.0,-0.0,-0.0,-0.0,-1.0,
        -0.0,-0.0,-2.8693514412082092E-5,-0.019093388890386278,-0.00086526182234124673,0.0011534496948579533,
        0.70301893050493458,0.0,0.0,0.0,0.0,0.0,1.0,0.0,-0.0,-0.0,-0.0,-0.0,-0.0,-1.0,-0.0,-0.0,
        -3.6522358297177077E-5,-0.012729738255884648,-0.7030194104393207,0.7030179575227482,0.00086526254243436229,
        0.0,0.0,0.0,0.0,0.0,1.0,0.0,-0.0,-0.0,-0.0,-0.0,-1.0,-0.0,-0.0,-4.9555154326319392E-5,-0.019093388890363633,
        0.019093388890363633,0.00057718512122799338,0.031805094385130267,0.0,0.0,0.0,0.0,0.0,1.0,0.0,0.0,-0.0,-0.0,
        -0.0,-0.0,-0.0,-1.0,-0.0,-0.0,-0.0095471785901946014,-0.0,-2.347307623617832E-5,-0.019093388890394081,0.0,
        0.0,0.0,0.0,0.0,1.0,0.0,-0.0,-0.0,-0.0,-0.0,-0.0,-1.0,-0.0,-0.0,-0.0,-3.6522353054843289E-5,
        -0.022271948634027618,0.0095471785901807826,0.00096131238304662065,0.00086526236509131937,0.0,0.0,0.0,0.0,
        0.0,1.0,0.0,-0.0,-0.0,-0.0,-0.0,-0.0,-1.0,-0.0,-0.0,-2.869351178855761E-5,-0.031805094385168986,
        0.012729738255898576,0.0011534495816052015,0.022271948634052637,0.0,0.0,0.0,0.0,0.0,1.0,0.0,-0.0,-0.0,-0.0,
        -0.0,-0.0,-1.0,-0.0,-0.0,-5.2157625694692715E-5,-0.70302082398311461,0.009547178590162405,
        4.4344920231689462E-5,0.0,0.0,0.0,0.0,0.0,1.0,0.0,-0.0,-0.0,-0.0,-0.0,-0.0,-1.0,-0.0,-0.0,
        -0.0095471785901023523,-6.3675350751752718E-5,-3.6522363302599268E-5,-5.2157642157939449E-5,
        3.6522363302599268E-5,5.2157642157939449E-5,0.0,0.0,0.0,0.0,0.0,1.0,0.0,-0.0,-0.0,-0.0,-0.0,-0.0,-1.0,-0.0,
        -0.0,-0.0,-0.0095471782676424029,-5.2157637599480228E-5,4.43449289708158E-5,0.7030208240262027,0.0,0.0,0.0,
        0.0,0.0,1.0,0.0,-0.0,-0.0,-0.0,-0.0,-0.0,-1.0,-0.0,-0.0,-0.00954717859018111,-6.3675350752329378E-5,
        -2.61462557358624E-8,2.3473090146008748E-5,0.0,0.0,0.0,0.0,0.0,1.0,0.0,-0.0,-0.0,-0.0,-0.0,-0.0,-1.0,-0.0,
        -0.0,-0.0,-0.019093388890365333,-0.0005771878743661479,2.347307623617832E-5,0.703018930505132,0.0,0.0,0.0,
        0.0,0.0,1.0,0.0,0.0,-0.0,-0.0,-0.0,-0.0,-0.0,-1.0,-0.0,-0.0,-2.3473029391852623E-5,-0.00057718529603716518,
        -0.019093388890394088,-0.0318050943851825,0.019093388890394088,0.031805094385182496,0.0,0.0,0.0,0.0,0.0,1.0,
        0.0,-0.0,-0.0,-0.0,-0.0,-0.0,-1.0,-0.0,-0.0,-0.0,5.2157625694692715E-5,-0.02227194863398212,
        -2.8693525502607085E-5,-4.4344920231689462E-5,0.009547178590162405,0.0,0.0,0.0,0.0,0.0,1.0,0.0,-0.0,-0.0,
        -0.0,-0.0,-0.0,-1.0,-0.0,0.019093388890363633,4.9555283182156878E-5,-2.3473075971598956E-5,
        -0.70301893050519171,-0.00057718787436614454,0.0,0.0,0.0,0.0,0.0,1.0,0.019093388890394081,-0.0,
        2.3473090146008764E-5,0.0095471785901946014,0.0,0.0,0.0,0.0,0.0,1.0,0.0,0.0,0.0,0.0,-0.0,-0.0,-0.0,-0.0,
        -1.0,-0.0,3.6522350246238994E-5,0.028629066349181113,-0.0095471782676607771,-0.00096131228402486523,
        -0.70302082398295684,0.0,0.0,0.0,0.0,0.0,1.0,0.0,-0.0,-1.0,-0.0,-0.0,4.4344797170912778E-5,
        -2.3473029391852627E-5,-0.019093388890365336,-0.031805094385133209,0.019093388890365336,0.0318050943851332,
        0.0,0.0,0.0,0.0,0.0,1.0,0.0,0.0,-0.0,-0.0,-0.0,-0.0,-0.0,-1.0,-0.0,2.3473076236178317E-5,
        2.6146230500341689E-8,-0.019093388890394081,0.70301893050479525,0.70301941043871474,0.0,0.0,0.0,0.0,0.0,1.0,
        0.0,0.0,0.0,-0.0,-0.0,-0.0,-0.0,-1.0,-0.0,-0.0,-0.0,5.2157594188888036E-5,-0.0318050943850639,
        -2.8693511788557617E-5,-4.4344896978036783E-5,0.022271948633982117,0.0,0.0,0.0,0.0,0.0,1.0,0.0,-0.0,-0.0,
        -0.0,-0.0,-0.0,-1.0,-0.0,2.8693525502607071E-5,0.00086526236509131948,-0.022271948634052637,
        -0.0011534502845418316,0.0095471785901909984,0.0,0.0,0.0,0.0,0.0,1.0,0.0,-0.0,-0.0,-0.0,-0.0,-0.0,-1.0,-0.0,
        4.9555283182156878E-5,-0.019093388890363629,-2.3473075971598956E-5,-0.00057718787436614584,
        0.70301893050519171,0.0,0.0,0.0,0.0,0.0,1.0,0.0,-0.0,-0.0,-0.0,-0.0,-0.0,-1.0,-0.0,3.6522358297177077E-5,
        -0.012729738255884648,-0.7030194104393207,-0.00096131256263816563,0.7030179575227482,0.0,0.0,0.0,0.0,0.0,
        1.0,-0.0,-1.0,-0.0,-0.0,-0.0,2.3473090146008754E-5,-0.0095471785901946,0.0,0.0,0.0,0.0,0.0,1.0,0.0,0.0,-0.0,
        -0.0,-0.0,-0.0,-0.0,-1.0,-0.0,-0.0,0.7030208239845892,-3.6522353054843289E-5,-0.00954717859010235,
        -5.2157625694692722E-5,3.6522353054843289E-5,5.2157625694692722E-5,0.0,0.0,0.0,0.0,0.0,1.0,0.0,0.0,-0.0,
        -0.0,-0.0,-0.0,-0.0,-1.0,-0.0,-0.0,0.028629066349181113,-3.6522350246238987E-5,-0.0095471782676607771,
        -0.70302082398295684,0.0008652622683001951,0.0,0.0,0.0,0.0,0.0,1.0,0.0,-0.0,-0.0,-0.0,-0.0,-0.0,-1.0,-0.0,
        0.028629066349226677,-2.3473083193394021E-5,-0.0011534501810579545,-0.0095471782676746046,
        -0.70302082398252286,0.0,0.0,0.0,0.0,0.0,1.0,-0.0,-1.0,-0.0,-0.0,-0.0,0.0095471785901624015,
        3.184849203842196E-5,-1.7403678606755017E-7,4.434493230781362E-5,0.0,0.0,0.0,0.0,0.0,1.0,0.0,0.0,-0.0,-0.0,
        -0.0,-0.0,-0.0,-1.0,-0.0,0.0095471782676709964,0.70301893050493447,-2.8693530706110979E-5,
        -0.00086526261211228468,-0.70302082402570232,0.0011534505450709808,0.0,0.0,0.0,0.0,1.0,0.0,-0.0,-0.0,-0.0,
        -0.0,-0.0,-1.0,-0.0,0.0286290663491211,-5.2157621136234754E-5,-0.0095471782676424012,-0.7030208239831145,
        4.4344916894692544E-5,0.0,0.0,0.0,0.0,0.0,1.0,-0.0,-1.0,-0.0,-0.0,0.00954717826766111,0.70301893050513187,
        -0.00057718860371856837,-0.70302082402582433,2.347308868183514E-5,0.0,0.0,0.0,0.0,0.0,1.0,0.0,0.0,-0.0,-0.0,
        -0.0,-0.0,-1.0,-0.0,0.019093388890394081,-2.347307623617831E-5,-1.0445958483366056E-7,-0.70301893050479525,
        -0.70301941043871474,0.0,0.0,0.0,0.0,0.0,1.0,0.0,-0.0,-0.0,-0.0,-0.0,-0.0,-1.0,-0.0,-0.0,-0.0,
        4.9555302606141827E-5,0.028629066349180127,-2.3473082928814485E-5,-0.0095471782676603088,
        -0.00057718828009965177,-0.7030208239827761,0.0,0.0,0.0,0.0,0.0,1.0,-0.0,-0.0,-0.0,-0.0,-0.0,-1.0,
        0.0095471785901803073,4.9555321759358343E-5,0.7030208240258643,-2.3473089881429021E-5,
        -0.00057718869381955288,0.0,0.0,0.0,0.0,0.0,1.0,0.0,0.0,-0.0,-0.0,-0.0,-0.0,-0.0,-1.0,0.000577187874366147,
        -0.019093388890365333,-2.347307623617832E-5,0.703018930505132,0.703019410439022,0.0,0.0,0.0,0.0,0.0,1.0,0.0,
        0.0,-0.0,-0.0,-0.0,-0.0,-1.0,-0.0,-0.0,2.3473083193394021E-5,0.028629066349226677,0.00057718845490894847,
        -0.0095471782676746046,-0.70302082398252286,0.0,0.0,0.0,0.0,0.0,1.0,0.0,0.0,-0.0,-0.0,-0.0,-0.0,-1.0,-0.0,
        0.70302082398295673,-3.6522353054843289E-5,-0.0095471785901807826,0.0008652623650913197,0.0,0.0,0.0,0.0,0.0,
        1.0,0.0,0.0,-0.0,-0.0,-0.0,-0.0,-0.0,-1.0,-0.0,-0.0,2.3473084392987658E-5,-0.00057718854500991032,
        3.6522353054843289E-5,0.70302082398295684,-0.0095471785901807861,0.0,0.0,0.0,0.0,0.0,1.0,0.0,0.0,-0.0,-0.0,
        -0.0,-0.0,-0.0,-1.0,-0.0,-0.0,-2.8693532638693606E-5,0.0,0.0095471785901946049,-2.3473090146008737E-5,0.0,
        0.0,0.0,0.0,0.0,1.0,0.0,0.0,-0.0,-0.0,-0.0,-0.0,-0.0,-1.0,-0.0,-0.0,-3.6522363302599275E-5,
        -0.009547178590180774,-0.70301795752274809,0.00096131273359152409,0.00086526270890343617,0.0,0.0,0.0,0.0,
        0.0,1.0,0.0,-0.0,-0.0,-0.0,-0.0,-0.0,-1.0,-0.0,-0.0,-0.0,-2.3473084657567229E-5,-1.044596382372305E-7,
        -3.1848487202701255E-5,0.0095471785901946049,0.0,0.0,0.0,0.0,0.0,1.0,0.0,-0.0,-0.0,-0.0,-0.0,-0.0,-1.0,-0.0,
        -0.0,-0.0,-2.8693529139888997E-5,-0.012729738255898571,-0.703019410438843,0.0011534504686312259,
        0.703017957522159,0.0,0.0,0.0,0.0,0.0,1.0,0.0,-0.0,-0.0,-0.0,-0.0,-0.0,-1.0,-0.0,-0.0,-0.0286290663491211,
        -5.2157621136234754E-5,0.0095471782676424012,0.0,0.0,0.0,0.0,0.0,1.0,0.0,-0.0,-0.0,-0.0,-0.0,-0.0,-1.0,-0.0,
        -0.0,-0.0,1.7403678606755019E-7,-0.0095471785901624015,-2.869353263869362E-5,-4.43449323078136E-5,0.0,0.0,
        0.0,0.0,0.0,1.0,0.0,-0.0,-0.0,-0.0,-0.0,-0.0,-1.0,-0.0,-0.0,-0.00057718837020061568,-0.70302082398273624,
        2.3473084657567242E-5,0.00954717859018112,0.0,0.0,0.0,0.0,0.0,1.0,0.0,0.0,-0.0,-0.0,-0.0,-0.0,-0.0,-1.0,
        -0.0,-0.0,4.4344920231689448E-5,-0.022271948634028347,-2.3473084657567242E-5,0.00954717859018111,0.0,0.0,
        0.0,0.0,0.0,1.0,0.0,-0.0,-0.0,-0.0,-0.0,-0.0,-1.0,-0.0,0.019093388890365333,0.00057718787436614671,
        -2.347307623617832E-5,-0.703018930505132,0.0,0.0,0.0,0.0,0.0,1.0,0.0,0.0,-0.0,-0.0,-0.0,-0.0,-0.0,-1.0,-0.0,
        -0.0,2.3473089881429038E-5,0.0095471785901937965,1.3060593352310909E-7,3.1848492038550092E-5,
        -2.6146264969321444E-6,0.0,0.0,0.0,0.0,0.0,1.0,0.0,0.0,0.0,-0.0,-0.0,-0.0,-0.0,-0.0,-1.0,
        4.4344896978036769E-5,-0.0318050943851332,-2.3473074125247868E-5,0.02227194863402835,0.0,0.0,0.0,0.0,0.0,
        1.0,0.0,-0.0,-0.0,-0.0,-0.0,-0.0,-1.0,-0.0,2.3473087461600324E-5,2.6146260689378505E-8,
        -0.012729738255903513,0.0031837672149024575,0.0,0.0,0.0,0.0,0.0,1.0,0.0,0.0,0.0,-0.0,-0.0,-0.0,-0.0,-1.0,
        -0.0,-0.0,-0.0,2.3473084657567235E-5,1.0445963823723051E-7,-0.00011141562924503268,0.0095471785901946014,
        0.0,0.0,0.0,0.0,0.0,1.0,0.0,0.0,-0.0,-0.0,-0.0,-0.0,-0.0,-1.0,-0.0,2.3473087197020675E-5,
        0.00096131256263816585,-0.012729738255902429,-0.00057718871560916,0.70301795752206764,0.0,0.0,0.0,0.0,0.0,
        1.0,0.0,0.0,-0.0,-0.0,-0.0,-0.0,-0.0,-1.0,-0.0,0.028629066349182733,-0.00057718828009965676,
        -0.00954717826766111,-0.70302082398273624,2.3473083193394035E-5,0.0,0.0,0.0,0.0,0.0,1.0,0.0,-0.0,-1.0,-0.0,
        -0.0,0.028629066349214694,-2.8693523570024966E-5,-0.0008652622683001951,-0.0095471782676709929,
        -0.70302082398261434,0.0011534501810579526,0.0,0.0,0.0,0.0,1.0,-0.0,-0.0,-0.0,-0.0,-0.0,-1.0,-0.0,
        0.0095471782676746011,9.5523836332220613E-5,-2.3473088681835134E-5,-1.0445966183159716E-7,
        -0.0031848488808076322,0.0,0.0,0.0,0.0,0.0,1.0,0.0,-0.0,-0.0,-0.0,-0.0,-1.0,-0.0,-0.0,3.1848487202701309E-5,
        -2.3473084657567225E-5,-1.0445963823723051E-7,-0.0095471785901946014,0.0,0.0,0.0,0.0,0.0,1.0,0.0,-0.0,-0.0,
        -0.0,-0.0,-0.0,-1.0,-0.0,-0.0,-0.0,0.70302082398311461,-5.2157625694692715E-5,-0.009547178590162405,
        4.4344920231689462E-5,0.0,0.0,0.0,0.0,0.0,1.0,0.0,-0.0,-0.0,-0.0,-0.0,-0.0,-1.0,-0.0,-0.0,
        0.0095471785901811122,3.1848492038499474E-5,-2.6146255735862374E-8,2.3473090146008754E-5,0.0,0.0,0.0,0.0,
        0.0,1.0,0.0,0.0,0.0,-0.0,-0.0,-0.0,-0.0,-0.0,-1.0,-0.0,0.00954717859018111,2.61462557358624E-8,
        3.1848492038499446E-5,-2.3473090146008748E-5,0.0,0.0,0.0,0.0,0.0,1.0,0.0,0.0,0.0,-0.0,-0.0,-0.0,-0.0,-1.0,
        -0.0,0.00057718854079985679,-0.012729738255885078,-2.347308746160033E-5,0.70301795752239227,0.0,0.0,0.0,0.0,
        0.0,1.0,0.0,0.0,-0.0,-0.0,-0.0,-0.0,-1.0,-0.0,-0.0,-0.0,0.70302082398261434,-2.8693525502607068E-5,
        -0.0095471785901909967,0.0011534502845418292,0.0,0.0,0.0,0.0,0.0,1.0,0.0,0.0,-0.0,-0.0,-0.0,-0.0,-0.0,-1.0,
        -0.0,-0.0,2.2183590036490517E-7,-0.00954717859018111,-6.3675350752329338E-5,-2.3473090146008754E-5,0.0,0.0,
        0.0,0.0,0.0,1.0,0.0,-0.0,-0.0,-0.0,-0.0,-0.0,-1.0,-0.0,-0.0,0.00954717826766111,0.70301893050513187,
        0.00057718860371856881,-2.3473088681835137E-5,-0.70302082402582433,0.0,0.0,0.0,0.0,0.0,1.0,0.0,0.0,-0.0,
        -0.0,-0.0,-0.0,-1.0,-0.0,4.9555314435549588E-5,-0.012729738255883995,-2.3473087197020668E-5,
        -0.00057718854079985842,0.70301795752246,0.0,0.0,0.0,0.0,0.0,1.0,0.0,-0.0,-0.0,-0.0,-0.0,-0.0,-1.0,-0.0,
        0.70302082398273635,-0.00057718837020061676,-0.0095471785901811157,2.3473084657567235E-5,0.0,0.0,0.0,0.0,
        0.0,1.0,0.0,0.0,-0.0,-0.0,-0.0,-0.0,-0.0,-1.0,-0.0,-0.0,0.019090619134681356,1.9698708193212854E-5,
        0.031801144962260629,2.8128608814077069E-5,-0.019090619134681356,-1.9698708193212854E-5,
        -0.031801144962260622,-2.8128608814077069E-5,0.0,0.0,0.0,0.0,0.0,0.0,1.0,0.0,-0.0,-0.0,-0.0,-0.0,-0.0,-0.0,
        -1.0,-0.0,-0.019090619134681356,1.9698796053693104E-5,0.70302132668970185,0.70302198987546416,
        2.812876028313039E-5,-1.9698796053693104E-5,-2.812876028313039E-5,0.0,0.0,0.0,0.0,0.0,0.0,0.0,0.0,-0.0,-0.0,
        -0.0,-0.0,-0.0,-0.0,-1.0,-0.0,-1.9698708193212854E-5,0.019090619134771825,0.00051827419652806573,
        0.031801144962405631,0.00046646943475609973,-0.019090619134771825,-0.031801144962405624,0.0,0.0,0.0,0.0,0.0,
        0.0,1.0,0.0,-0.0,-0.0,-0.0,-0.0,-0.0,-0.0,-1.0,-0.0,-0.031801144962260629,0.012727560925437413,
        1.9698786737908893E-5,0.022268586633773707,-2.8128744395695976E-5,0.0,0.0,0.0,0.0,0.0,0.0,1.0,-0.0,-0.0,
        -0.0,-0.0,-0.0,-0.0,-0.0,-0.0,0.019090619134681356,1.9698796053693104E-5,2.812876028313039E-5,
        -1.9698796053693104E-5,-0.70302132668970185,-0.70302198987546416,-2.812876028313039E-5,0.0,0.0,0.0,0.0,0.0,
        0.0,1.0,0.0,-0.0,-0.0,-0.0,-0.0,-0.0,-0.0,-0.0,-0.0,1.9698708193212854E-5,0.019090619134771825,
        0.031801144962405631,-0.019090619134771825,-0.00051827419652806551,-0.031801144962405624,
        -0.0004664694347561,0.0,0.0,0.0,0.0,0.0,0.0,1.0,0.0,-0.0,-0.0,-0.0,-0.0,-0.0,-0.0,-1.0,-0.0,
        0.031801144962260615,1.9698786737908893E-5,2.8128744395695976E-5,-1.9698786737908893E-5,
        -0.022268586633773728,-2.8128744395695976E-5,0.0,0.0,0.0,0.0,0.0,0.0,0.0,-0.0,-0.0,-0.0,-0.0,-0.0,-0.0,-1.0,
        -0.0,2.8128608814077076E-5,0.019090619134755675,-0.028625312286987122,-2.3917489470357002E-5,
        -0.031801144962379853,0.0,0.0,0.0,0.0,0.0,0.0,1.0,-0.0,-0.0,-0.0,-0.0,-0.0,-0.0,-1.0,-0.0,
        -0.019090619134771832,-1.96987960536931E-5,0.70302132668557837,0.00051827764697021269,0.703021989871836,0.0,
        0.0,0.0,0.0,0.0,0.0,0.0,0.0,-0.0,-0.0,-0.0,-0.0,-0.0,-0.0,-1.0,-0.0,-0.70302198987546416,
        -0.0095453969111649866,1.969881865583273E-5,2.8128799400406096E-5,-1.969881865583273E-5,
        -2.8128799400406096E-5,0.0,0.0,0.0,0.0,0.0,0.0,1.0,0.0,0.0,-0.0,-0.0,-0.0,-0.0,-0.0,-0.0,-0.0,
        -0.019090619134771832,-1.0,-0.0095453965888329766,1.9698816577192295E-5,0.70302389915642427,
        -0.00051827845671632378,0.0,0.0,0.0,0.0,0.0,0.0,0.0,0.0,-0.0,-0.0,-0.0,-0.0,-0.0,-0.0,-0.0,
        -0.019090619134755678,2.8128760283130393E-5,0.70302132668573147,0.70302198987197362,-2.391759050064508E-5,
        0.0,0.0,0.0,0.0,0.0,0.0,0.0,-0.0,-0.0,-0.0,-0.0,-0.0,-0.0,-1.0,-0.0,-1.2662680587240977E-5,
        -0.00051827419652806562,0.019090619134789062,0.031801144962433255,0.00031109000754501613,
        -0.019090619134789062,-0.031801144962433248,0.0,0.0,0.0,0.0,0.0,0.0,1.0,0.0,-0.0,-0.0,-0.0,-0.0,-0.0,-1.0,
        -1.96987960536931E-5,-0.70302132668557837,-0.0,-1.2662721735532011E-5,0.0190906191347903,0.0,0.0,0.0,0.0,
        0.0,0.0,1.0,0.0,0.0,-0.0,-0.0,-0.0,-0.0,-0.0,-0.0,-0.0,-1.9698786737908893E-5,0.031801144962405617,
        0.00051827728340074172,0.00046647258891376628,-0.02226858663388067,0.0,0.0,0.0,0.0,0.0,0.0,0.0,-0.0,-0.0,
        -0.0,-0.0,-0.0,-0.0,-1.0,-0.0,-0.70302389911323138,-0.00031109412840517645,0.0095453969112158227,
        1.2662726753574502E-5,0.0,0.0,0.0,0.0,0.0,0.0,1.0,0.0,-0.0,-0.0,-0.0,-0.0,-0.0,-0.0,-0.0,
        0.019090619134771832,1.96987960536931E-5,-0.00051827764697021247,-0.703021989871836,-0.00046647295233684589,
        0.0,0.0,0.0,0.0,0.0,0.0,1.0,0.0,-0.0,-0.0,-0.0,-0.0,-0.0,-0.0,-0.0,-0.0,0.0095453965887846749,
        0.70302132668970174,1.9698816577192298E-5,-0.70302389915867736,0.0,0.0,0.0,0.0,0.0,0.0,-0.0,-0.0,-0.0,-0.0,
        -0.0,-0.0,-0.0,-0.0,-0.0,0.019090619134755678,2.8128760283130393E-5,-0.70302132668573147,
        -2.391759050064508E-5,-0.70302198987197362,0.0,0.0,0.0,0.0,0.0,0.0,1.0,-0.0,-0.0,-0.0,-0.0,-0.0,-0.0,-0.0,
        -0.0,1.2662717356786931E-5,-0.0,1.9698786737908893E-5,0.031801144962405617,-0.02226858663388067,0.0,0.0,0.0,
        0.0,0.0,0.0,0.0,-0.0,-0.0,-0.0,-0.0,-0.0,-0.0,-1.0,-0.0,1.5477721799550191E-5,0.019090619134785883,
        0.0318011449624282,-0.019090619134785883,-0.00062190102317909439,-0.031801144962428196,0.0,0.0,0.0,0.0,0.0,
        0.0,1.0,0.0,-0.0,-0.0,-0.0,-0.0,-0.0,-0.0,-1.0,-0.0,0.703023899115892,1.9698806952807862E-5,
        2.8128779299660833E-5,-0.0095453969111649849,-1.9698806952807862E-5,-2.8128779299660833E-5,0.0,0.0,0.0,0.0,
        0.0,0.0,0.0,0.0,-0.0,-0.0,-0.0,-0.0,-0.0,-0.0,-1.0,-0.0,0.031801144962379846,2.8128744395695979E-5,
        -0.0222685866338617,-2.3917579535657793E-5,0.0,0.0,0.0,0.0,0.0,0.0,-0.0,-0.0,-0.0,-0.0,-0.0,-0.0,-1.0,-0.0,
        2.3917489470357002E-5,0.019090619134776735,0.031801144962413506,-0.019090619134776735,
        -1.2662680729905015E-5,-0.0318011449624135,0.0,0.0,0.0,0.0,0.0,0.0,1.0,-0.0,-0.0,-0.0,-0.0,-0.0,-0.0,-1.0,
        -0.0,-0.0095453965888329766,-1.9698816577192295E-5,-0.70302132668557837,0.000518278456716324,
        0.70302389915642427,0.0,0.0,0.0,0.0,0.0,0.0,-0.000518278456716324,-0.0190906191347903,
        -1.2662721735532009E-5,0.70302132668433548,0.0,0.0,0.0,0.0,0.0,0.0,0.0,0.0,0.0,-0.0,-0.0,-0.0,-0.0,-0.0,
        -0.0,-1.0,-0.70302198987197362,-0.009545396911204521,2.8128799400406096E-5,-2.3917616316653218E-5,0.0,0.0,
        0.0,0.0,0.0,0.0,1.0,0.0,-0.0,-0.0,-0.0,-0.0,-0.0,-0.0,-0.0,-0.0190906191347903,1.2662721735532011E-5,
        0.00062190433932153262,0.70302132668433548,0.70302198987074482,0.0,0.0,0.0,0.0,0.0,0.0,0.0,-0.0,-0.0,-0.0,
        -0.0,-0.0,-0.0,-1.0,-0.0,-0.0,-0.019090619134776735,2.3917590500645084E-5,0.70302132668481432,
        0.70302198987116749,-1.2662721735532018E-5,0.0,0.0,0.0,0.0,0.0,0.0,0.0,-0.0,-0.0,-0.0,-0.0,-0.0,-0.0,-1.0,
        -0.0,-2.6725935706809509E-5,0.019090619134775496,1.266268058724098E-5,0.031801144962411515,
        0.00031108991318128158,-0.019090619134775496,-0.031801144962411508,0.0,0.0,0.0,0.0,0.0,0.0,1.0,-0.0,-0.0,
        -1.0,-0.0,-0.0,-1.2662680729905011E-5,-1.409310690356228E-8,0.0190906191347903,0.031801144962435253,
        -0.0190906191347903,-0.031801144962435246,0.0,0.0,0.0,0.0,0.0,0.0,1.0,0.0,0.0,-0.0,-0.0,-0.0,-0.0,-0.0,-0.0,
        -1.0,-1.266271721412136E-5,-0.00051827728340074139,0.031801144962433241,0.00031109336351220344,
        -0.022268586633901109,0.0,0.0,0.0,0.0,0.0,0.0,0.0,-0.0,-0.0,-0.0,-0.0,-0.0,-1.0,-1.9698813893384417E-5,
        0.012727560925500418,0.703021989871836,0.00051827834893492582,-0.70301996014609,0.0,0.0,0.0,0.0,0.0,-0.0,
        -0.0,-1.9698806952807862E-5,0.70302389911363883,0.00051827808005669451,0.00046647340122252029,
        -0.0095453969112132882,0.0,0.0,0.0,0.0,0.0,0.0,0.0,0.0,-0.0,-0.0,-0.0,-0.0,-0.0,-0.0,-1.0,-0.0,
        -0.028625312287017864,-0.00031109403831578147,0.00954539658883551,1.2662725775745235E-5,0.70302389911323138,
        0.0,0.0,0.0,0.0,0.0,0.0,0.0,-0.0,-0.0,-0.0,-0.0,-0.0,-0.0,-0.0,-2.672608714538138E-5,-0.70302389911330532,
        0.0095453969112151774,1.2662726610908533E-5,0.00031109412840517672,0.0,0.0,0.0,0.0,0.0,0.0,1.0,-0.0,-0.0,
        -0.0,-0.0,-0.0,-0.0,-0.0,-0.0095453969112158244,-3.1846509886780489E-5,-1.409331339493356E-8,
        1.2662732240991401E-5,0.0,0.0,0.0,0.0,0.0,0.0,1.0,0.0,0.0,-0.0,-0.0,-0.0,-0.0,-0.0,-0.0,-0.0,
        0.012727560925500423,1.9698813893384417E-5,0.703021989871836,-0.70301996014609,-0.00051827834893492571,0.0,
        0.0,0.0,0.0,0.0,0.0,0.0,-0.0,-0.0,-0.0,-0.0,-0.0,-0.0,-0.0,-0.0,0.019090619134785883,1.5477777817667707E-5,
        0.00046647295233684589,-0.00062190433932153241,-0.70302198987094966,0.0,0.0,0.0,0.0,0.0,0.0,1.0,-0.0,-0.0,
        -0.0,-0.0,-0.0,-0.0,-0.0,0.028625312286878282,1.9698804874168142E-5,-1.9698804874168142E-5,
        -0.70302389911589191,-2.8128775714311272E-5,0.0,0.0,0.0,0.0,0.0,0.0,1.0,0.0,-0.0,-0.0,-0.0,-0.0,-0.0,-0.0,
        -0.0,-0.0,1.2662732240991405E-5,-0.0,0.0095453969112132848,1.9698818655832726E-5,0.0,0.0,0.0,0.0,0.0,0.0,
        0.0,-0.0,-0.0,-0.0,-0.0,-0.0,-0.0,-1.0,-0.0,-0.0,0.019090619134776735,2.3917590500645084E-5,
        -1.2662721735532018E-5,-0.70302132668481432,-0.70302198987116749,0.0,0.0,0.0,0.0,0.0,0.0,1.0,-0.0,-0.0,-0.0,
        -0.0,-0.0,-0.0,-0.0,-0.0,0.0127275609254891,2.8128791141921728E-5,-1.5477789140033363E-5,
        -0.70301996014627421,-2.3917610862687858E-5,0.0,0.0,0.0,0.0,0.0,0.0,1.0,-0.0,-0.0,-0.0,-0.0,-0.0,-0.0,-0.0,
        -0.0,0.0318011449624135,0.00031109326914857016,-1.266271735678693E-5,-0.022268586633886613,0.0,0.0,0.0,0.0,
        0.0,0.0,0.0,-0.0,-0.0,-0.0,-0.0,-0.0,-0.0,-1.0,-0.0,1.2662680729905011E-5,5.6328242201916585E-8,
        0.0190906191347903,0.031801144962435253,-0.0190906191347903,-0.031801144962435246,0.0,0.0,0.0,0.0,0.0,0.0,
        1.0,-0.0,-0.0,-0.0,-0.0,-0.0,-0.0,-1.0,-0.0,-0.0,1.2662717214121362E-5,0.031801144962433241,
        -0.022268586633901109,-0.0003110933635122049,0.0,0.0,0.0,0.0,0.0,0.0,0.0,-0.0,-0.0,-0.0,-0.0,-0.0,-0.0,-1.0,
        -0.0,1.2662726753574496E-5,5.6328578923948309E-8,3.1846505053644177E-5,-0.0095453969112230981,0.0,0.0,0.0,
        0.0,0.0,0.0,0.0,-0.0,-0.0,-0.0,-0.0,-0.0,-0.0,-1.0,-0.0,-0.0,1.9698806952807862E-5,0.70302389911363883,
        -0.0095453969112132882,-0.00051827808005669429,0.0,0.0,0.0,0.0,0.0,0.0,0.0,0.0,-0.0,-0.0,-0.0,-0.0,-0.0,
        -0.0,-1.0,-0.0,0.0095453969111649849,0.70302389915867736,1.969881865583273E-5,2.8128799400406096E-5,
        -1.969881865583273E-5,-2.8128799400406096E-5,0.0,0.0,0.0,0.0,0.0,0.0,0.0,-0.0,-0.0,-0.0,-0.0,-0.0,-0.0,-1.0,
        -0.0,-0.0,-0.031801144962413513,2.39175795356578E-5,0.012727560925503808,0.022268586633886582,
        -1.2662717356786931E-5,0.0,0.0,0.0,0.0,0.0,0.0,1.0,-0.0,-0.0,-0.0,-0.0,-0.0,-0.0,-0.0,
        -1.9698804874168138E-5,-0.028625312287010624,0.0095453965888329748,0.00051827799899146088,
        0.70302389911363883,0.0,0.0,0.0,0.0,0.0,0.0,-1.9698818655832726E-5,-0.0,-0.0095453969112231,
        -1.2662732240991401E-5,0.0,0.0,0.0,0.0,0.0,0.0,1.0,0.0,0.0,0.0,-0.0,-0.0,-0.0,-0.0,-0.0,-0.0,
        -0.019090619134775496,-2.672607037152409E-5,1.2662721592866277E-5,0.70302132668494977,
        0.00031109363213255683,0.0,0.0,0.0,0.0,0.0,0.0,0.0,-0.0,-0.0,-1.0,-0.0,-0.0222685866337737,
        0.0095453969111649849,1.9698806952807862E-5,2.8128779299660833E-5,-1.9698806952807862E-5,
        -2.8128779299660833E-5,0.0,0.0,0.0,0.0,0.0,0.0,1.0,0.0,-0.0,-0.0,-0.0,-0.0,-0.0,-0.0,-0.0,
        -0.009545396911213283,-3.1846509886773774E-5,1.9698818655832726E-5,-0.00051827853778158494,
        -0.00046647386562355766,0.0,0.0,0.0,0.0,0.0,0.0,1.0,0.0,0.0,-0.0,-0.0,-0.0,-0.0,-0.0,-0.0,-0.0,-0.0,
        -0.031801144962379853,2.8128744395695979E-5,0.012727560925489097,0.022268586633861678,
        -2.3917579535657793E-5,0.0,0.0,0.0,0.0,0.0,0.0,1.0,-0.0,-0.0,-0.0,-0.0,-0.0,-0.0,-0.0,-0.012727560925503811,
        -0.70302198987116749,2.3917610862687861E-5,0.703019960145122,-1.2662730042975289E-5,0.0,0.0,0.0,0.0,0.0,0.0,
        0.0,-0.0,-0.0,-0.0,-0.0,-0.0,-0.0,-0.0,-0.028625312287010627,1.9698804874168145E-5,0.0095453965888329714,
        0.70302389911363894,-0.00051827799899146034,0.0,0.0,0.0,0.0,0.0,0.0,0.0,-0.0,-0.0,-0.0,-0.0,-0.0,-0.0,-0.0,
        -0.019090619134785883,1.5477777817667707E-5,0.00046647295233684589,0.70302132668456918,
        -0.00062190433932153241,0.0,0.0,0.0,0.0,0.0,0.0,-0.0,-0.0,-1.0,-0.0,-0.0,-0.0095453969112231016,
        1.2662732240991405E-5,0.0,0.0,0.0,0.0,0.0,0.0,1.0,0.0,-0.0,-0.0,-0.0,-0.0,-0.0,-0.0,-0.0,-0.0,
        -0.00031108991318128088,0.019090619134776735,1.2662680729905008E-5,0.031801144962413506,
        -0.019090619134776735,-0.0318011449624135,0.0,0.0,0.0,0.0,0.0,0.0,1.0,0.0,-0.0,-0.0,-0.0,-0.0,-0.0,-0.0,
        -1.0,-0.0,-2.672607037152409E-5,0.019090619134775496,1.2662721592866277E-5,0.00031109363213255683,
        -0.70302198987128661,0.0,0.0,0.0,0.0,0.0,0.0,1.0,-0.0,-0.0,-0.0,-0.0,-0.0,-0.0,-0.0,-2.6726105057290468E-5,
        0.0095453969112151756,0.70301996014529189,1.2662732098325213E-5,0.00031109461283014187,0.0,0.0,0.0,0.0,0.0,
        0.0,-0.0,-0.0,-1.0,-0.0,-0.0,-1.266271735678693E-5,-1.4093258936886059E-8,0.00010611233241278757,
        -0.022268586633902576,0.0,0.0,0.0,0.0,0.0,0.0,0.0,0.0,-0.0,-0.0,-0.0,-0.0,-0.0,-0.0,-1.0,
        -1.2662729900309189E-5,-0.00051827834893492593,0.012727560925512416,0.703021989870864,
        0.00031109450041720229,-0.70301996014469514,0.0,0.0,0.0,0.0,0.0,0.0,-0.0,-0.0,-0.0,-0.0,-0.0,-0.0,-0.0,
        -2.6726056124045137E-5,0.0318011449624115,1.2662717214121353E-5,0.00031109326914856815,
        -0.022268586633885149,0.0,0.0,0.0,0.0,0.0,0.0,-0.0,-0.0,-1.0,-0.0,-1.2662726610908526E-5,
        -0.00051827808005669429,0.70302389911304008,0.0003110942227687848,-0.0095453969112224563,0.0,0.0,0.0,0.0,
        0.0,0.0,0.0,0.0,-0.0,-0.0,-0.0,-0.0,-0.0,-1.0,-1.9698818655832726E-5,0.009545396911213283,
        6.3667426064628618E-5,0.00051827853778158516,0.00046647386562355717,0.0,0.0,0.0,0.0,0.0,0.0,0.0,-0.0,-0.0,
        -0.0,-0.0,-0.0,-0.0,-1.0,-0.0,-0.0,-0.028625312287016046,-2.67260839671231E-5,0.0095453965888348622,
        1.2662725633079306E-5,0.70302389911330532,0.00031109403831578217,0.0,0.0,0.0,0.0,0.0,0.0,-0.0,-0.0,-0.0,
        -0.0,-0.0,-0.0,-1.2662725775745226E-5,-0.028625312287037685,-0.00031109413267939307,0.0095453965888427882,
        0.703023899112966,0.0,0.0,0.0,0.0,0.0,0.0,0.0,0.0,-0.0,-0.0,-0.0,-0.0,-0.0,-0.0,-0.70302389911363894,
        1.9698806952807862E-5,0.009545396911213283,-0.00051827808005669386,-0.00046647340122252039,0.0,0.0,0.0,0.0,
        0.0,0.0,1.0,0.0,-0.0,-0.0,-0.0,-0.0,-0.0,-0.0,-0.0,-0.0095453969112151774,-2.6726105057290468E-5,
        -0.70302389915609076,1.2662732098325213E-5,0.00031109461283014155,0.0,0.0,0.0,0.0,0.0,0.0,1.0,0.0,-0.0,-0.0,
        -0.0,-0.0,-0.0,-0.0,-0.000311093632132556,0.019090619134776735,1.2662721735532011E-5,-0.70302198987116749,
        0.0,0.0,0.0,0.0,0.0,0.0,1.0,0.0,-0.0,-0.0,-0.0,-0.0,-0.0,-0.0,-0.0,-0.0,-0.0095453965888355127,
        0.70302389915601671,-0.019090619134776735,-0.00031109363213255607,1.2662721735532011E-5,0.0,0.0,0.0,0.0,0.0,
        0.0,0.0,0.0,-0.0,-0.0,-0.0,-0.0,-0.0,-0.0,-1.0,-0.0,0.012727560925513264,1.0,-1.26627322409914E-5,
        0.0095453969112230929,0.0,0.0,0.0,0.0,0.0,0.0,0.0,0.0,-0.0,-0.0,-0.0,-0.0,-0.0,-0.0,-1.0,-0.0,
        0.0190906191347903,1.2662721735532011E-5,0.00062190433932153262,-0.70302132668433548,-0.70302198987074482,
        0.0,0.0,0.0,0.0,0.0,0.0,1.0,-0.0,-0.0,-0.0,-0.0,-0.0,-0.0,-0.0,-0.0,-0.0,0.0095453969112158244,
        6.3667426064645816E-5,1.4093313394933593E-8,-1.2662732240991405E-5,0.0,0.0,0.0,0.0,0.0,0.0,0.0,-0.0,-0.0,
        -0.0,-0.0,-0.0,-0.0,-1.0,-0.0,-0.0,0.012727560925510174,1.5477789140033356E-5,0.00046647367229367192,
        -0.7030199601448206,-0.00062190500529599364,0.0,0.0,0.0,0.0,0.0,0.0,1.0,-0.0,-0.0,-0.0,-0.0,-0.0,-0.0,-0.0,
        -0.0,2.6726056124045134E-5,0.0318011449624115,-1.266271721412136E-5,0.0,0.0,0.0,0.0,0.0,0.0,1.0,-0.0,-0.0,
        -0.0,-0.0,-0.0,-0.0,-1.0,-0.0,-0.0,-0.00010611233241278759,1.266271735678693E-5,0.012727560925513267,
        0.022268586633902566,0.0,0.0,0.0,0.0,0.0,0.0,1.0,-0.0,-0.0,-0.0,-0.0,-0.0,-0.0,-0.0,-0.0,
        0.70302389911323138,0.00031109412840517781,-0.0095453969112158227,-1.2662726753574506E-5,0.0,0.0,0.0,0.0,
        0.0,0.0,0.0,0.0,-0.0,-0.0,-0.0,-0.0,-0.0,-0.0,-1.0,-0.0,-0.022268586633886586,2.3917602785793205E-5,
        0.0095453969112158227,-1.2662726753574504E-5,0.0,0.0,0.0,0.0,0.0,0.0,1.0,-0.0,-0.0,-0.0,-0.0,-0.0,-0.0,-0.0,
        -1.9698806952807862E-5,-0.70302389911363883,0.0095453969112132882,0.00051827808005669451,0.0,0.0,0.0,0.0,
        0.0,0.0,1.0,0.0,-0.0,-0.0,-0.0,-0.0,-0.0,-0.0,-0.0,-0.0,-0.0095453965888427916,-1.2662731263161793E-5,
        -9.5513929494329763E-5,-1.4093315727616534E-8,0.0031846506656924463,0.0,0.0,0.0,0.0,0.0,0.0,0.0,0.0,0.0,
        -0.0,-0.0,-0.0,-0.0,-0.0,-0.0,-0.022268586633861689,2.8128779299660836E-5,0.00954539691120452,
        -2.3917602785793216E-5,0.0,0.0,0.0,0.0,0.0,0.0,1.0,-0.0,-0.0,-0.0,-0.0,-0.0,-0.0,-0.0,
        -0.0095453969112207285,-3.1846509886793804E-5,1.5477792152379083E-5,-2.81643067314548E-6,0.0,0.0,0.0,0.0,
        0.0,0.0,1.0,0.0,0.0,-0.0,-0.0,-0.0,-0.0,-0.0,-0.0,-0.0,-0.0,-0.0095453969112158244,-6.3667426064645748E-5,
        1.1964809706348631E-7,-1.2662732240991401E-5,0.0,0.0,0.0,0.0,0.0,0.0,1.0,0.0,-0.0,-0.0,-0.0,-0.0,-0.0,-0.0,
        -0.0,-0.0095453965888404185,-0.70302132668456918,1.5477790827995437E-5,0.703023899155877,
        -0.00062190510862303544,0.0,0.0,0.0,0.0,0.0,0.0,0.0,0.0,-0.0,-0.0,-0.0,-0.0,-0.0,-0.0,-0.0,
        -2.6726087145381383E-5,0.70302389911330532,1.2662726610908526E-5,0.00031109412840517521,
        -0.0095453969112151774,0.0,0.0,0.0,0.0,0.0,0.0,0.0,-0.0,-0.0,-1.0,-0.0,-2.6726097733171875E-5,
        0.01272756092550296,0.70302198987128661,1.2662729900309186E-5,0.00031109440605359812,-0.70301996014529189,
        0.0,0.0,0.0,0.0,0.0,-0.0,-0.0,-0.0,-0.0,-0.0,-0.0,-0.0,-1.2662732098325213E-5,-7.0421936123401543E-8,
        0.0095453969112224528,6.3667426064685376E-5,1.4093318379358016E-6,0.0,0.0,0.0,0.0,0.0,0.0,0.0,-0.0,-0.0,
        -0.0,-0.0,-0.0,-1.0,-0.0,-1.4093313394933583E-8,0.00954539691121582,6.3667426064645857E-5,
        1.2662732240991394E-5,0.0,0.0,0.0,0.0,0.0,0.0,0.0,-0.0,-0.0,-0.0,-0.0,-0.0,-0.0,-1.0,-0.0,-0.0,
        -0.0003110932691485688,0.0318011449624135,1.2662717356786933E-5,-0.022268586633886613,0.0,0.0,0.0,0.0,0.0,
        0.0,0.0,-0.0,-0.0,-0.0,-0.0,-0.0,-0.0,-1.0,-0.0,-1.2662726753574494E-5,-1.4093297863266229E-8,
        3.184650505364419E-5,-0.0095453969112231033,0.0,0.0,0.0,0.0,0.0,0.0,0.0,0.0,0.0,-0.0,-0.0,-0.0,-0.0,-0.0,
        -0.0,-1.0,-1.2662726753574494E-5,-3.1846505053644244E-5,-1.4093297863266219E-8,0.0095453969112230981,0.0,
        0.0,0.0,0.0,0.0,0.0,1.0,0.0,0.0,-0.0,-0.0,-0.0,-0.0,-0.0,-0.0,-0.70302389911309171,1.5477784653254034E-5,
        0.009545396911220725,-0.00062190474080434219,0.0,0.0,0.0,0.0,0.0,0.0,1.0,0.0,-0.0,-0.0,-0.0,-0.0,-0.0,-0.0,
        -0.0,-0.0,-0.00031109440605359866,0.012727560925503811,1.2662730042975288E-5,-0.703019960145122,0.0,0.0,0.0,
        0.0,0.0,0.0,1.0,0.0,-0.0,-0.0,-0.0,-0.0,-0.0,-0.0,-0.0,-0.0,-0.00011139879369970853,1.2662726753574502E-5,
        5.6328578923948216E-8,0.0095453969112230981,0.0,0.0,0.0,0.0,0.0,0.0,1.0,-0.0,-0.0,-0.0,-0.0,-0.0,-0.0,-0.0,
        -0.0,-1.266272661090853E-5,-0.00051827808005669429,-0.70302389911304008,0.0095453969112224545,
        0.0003110942227687848,0.0,0.0,0.0,0.0,0.0,0.0,1.0,0.0,-0.0,-0.0,-0.0,-0.0,-0.0,-0.0,-0.028625312287031243,
        1.5477783328870845E-5,0.0095453965888404081,0.70302389911309171,-0.0006219046642527053,0.0,0.0,0.0,0.0,0.0,
        0.0,0.0,-0.0,-0.0,-0.0,-0.0,-0.0,-0.0,-0.0,-0.00031109412840517629,0.70302389911323138,
        1.2662726753574499E-5,-0.0095453969112158261,0.0,0.0,0.0,0.0,0.0,0.0,0.0,0.0,-0.0,-0.0,-0.0,-0.0,-0.0,-0.0,
        -1.0,-0.0,3.6522249178886062E-5,0.019093388890196454,5.2157458590361115E-5,0.031805094384842234,
        -3.6522249178886062E-5,-0.019093388890196454,-5.2157458590361115E-5,-0.031805094384842227,0.0,0.0,0.0,0.0,
        0.0,0.0,0.0,1.0,-0.0,-0.0,-0.0,-0.0,-0.0,-0.0,-0.0,-1.0,-3.6522249178886062E-5,0.019093388890364354,
        0.00096130880269788594,0.00086525886760264287,0.031805094385131148,-0.019093388890364354,
        -0.031805094385131141,0.0,0.0,0.0,0.0,0.0,0.0,1.0,0.0,-0.0,-0.0,-0.0,-0.0,-0.0,-0.0,-0.0,-1.0,
        -0.019093388890196458,3.652233705213242E-5,0.70301893050798425,5.2157599879956529E-5,0.70301941044164273,
        -3.652233705213242E-5,-5.2157599879956529E-5,0.0,0.0,0.0,0.0,0.0,0.0,0.0,0.0,-0.0,-0.0,-0.0,-0.0,-0.0,-0.0,
        -0.0,-1.0,-5.2157458590361109E-5,2.8693453280709772E-5,0.019093388890325125,4.43447971709128E-5,
        -0.0318050943850639,0.0,0.0,0.0,0.0,0.0,0.0,0.0,-0.0,-0.0,-0.0,-0.0,-0.0,-0.0,-1.0,-0.0,
        3.6522249178886062E-5,0.019093388890364354,0.031805094385131148,-0.019093388890364354,
        -0.00096130880269788594,-0.00086525886760264342,-0.031805094385131141,0.0,0.0,0.0,0.0,0.0,0.0,0.0,1.0,-0.0,
        -0.0,-0.0,-0.0,-0.0,-0.0,-1.0,-0.0,0.019093388890196458,3.652233705213242E-5,5.2157599879956529E-5,
        -3.652233705213242E-5,-0.70301893050798425,-5.2157599879956529E-5,-0.70301941044164273,0.0,0.0,0.0,0.0,0.0,
        0.0,0.0,1.0,-0.0,-0.0,-0.0,-0.0,-0.0,-0.0,-0.0,-0.0,5.2157458590361109E-5,0.019093388890325125,
        0.03180509438506391,-0.019093388890325125,-4.43447971709128E-5,-0.0318050943850639,0.0,0.0,0.0,0.0,0.0,0.0,
        1.0,-0.0,-0.0,-0.0,-0.0,-0.0,-0.0,-0.0,-1.0,0.031805094384842234,3.6522333405210253E-5,
        -4.9555278001043236E-5,-0.022271948633834655,-5.2157594188888043E-5,0.0,0.0,0.0,0.0,0.0,0.0,0.0,-0.0,-0.0,
        -0.0,-0.0,-0.0,-0.0,-0.0,-1.0,-3.6522337052132434E-5,-0.019093388890364351,0.00096131182465395966,
        0.703018930505452,0.00086526182234124684,0.0,0.0,0.0,0.0,0.0,0.0,0.0,0.0,-0.0,-0.0,-0.0,-0.0,-0.0,-0.0,-0.0,
        -1.0,-0.00086525886760264266,-2.3473029391852623E-5,0.019093388890394088,0.0318050943851825,
        -0.019093388890394088,-0.031805094385182496,0.0,0.0,0.0,0.0,0.0,0.0,0.0,1.0,0.0,-0.0,-0.0,-0.0,-0.0,-0.0,
        -0.0,-1.0,-3.6522337052132434E-5,-0.0,-2.3473075971598973E-5,0.019093388890392377,0.00057718804917542433,
        -0.70301893050485509,0.0,0.0,0.0,0.0,0.0,0.0,1.0,0.0,-0.0,-0.0,-0.0,-0.0,-0.0,-0.0,-0.0,
        -3.652233340521026E-5,0.031805094385131134,0.00096131171151488386,0.00086526170925901034,
        -0.022271948634027636,0.0,0.0,0.0,0.0,0.0,0.0,0.0,-0.0,-0.0,-0.0,-0.0,-0.0,-0.0,-0.0,-1.0,
        -0.00954717826758235,-0.70301893050798414,3.65223604939942E-5,5.2157637599480248E-5,0.70302082402767729,
        -3.65223604939942E-5,-5.2157637599480248E-5,0.0,0.0,0.0,0.0,0.0,0.0,0.0,0.0,-0.0,-0.0,-0.0,-0.0,-0.0,-0.0,
        -0.019093388890364354,-0.00096131182465395966,-1.0,-0.00954717859018078,3.6522363302599261E-5,0.0,0.0,0.0,
        0.0,0.0,0.0,0.0,1.0,0.0,-0.0,-0.0,-0.0,-0.0,-0.0,-0.0,-0.0,-0.019093388890325125,5.2157599879956516E-5,
        0.70301893050571762,0.70301941043955929,-4.43449011383923E-5,0.0,0.0,0.0,0.0,0.0,0.0,0.0,-0.0,-0.0,-0.0,
        -0.0,-0.0,-0.0,-0.0,-1.0,-0.00057718837020061448,-0.70302082398273624,2.3473084657567242E-5,
        0.0095471785901811157,0.0,0.0,0.0,0.0,0.0,0.0,0.0,1.0,-0.0,-0.0,-0.0,-0.0,-0.0,-0.0,-0.0,
        3.6522337052132434E-5,0.019093388890364351,-0.703018930505452,-0.00086526182234124727,-0.7030194104393207,
        0.0,0.0,0.0,0.0,0.0,0.0,0.0,1.0,-0.0,-0.0,-0.0,-0.0,-0.0,-0.0,-0.0,-0.0,2.347302912727454E-5,
        0.00096130880269788583,0.019093388890392381,-0.00057718529603716312,0.0,0.0,0.0,0.0,0.0,0.0,-0.0,-0.0,-0.0,
        -0.0,-0.0,-0.0,-1.0,-0.0,-0.0,3.652233340521026E-5,0.031805094385131134,-0.00096131171151488386,
        -0.022271948634027636,-0.00086526170925901077,0.0,0.0,0.0,0.0,0.0,0.0,0.0,-0.0,-0.0,-0.0,-0.0,-0.0,-0.0,
        -1.0,-0.0,0.0095471785901624015,-1.0,0.019093388890325125,5.2157599879956516E-5,-4.43449011383923E-5,0.0,
        0.0,0.0,0.0,0.0,0.0,1.0,-0.0,-0.0,-0.0,-0.0,-0.0,-0.0,-0.0,-0.0,0.012729738255777539,3.6522358297177071E-5,
        5.2157634143092755E-5,-3.6522358297177071E-5,-0.70301795752567109,-5.2157634143092755E-5,0.0,0.0,0.0,0.0,
        0.0,0.0,0.0,1.0,-0.0,-0.0,-0.0,-0.0,-0.0,-0.0,-0.0,-0.0,0.00057718512122799316,0.019093388890365336,
        0.031805094385133209,-2.3473029391852627E-5,-0.019093388890365336,-0.0318050943851332,0.0,0.0,0.0,0.0,0.0,
        0.0,1.0,0.0,-0.0,-0.0,-0.0,-0.0,-0.0,-0.0,-0.0,-1.0,5.2157594188888036E-5,0.0318050943850639,
        -4.4344896978036783E-5,-0.022271948633982117,0.0,0.0,0.0,0.0,0.0,0.0,-0.0,-0.0,-0.0,-0.0,-0.0,-0.0,-0.0,
        -1.0,0.022271948633834648,3.6522353054843289E-5,5.2157625694692722E-5,-3.6522353054843289E-5,
        -0.009547178590102354,-5.2157625694692722E-5,0.0,0.0,0.0,0.0,0.0,0.0,0.0,-0.0,-0.0,-0.0,-0.0,-0.0,-0.0,-0.0,
        -1.0,-2.3473075971598973E-5,-0.019093388890392377,-0.00096131182465395988,0.70301893050485509,
        0.00057718804917542433,0.0,0.0,0.0,0.0,0.0,0.0,-0.703018930504855,-3.6522363302599275E-5,
        -0.009547178590180774,0.00096131273359152409,0.0,0.0,0.0,0.0,0.0,0.0,1.0,0.0,0.0,-0.0,-0.0,-0.0,-0.0,-0.0,
        -0.0,-0.0,-0.000865261709259011,-2.3473074125247875E-5,0.031805094385182496,-0.02227194863406157,0.0,0.0,
        0.0,0.0,0.0,0.0,0.0,0.0,-0.0,-0.0,-0.0,-0.0,-0.0,-0.0,-1.0,-3.6522363302599275E-5,0.009547178590180774,
        0.70301795752274809,0.00096131273359152409,0.00086526270890343563,0.0,0.0,0.0,0.0,0.0,0.0,0.0,-0.0,-0.0,
        -0.0,-0.0,-0.0,-0.0,-0.0,-1.0,-0.0,-3.6522353054843289E-5,0.022271948634027618,0.00096131238304662065,
        0.00086526236509131883,-0.0095471785901807826,0.0,0.0,0.0,0.0,0.0,0.0,0.0,-0.0,-0.0,-0.0,-0.0,-0.0,-0.0,
        -0.0,-1.0,-0.028629066348924127,3.6522350246238987E-5,0.0095471782675823486,5.2157621136234768E-5,
        0.70302082398458909,-3.6522350246238987E-5,-5.2157621136234768E-5,0.0,0.0,0.0,0.0,0.0,0.0,0.0,-0.0,-0.0,
        -0.0,-1.0,-0.0,-0.009547178590102354,-3.18484920381726E-5,3.6522363302599268E-5,5.2157642157939449E-5,
        -3.6522363302599268E-5,-5.2157642157939449E-5,0.0,0.0,0.0,0.0,0.0,0.0,0.0,1.0,0.0,-0.0,-0.0,-0.0,-0.0,-0.0,
        -0.0,-0.0,-0.0095471782676424029,-0.70301893050571751,5.2157637599480228E-5,0.70302082402620258,
        -4.43449289708158E-5,0.0,0.0,0.0,0.0,0.0,0.0,0.0,-0.0,-0.0,-0.0,-0.0,-0.0,-0.0,-0.019093388890386278,
        2.8693514412082078E-5,0.000865261822341247,0.70301893050493458,-0.001153449694857952,0.0,0.0,0.0,0.0,0.0,
        -1.0,-0.0,-0.019093388890365333,0.0005771878743661479,0.703018930505132,0.703019410439022,
        -2.347307623617832E-5,0.0,0.0,0.0,0.0,0.0,0.0,0.0,0.0,-0.0,-0.0,-0.0,-0.0,-0.0,-0.0,-0.0,-1.0,
        -4.9555306757672129E-5,-0.7030208239827761,2.3473084392987648E-5,0.0095471785901803125,
        0.00057718837020061221,0.0,0.0,0.0,0.0,0.0,0.0,1.0,-0.0,-0.0,-0.0,-0.0,-0.0,-0.0,-0.0,-0.028629066349182733,
        -0.00057718828009965415,2.3473083193394028E-5,0.00954717826766111,0.70302082398273624,0.0,0.0,0.0,0.0,0.0,
        0.0,0.0,-0.0,-0.0,-0.0,-0.0,-0.0,-0.0,-0.0,-2.3473084657567229E-5,-2.6146252961331178E-8,
        -3.1848487202701323E-5,0.0095471785901946049,0.0,0.0,0.0,0.0,0.0,0.0,0.0,1.0,0.0,-0.0,-0.0,-0.0,-0.0,-0.0,
        -0.0,-0.0,2.8693514412082092E-5,0.019093388890386278,0.00086526182234124673,-0.0011534496948579533,
        -0.70301893050493458,0.0,0.0,0.0,0.0,0.0,0.0,1.0,-0.0,-0.0,-0.0,-0.0,-0.0,-0.0,-0.0,-0.0,
        3.6522358297177077E-5,0.012729738255884648,0.7030194104393207,-0.7030179575227482,-0.00086526254243436229,
        0.0,0.0,0.0,0.0,0.0,0.0,0.0,-0.0,-0.0,-0.0,-0.0,-0.0,-0.0,-0.0,4.9555154326319392E-5,0.019093388890363633,
        -0.019093388890363633,-0.00057718512122799338,-0.031805094385130267,0.0,0.0,0.0,0.0,0.0,0.0,0.0,1.0,-0.0,
        -0.0,-0.0,-0.0,-0.0,-0.0,-1.0,-0.0,0.0095471785901946014,-1.0,2.347307623617832E-5,0.019093388890394081,0.0,
        0.0,0.0,0.0,0.0,0.0,1.0,-0.0,-0.0,-0.0,-0.0,-0.0,-0.0,-0.0,-0.0,-0.0,3.6522353054843289E-5,
        0.022271948634027618,-0.0095471785901807826,-0.00096131238304662065,-0.00086526236509131937,0.0,0.0,0.0,0.0,
        0.0,0.0,0.0,-0.0,-0.0,-0.0,-0.0,-0.0,-0.0,-1.0,-0.0,2.869351178855761E-5,0.031805094385168986,
        -0.012729738255898576,-0.0011534495816052015,-0.022271948634052637,0.0,0.0,0.0,0.0,0.0,0.0,0.0,-0.0,-0.0,
        -0.0,-0.0,-0.0,-0.0,-1.0,-0.0,5.2157625694692715E-5,0.70302082398311461,-0.009547178590162405,
        -4.4344920231689462E-5,0.0,0.0,0.0,0.0,0.0,0.0,0.0,-0.0,-0.0,-0.0,-0.0,-0.0,-0.0,-0.0,-1.0,
        0.0095471785901023523,6.3675350751752718E-5,3.6522363302599268E-5,5.2157642157939449E-5,
        -3.6522363302599268E-5,-5.2157642157939449E-5,0.0,0.0,0.0,0.0,0.0,0.0,0.0,-0.0,-0.0,-0.0,-0.0,-0.0,-0.0,
        -0.0,-1.0,-0.0,0.0095471782676424029,5.2157637599480228E-5,-4.43449289708158E-5,-0.7030208240262027,0.0,0.0,
        0.0,0.0,0.0,0.0,1.0,-0.0,-0.0,-0.0,-0.0,-0.0,-0.0,-0.0,-0.0,0.00954717859018111,6.3675350752329378E-5,
        2.61462557358624E-8,-2.3473090146008748E-5,0.0,0.0,0.0,0.0,0.0,0.0,0.0,-0.0,-0.0,-0.0,-0.0,-0.0,-0.0,-0.0,
        -1.0,-0.0,0.019093388890365333,0.0005771878743661479,-2.347307623617832E-5,-0.703018930505132,0.0,0.0,0.0,
        0.0,0.0,0.0,1.0,0.0,-0.0,-0.0,-0.0,-0.0,-0.0,-0.0,-0.0,-0.0,2.3473029391852623E-5,0.00057718529603716518,
        0.019093388890394088,0.0318050943851825,-0.019093388890394088,-0.031805094385182496,0.0,0.0,0.0,0.0,0.0,0.0,
        1.0,-0.0,-0.0,-0.0,-0.0,-0.0,-0.0,-0.0,-1.0,-0.0,-5.2157625694692715E-5,0.02227194863398212,
        2.8693525502607085E-5,4.4344920231689462E-5,-0.009547178590162405,0.0,0.0,0.0,0.0,0.0,0.0,0.0,-0.0,-0.0,
        -0.0,-0.0,-0.0,-0.0,-1.0,-0.019093388890363633,-4.9555283182156878E-5,2.3473075971598956E-5,
        0.70301893050519171,0.00057718787436614454,0.0,0.0,0.0,0.0,0.0,0.0,-0.019093388890394081,-1.0,
        -2.3473090146008764E-5,-0.0095471785901946014,0.0,0.0,0.0,0.0,0.0,0.0,0.0,1.0,0.0,0.0,-0.0,-0.0,-0.0,-0.0,
        -0.0,-0.0,-3.6522350246238994E-5,-0.028629066349181113,0.0095471782676607771,0.00096131228402486523,
        0.70302082398295684,0.0,0.0,0.0,0.0,0.0,0.0,0.0,-0.0,-0.0,-0.0,-1.0,-4.4344797170912778E-5,
        2.3473029391852627E-5,0.019093388890365336,0.031805094385133209,-0.019093388890365336,-0.0318050943851332,
        0.0,0.0,0.0,0.0,0.0,0.0,0.0,1.0,-0.0,-0.0,-0.0,-0.0,-0.0,-0.0,-1.0,-2.3473076236178317E-5,
        -2.6146230500341689E-8,0.019093388890394081,-0.70301893050479525,-0.70301941043871474,0.0,0.0,0.0,0.0,0.0,
        0.0,0.0,1.0,0.0,-0.0,-0.0,-0.0,-0.0,-0.0,-1.0,-0.0,-0.0,-5.2157594188888036E-5,0.0318050943850639,
        2.8693511788557617E-5,4.4344896978036783E-5,-0.022271948633982117,0.0,0.0,0.0,0.0,0.0,0.0,0.0,-0.0,-0.0,
        -0.0,-0.0,-0.0,-0.0,-1.0,-2.8693525502607071E-5,-0.00086526236509131948,0.022271948634052637,
        0.0011534502845418316,-0.0095471785901909984,0.0,0.0,0.0,0.0,0.0,0.0,0.0,-0.0,-0.0,-0.0,-0.0,-0.0,-0.0,-1.0,
        -4.9555283182156878E-5,0.019093388890363629,2.3473075971598956E-5,0.00057718787436614584,
        -0.70301893050519171,0.0,0.0,0.0,0.0,0.0,0.0,1.0,-0.0,-0.0,-0.0,-0.0,-0.0,-0.0,-0.0,-3.6522358297177077E-5,
        0.012729738255884648,0.7030194104393207,0.00096131256263816563,-0.7030179575227482,0.0,0.0,0.0,0.0,0.0,0.0,
        -0.0,-0.0,-0.0,-1.0,-0.0,-2.3473090146008754E-5,0.0095471785901946,0.0,0.0,0.0,0.0,0.0,0.0,0.0,0.0,-0.0,
        -0.0,-0.0,-0.0,-0.0,-0.0,-1.0,-0.0,-0.7030208239845892,3.6522353054843289E-5,0.00954717859010235,
        5.2157625694692722E-5,-3.6522353054843289E-5,-5.2157625694692722E-5,0.0,0.0,0.0,0.0,0.0,0.0,0.0,1.0,-0.0,
        -0.0,-0.0,-0.0,-0.0,-0.0,-0.0,-0.0,-0.028629066349181113,3.6522350246238987E-5,0.0095471782676607771,
        0.70302082398295684,-0.0008652622683001951,0.0,0.0,0.0,0.0,0.0,0.0,0.0,-0.0,-0.0,-0.0,-0.0,-0.0,-0.0,-0.0,
        -0.028629066349226677,2.3473083193394021E-5,0.0011534501810579545,0.0095471782676746046,0.70302082398252286,
        0.0,0.0,0.0,0.0,0.0,0.0,-0.0,-0.0,-0.0,-1.0,-0.0,-0.0095471785901624015,-3.184849203842196E-5,
        1.7403678606755017E-7,-4.434493230781362E-5,0.0,0.0,0.0,0.0,0.0,0.0,1.0,0.0,-0.0,-0.0,-0.0,-0.0,-0.0,-0.0,
        -0.0,-0.0095471782676709964,-0.70301893050493447,2.8693530706110979E-5,0.00086526261211228468,
        0.70302082402570232,-0.0011534505450709808,0.0,0.0,0.0,0.0,0.0,0.0,-0.0,-0.0,-0.0,-0.0,-0.0,-0.0,-0.0,
        -0.0286290663491211,5.2157621136234754E-5,0.0095471782676424012,0.7030208239831145,-4.4344916894692544E-5,
        0.0,0.0,0.0,0.0,0.0,0.0,-0.0,-0.0,-0.0,-1.0,-0.00954717826766111,-0.70301893050513187,
        0.00057718860371856837,0.70302082402582433,-2.347308868183514E-5,0.0,0.0,0.0,0.0,0.0,0.0,0.0,0.0,-0.0,-0.0,
        -0.0,-0.0,-0.0,-0.0,-0.019093388890394081,2.347307623617831E-5,1.0445958483366056E-7,0.70301893050479525,
        0.70301941043871474,0.0,0.0,0.0,0.0,0.0,0.0,0.0,-0.0,-0.0,-0.0,-0.0,-0.0,-0.0,-0.0,-1.0,-0.0,
        -4.9555302606141827E-5,-0.028629066349180127,2.3473082928814485E-5,0.0095471782676603088,
        0.00057718828009965177,0.7030208239827761,0.0,0.0,0.0,0.0,0.0,0.0,-0.0,-0.0,-0.0,-0.0,-0.0,-0.0,
        -0.0095471785901803073,-4.9555321759358343E-5,-0.7030208240258643,2.3473089881429021E-5,
        0.00057718869381955288,0.0,0.0,0.0,0.0,0.0,0.0,1.0,0.0,-0.0,-0.0,-0.0,-0.0,-0.0,-0.0,-0.000577187874366147,
        0.019093388890365333,2.347307623617832E-5,-0.703018930505132,-0.703019410439022,0.0,0.0,0.0,0.0,0.0,0.0,0.0,
        1.0,-0.0,-0.0,-0.0,-0.0,-0.0,-0.0,-0.0,-2.3473083193394021E-5,-0.028629066349226677,-0.00057718845490894847,
        0.0095471782676746046,0.70302082398252286,0.0,0.0,0.0,0.0,0.0,0.0,0.0,0.0,-0.0,-0.0,-0.0,-0.0,-0.0,-0.0,
        -0.70302082398295673,3.6522353054843289E-5,0.0095471785901807826,-0.0008652623650913197,0.0,0.0,0.0,0.0,0.0,
        0.0,0.0,1.0,-0.0,-0.0,-0.0,-0.0,-0.0,-0.0,-0.0,-0.0,-2.3473084392987658E-5,0.00057718854500991032,
        -3.6522353054843289E-5,-0.70302082398295684,0.0095471785901807861,0.0,0.0,0.0,0.0,0.0,0.0,1.0,0.0,-0.0,-0.0,
        -0.0,-0.0,-0.0,-0.0,-0.0,-0.0,2.8693532638693606E-5,0.0,-0.0095471785901946049,2.3473090146008737E-5,0.0,
        0.0,0.0,0.0,0.0,0.0,1.0,0.0,-0.0,-0.0,-0.0,-0.0,-0.0,-0.0,-0.0,-0.0,3.6522363302599275E-5,
        0.009547178590180774,0.70301795752274809,-0.00096131273359152409,-0.00086526270890343617,0.0,0.0,0.0,0.0,
        0.0,0.0,0.0,-0.0,-0.0,-0.0,-0.0,-0.0,-0.0,-1.0,-0.0,-0.0,2.3473084657567229E-5,1.044596382372305E-7,
        3.1848487202701255E-5,-0.0095471785901946049,0.0,0.0,0.0,0.0,0.0,0.0,0.0,-0.0,-0.0,-0.0,-0.0,-0.0,-0.0,-0.0,
        -1.0,-0.0,2.8693529139888997E-5,0.012729738255898571,0.703019410438843,-0.0011534504686312259,
        -0.703017957522159,0.0,0.0,0.0,0.0,0.0,0.0,0.0,-0.0,-0.0,-0.0,-0.0,-0.0,-0.0,-0.0,-0.0,0.0286290663491211,
        5.2157621136234754E-5,-0.0095471782676424012,0.0,0.0,0.0,0.0,0.0,0.0,0.0,-0.0,-0.0,-0.0,-0.0,-0.0,-0.0,-0.0,
        -1.0,-0.0,-1.7403678606755019E-7,0.0095471785901624015,2.869353263869362E-5,4.43449323078136E-5,0.0,0.0,0.0,
        0.0,0.0,0.0,0.0,-0.0,-0.0,-0.0,-0.0,-0.0,-0.0,-1.0,-0.0,0.00057718837020061568,0.70302082398273624,
        -2.3473084657567242E-5,-0.00954717859018112,0.0,0.0,0.0,0.0,0.0,0.0,0.0,0.0,-0.0,-0.0,-0.0,-0.0,-0.0,-0.0,
        -0.0,-1.0,-4.4344920231689448E-5,0.022271948634028347,2.3473084657567242E-5,-0.00954717859018111,0.0,0.0,
        0.0,0.0,0.0,0.0,0.0,-0.0,-0.0,-0.0,-0.0,-0.0,-0.0,-1.0,-0.019093388890365333,-0.00057718787436614671,
        2.347307623617832E-5,0.703018930505132,0.0,0.0,0.0,0.0,0.0,0.0,0.0,0.0,-0.0,-0.0,-0.0,-0.0,-0.0,-0.0,-1.0,
        -0.0,-2.3473089881429038E-5,-0.0095471785901937965,-1.3060593352310909E-7,-3.1848492038550092E-5,
        2.6146264969321444E-6,0.0,0.0,0.0,0.0,0.0,0.0,1.0,0.0,0.0,-0.0,-0.0,-0.0,-0.0,-0.0,-0.0,
        -4.4344896978036769E-5,0.0318050943851332,2.3473074125247868E-5,-0.02227194863402835,0.0,0.0,0.0,0.0,0.0,
        0.0,0.0,-0.0,-0.0,-0.0,-0.0,-0.0,-0.0,-1.0,-2.3473087461600324E-5,-2.6146260689378505E-8,
        0.012729738255903513,-0.0031837672149024575,0.0,0.0,0.0,0.0,0.0,0.0,0.0,1.0,0.0,-0.0,-0.0,-0.0,-0.0,-0.0,
        -1.0,-0.0,-0.0,-2.3473084657567235E-5,-1.0445963823723051E-7,0.00011141562924503268,-0.0095471785901946014,
        0.0,0.0,0.0,0.0,0.0,0.0,0.0,0.0,-0.0,-0.0,-0.0,-0.0,-0.0,-0.0,-1.0,-2.3473087197020675E-5,
        -0.00096131256263816585,0.012729738255902429,0.00057718871560916,-0.70301795752206764,0.0,0.0,0.0,0.0,0.0,
        0.0,1.0,0.0,-0.0,-0.0,-0.0,-0.0,-0.0,-0.0,-0.0,-0.028629066349182733,0.00057718828009965676,
        0.00954717826766111,0.70302082398273624,-2.3473083193394035E-5,0.0,0.0,0.0,0.0,0.0,0.0,0.0,-0.0,-0.0,-0.0,
        -1.0,-0.028629066349214694,2.8693523570024966E-5,0.0008652622683001951,0.0095471782676709929,
        0.70302082398261434,-0.0011534501810579526,0.0,0.0,0.0,0.0,0.0,-0.0,-0.0,-0.0,-0.0,-0.0,-0.0,-0.0,
        -0.0095471782676746011,-9.5523836332220613E-5,2.3473088681835134E-5,1.0445966183159716E-7,
        0.0031848488808076322,0.0,0.0,0.0,0.0,0.0,0.0,0.0,-0.0,-0.0,-0.0,-0.0,-0.0,-0.0,-0.0,-3.1848487202701309E-5,
        2.3473084657567225E-5,1.0445963823723051E-7,0.0095471785901946014,0.0,0.0,0.0,0.0,0.0,0.0,1.0,-0.0,-0.0,
        -0.0,-0.0,-0.0,-0.0,-0.0,-0.0,-0.0,-0.70302082398311461,5.2157625694692715E-5,0.009547178590162405,
        -4.4344920231689462E-5,0.0,0.0,0.0,0.0,0.0,0.0,1.0,-0.0,-0.0,-0.0,-0.0,-0.0,-0.0,-0.0,-0.0,
        -0.0095471785901811122,-3.1848492038499474E-5,2.6146255735862374E-8,-2.3473090146008754E-5,0.0,0.0,0.0,0.0,
        0.0,0.0,1.0,0.0,0.0,-0.0,-0.0,-0.0,-0.0,-0.0,-0.0,-0.0,-0.00954717859018111,-2.61462557358624E-8,
        -3.1848492038499446E-5,2.3473090146008748E-5,0.0,0.0,0.0,0.0,0.0,0.0,0.0,1.0,0.0,-0.0,-0.0,-0.0,-0.0,-0.0,
        -0.0,-0.00057718854079985679,0.012729738255885078,2.347308746160033E-5,-0.70301795752239227,0.0,0.0,0.0,0.0,
        0.0,0.0,0.0,1.0,-0.0,-0.0,-0.0,-0.0,-0.0,-1.0,-0.0,-0.0,-0.70302082398261434,2.8693525502607068E-5,
        0.0095471785901909967,-0.0011534502845418292,0.0,0.0,0.0,0.0,0.0,0.0,0.0,1.0,-0.0,-0.0,-0.0,-0.0,-0.0,-0.0,
        -0.0,-0.0,-2.2183590036490517E-7,0.00954717859018111,6.3675350752329338E-5,2.3473090146008754E-5,0.0,0.0,
        0.0,0.0,0.0,0.0,0.0,-0.0,-0.0,-0.0,-0.0,-0.0,-0.0,-1.0,-0.0,-0.00954717826766111,-0.70301893050513187,
        -0.00057718860371856881,2.3473088681835137E-5,0.70302082402582433,0.0,0.0,0.0,0.0,0.0,0.0,0.0,0.0,-0.0,-0.0,
        -0.0,-0.0,-0.0,-0.0,-4.9555314435549588E-5,0.012729738255883995,2.3473087197020668E-5,
        0.00057718854079985842,-0.70301795752246,0.0,0.0,0.0,0.0,0.0,0.0,1.0,-0.0,-0.0,-0.0,-0.0,-0.0,-0.0,-0.0,
        -0.70302082398273635,0.00057718837020061676,0.0095471785901811157,-2.3473084657567235E-5,0.0,0.0,0.0,0.0,
        0.0,0.0,1.0,0.0,-0.0,-0.0,-0.0,-0.0,-0.0,-0.0,-0.0,-0.0,0.9996312291726841,-4.600588354065297E-9,
        0.99897637109654081,-7.9312879089261515E-9,-0.9996312291726841,4.600588354065297E-9,-0.99897637109654081,
        7.9312879089261531E-9,0.0,0.0,0.0,0.0,0.0,0.0,0.0,0.0,-0.0,-0.0,-0.0,-0.0,-0.0,-0.0,-0.0,-0.0,
        -0.99963122917268421,8.2687665553021133E-25,0.0,0.0,1.6526715295000529E-24,-8.2687665553021133E-25,0.0,0.0,
        0.0,0.0,0.0,0.0,0.0,0.0,1.0,-0.0,-0.0,-0.0,-0.0,-0.0,-0.0,-0.0,-0.0,4.600588354065297E-9,
        0.99963122917267422,-1.8067389175382345E-7,0.9989763710965166,-1.8418939393988118E-7,-0.99963122917267422,
        -0.9989763710965166,0.0,0.0,0.0,0.0,0.0,0.0,0.0,0.0,-0.0,-0.0,-0.0,-0.0,-0.0,-0.0,-0.0,-0.0,
        -0.99897637109654069,0.99983610538248957,-2.1332465124273696E-9,0.99949819932039374,3.6722326320306744E-9,
        0.0,0.0,0.0,0.0,0.0,0.0,0.0,-0.0,-0.0,-0.0,-0.0,-0.0,-0.0,-0.0,-0.0,0.99963122917268421,
        8.2687665553021133E-25,1.6526715295000529E-24,-8.2687665553021133E-25,0.0,0.0,0.0,0.0,0.0,0.0,0.0,0.0,0.0,
        0.0,0.0,-0.0,-0.0,-0.0,-0.0,-0.0,-0.0,-0.0,-1.0,-4.600588354065297E-9,0.99963122917267422,
        0.9989763710965166,-0.99963122917267422,1.8067389175382345E-7,-0.9989763710965166,1.8418939393988137E-7,0.0,
        0.0,0.0,0.0,0.0,0.0,0.0,0.0,-0.0,-0.0,-0.0,-0.0,-0.0,-0.0,-0.0,-0.0,0.99897637109654069,
        -2.1332465124273696E-9,-3.6722326320306728E-9,2.1332465124273696E-9,-0.99949819932039374,
        3.6722326320306744E-9,0.0,0.0,0.0,0.0,0.0,0.0,0.0,-0.0,-0.0,-0.0,-0.0,-0.0,-0.0,-0.0,-0.0,
        -7.9312879089261548E-9,0.99963122917267511,-0.9991706919990635,5.2901915156994029E-9,-0.99897637109651882,
        0.0,0.0,0.0,0.0,0.0,0.0,0.0,-0.0,-0.0,-0.0,-0.0,-0.0,-0.0,-0.0,-0.0,-0.99963122917267433,
        -1.6537533110604227E-24,0.0,0.0,0.0,0.0,0.0,0.0,0.0,0.0,0.0,1.0,0.0,-0.0,-0.0,-0.0,-0.0,-0.0,-0.0,-0.0,-0.0,
        6.1283679523231971E-15,-0.99990781756998193,8.2687665553020968E-25,1.6526715295000437E-24,
        -8.2687665553020968E-25,0.0,0.0,0.0,0.0,0.0,0.0,0.0,0.0,0.0,1.0,-0.0,-0.0,-0.0,-0.0,-0.0,-0.0,-0.0,
        -0.99963122917267433,-0.0,-0.99990781757620562,1.6537533110604194E-24,0.0,0.0,0.0,0.0,0.0,0.0,0.0,0.0,0.0,
        1.0,-0.0,-0.0,-0.0,-0.0,-0.0,-0.0,-0.0,-0.99963122917267522,0.0,0.0,0.0,-4.9605957844188972E-24,0.0,0.0,0.0,
        0.0,0.0,0.0,1.0,-0.0,-0.0,-0.0,-0.0,-0.0,-0.0,-0.0,-0.0,2.1471542311112688E-9,1.8067389175382345E-7,
        0.99963122917267189,0.99897637109651083,-1.9473352705673237E-7,-0.99963122917267189,-0.99897637109651083,
        0.0,0.0,0.0,0.0,0.0,0.0,0.0,0.0,-0.0,-0.0,-0.0,-0.0,-0.0,-0.0,-1.5346727990777808E-24,0.0,-0.0,
        -1.5544370926445683E-24,0.99963122917267155,0.0,0.0,0.0,0.0,0.0,0.0,0.0,0.0,0.0,-0.0,-0.0,-0.0,-0.0,-0.0,
        -0.0,-1.0,2.1332465124273696E-9,0.9989763710965166,-8.3705110748110957E-8,-8.5106993189669639E-8,
        -0.99949819932037964,0.0,0.0,0.0,0.0,0.0,0.0,0.0,-0.0,-0.0,-0.0,-0.0,-0.0,-0.0,-0.0,-0.0,
        1.1176480597257923E-5,5.0744975560979278E-8,0.99990781756997837,-5.7482272524168214E-10,0.0,0.0,0.0,0.0,0.0,
        0.0,0.0,0.0,-0.0,-0.0,-0.0,-0.0,-0.0,-1.0,-0.0,0.99963122917267433,1.6537533110604227E-24,0.0,0.0,
        9.13109398655825E-23,0.0,0.0,0.0,0.0,0.0,0.0,0.0,0.0,-0.0,-0.0,-0.0,-0.0,-0.0,-0.0,-1.0,-0.0,
        0.99990781757620883,0.0,8.2687665553020977E-25,0.0,0.0,0.0,0.0,0.0,0.0,0.0,-0.0,-0.0,-0.0,-0.0,-0.0,-0.0,
        -0.0,-1.0,-0.0,0.99963122917267522,0.0,0.0,-4.9605957844188972E-24,0.0,0.0,0.0,0.0,0.0,0.0,0.0,0.0,-0.0,
        -0.0,-0.0,-0.0,-0.0,-0.0,-0.0,-1.0,-9.9658601061337942E-10,-0.0,-2.1332465124273696E-9,0.9989763710965166,
        -0.99949819932037964,0.0,0.0,0.0,0.0,0.0,0.0,0.0,-0.0,-0.0,-0.0,-0.0,-0.0,-0.0,-0.0,-0.0,
        -2.9332448224953815E-9,0.99963122917267211,0.9989763710965115,-0.99963122917267211,1.736417092051019E-7,
        -0.9989763710965115,0.0,0.0,0.0,0.0,0.0,0.0,0.0,0.0,-0.0,-0.0,-0.0,-0.0,-0.0,-0.0,-0.0,-0.0,
        -1.1176480597134225E-5,-1.2259255630878441E-9,-2.1056109700059608E-9,-0.99990781756998193,
        1.2259255630878441E-9,2.1056109700059624E-9,0.0,0.0,0.0,0.0,0.0,0.0,0.0,1.0,-0.0,-0.0,-0.0,-0.0,-0.0,-0.0,
        -0.0,-0.0,0.99897637109651882,-3.6722326320306756E-9,-0.99949819932038086,2.4609503764964777E-9,0.0,0.0,0.0,
        0.0,0.0,0.0,-0.0,-0.0,-0.0,-0.0,-0.0,-0.0,-0.0,-0.0,-5.2901915156994062E-9,0.99963122917267289,
        0.99897637109651327,-0.99963122917267289,2.147154320450922E-9,-0.99897637109651327,0.0,0.0,0.0,0.0,0.0,0.0,
        0.0,-0.0,-0.0,-0.0,-0.0,-0.0,-0.0,-0.0,-0.0,-0.99990781757620562,-1.6537533110604194E-24,
        -2.6174432767160708E-31,0.0,0.0,0.0,0.0,0.0,0.0,0.0,0.0,-6.0877461546222069E-23,-0.99963122917267155,
        -8.2710550537587605E-25,0.0,0.0,0.0,0.0,0.0,0.0,0.0,0.0,1.0,0.0,-0.0,-0.0,-0.0,-0.0,-0.0,-0.0,-0.0,
        -3.8968556945376565E-15,-0.999907817569979,-1.0905409018537997E-24,-4.9605957844188833E-24,0.0,0.0,0.0,0.0,
        0.0,0.0,0.0,1.0,-0.0,-0.0,-0.0,-0.0,-0.0,-0.0,-0.0,-0.99963122917267155,8.2710533781282186E-25,
        3.653049195283498E-22,0.0,0.0,0.0,0.0,0.0,0.0,0.0,0.0,1.0,-0.0,-0.0,-0.0,-0.0,-0.0,-0.0,-0.0,-0.0,-0.0,
        -0.99963122917267289,7.4408936766283455E-24,0.0,0.0,0.0,0.0,0.0,0.0,0.0,0.0,0.0,1.0,-0.0,-0.0,-0.0,-0.0,
        -0.0,-0.0,-0.0,-0.0,7.0513718706461245E-9,0.99963122917267311,-2.14715423111127E-9,0.99897637109651394,
        -1.947335326058504E-7,-0.99963122917267311,-0.99897637109651394,0.0,0.0,0.0,0.0,0.0,0.0,0.0,-0.0,-0.0,-0.0,
        -0.0,-1.0,2.147154320450922E-9,8.8218854606609019E-12,0.99963122917267144,0.99897637109651016,
        -0.99963122917267144,-0.99897637109651016,0.0,0.0,0.0,0.0,0.0,0.0,0.0,0.0,0.0,-0.0,-0.0,-0.0,-0.0,-0.0,-0.0,
        -0.0,9.9658596963912385E-10,8.3705110748110917E-8,0.99897637109651072,-8.9311693624015258E-8,
        -0.9994981993203762,0.0,0.0,0.0,0.0,0.0,0.0,0.0,-0.0,-0.0,-0.0,-0.0,-0.0,-0.0,-1.0178752559210842E-24,
        0.99983610538248446,-6.1283679522649974E-15,0.0,-2.4518315687173011E-14,0.0,0.0,0.0,0.0,0.0,-0.0,-1.0,
        1.2259255630878439E-9,-1.1176480597053242E-5,-4.7948113514096212E-8,-4.8647446853876473E-8,
        -0.99990781756997882,0.0,0.0,0.0,0.0,0.0,0.0,1.0,0.0,-0.0,-0.0,-0.0,-0.0,-0.0,-0.0,-0.0,-0.0,
        -0.99917069199905872,5.07449741287703E-8,0.99990781757620506,-5.748227096964193E-10,-1.1176480635102603E-5,
        0.0,0.0,0.0,0.0,0.0,0.0,0.0,-0.0,-0.0,-0.0,-0.0,-0.0,-0.0,-0.0,1.8763240733251467E-9,1.1176480597253228E-5,
        0.99990781756997849,-5.7482270196104807E-10,-5.0744975560979436E-8,0.0,0.0,0.0,0.0,0.0,0.0,0.0,-0.0,-0.0,
        -0.0,-0.0,-0.0,-0.0,-1.0,-0.99990781756997826,2.3108031076841295E-19,7.782111081218338E-27,0.0,0.0,0.0,0.0,
        0.0,0.0,0.0,0.0,0.0,1.0,-0.0,-0.0,-0.0,-0.0,-0.0,-1.0,-0.0,0.99983610538248446,1.4982415428688111E-24,
        -6.1283679522649981E-15,-2.4518315687173039E-14,6.0877362830839736E-23,0.0,0.0,0.0,0.0,0.0,0.0,0.0,-0.0,
        -0.0,-0.0,-0.0,-0.0,-0.0,-1.0,-0.0,0.99963122917267211,2.4811359075780219E-24,-9.13108380663039E-23,
        -1.826524320052037E-22,0.0,0.0,0.0,0.0,0.0,0.0,0.0,0.0,-0.0,-0.0,-0.0,-0.0,-0.0,-1.0,-0.0,
        0.99917069199908215,-1.2259255300422014E-9,1.2259255300422014E-9,1.1176480610683842E-5,
        2.1056109130070607E-9,0.0,0.0,0.0,0.0,0.0,0.0,0.0,0.0,-0.0,-0.0,-0.0,-0.0,-0.0,-0.0,-0.0,-1.0,
        3.71683850222726E-25,-0.0,0.99990781756997882,8.5600255046274665E-25,0.0,0.0,0.0,0.0,0.0,0.0,0.0,-0.0,-0.0,
        -0.0,-0.0,-0.0,-0.0,-0.0,-1.0,-0.0,0.99963122917267289,7.4408936766283455E-24,0.0,0.0,0.0,0.0,0.0,0.0,0.0,
        0.0,0.0,0.0,-0.0,-0.0,-0.0,-0.0,-0.0,-0.0,-0.0,-1.0,0.99983610538248491,-1.242061175724179E-24,
        -2.48113590757802E-24,2.4518315687199128E-14,-7.4408936766283308E-24,0.0,0.0,0.0,0.0,0.0,0.0,0.0,-0.0,-0.0,
        -0.0,-0.0,-0.0,-0.0,-0.0,-1.0,0.99897637109651327,-8.931169603682376E-8,9.9658601061338025E-10,
        -0.99949819932037753,0.0,0.0,0.0,0.0,0.0,0.0,0.0,-0.0,-0.0,-0.0,-0.0,-0.0,-0.0,-0.0,-0.0,
        -2.147154320450922E-9,-1.5727474128375975E-11,0.99963122917267144,0.99897637109651016,-0.99963122917267144,
        -0.99897637109651016,0.0,0.0,0.0,0.0,0.0,0.0,0.0,-0.0,-0.0,-0.0,-0.0,-0.0,-0.0,-0.0,-0.0,-0.0,
        -9.9658596963912385E-10,0.99897637109651072,-0.9994981993203762,8.9311693624015827E-8,0.0,0.0,0.0,0.0,0.0,
        0.0,0.0,-0.0,-0.0,-0.0,-0.0,-0.0,-0.0,-0.0,-0.0,-5.7482272524168008E-10,-4.2161617423001467E-12,
        -5.0628697867350495E-10,-0.99990781756997782,0.0,0.0,0.0,0.0,0.0,0.0,1.0,-0.0,-0.0,-0.0,-0.0,-0.0,-0.0,-0.0,
        -0.0,-0.0,-1.2259255630878439E-9,-1.1176480597053242E-5,-0.99990781756997882,4.7948113514096212E-8,0.0,0.0,
        0.0,0.0,0.0,0.0,0.0,1.0,-0.0,-0.0,-0.0,-0.0,-0.0,-0.0,-0.0,-0.0,0.99990781756998193,-5.1011863363820206E-15,
        8.2687665553020968E-25,1.6526715295000437E-24,-8.2687665553020968E-25,0.0,0.0,0.0,0.0,0.0,0.0,0.0,0.0,-0.0,
        -0.0,-0.0,-0.0,-0.0,-0.0,-0.0,-0.0,-1.0,-0.99897637109651327,-2.4609503764964814E-9,0.9998361053824838,
        0.99949819932037753,9.965860106133786E-10,0.0,0.0,0.0,0.0,0.0,0.0,0.0,-0.0,-0.0,-0.0,-0.0,-0.0,-0.0,-0.0,
        1.2259255300422008E-9,-0.9991706919990615,0.9999078175762055,-4.7948112225350524E-8,-1.117648063511143E-5,
        0.0,0.0,0.0,0.0,0.0,0.0,-8.5600255046274665E-25,-0.0,-0.99990781756997793,-3.7168401778578055E-25,0.0,0.0,
        0.0,0.0,0.0,0.0,0.0,0.0,1.0,0.0,-0.0,-0.0,-0.0,-0.0,-0.0,-1.0,-0.99963122917267311,-2.4794888517521493E-24,
        0.0,0.0,0.0,0.0,0.0,0.0,0.0,0.0,0.0,1.0,-0.0,-0.0,-0.0,-0.0,-0.99949819932039363,0.99990781756998193,
        -1.2259255630878441E-9,-2.1056109700059608E-9,1.2259255630878441E-9,2.1056109700059624E-9,0.0,0.0,0.0,0.0,
        0.0,0.0,0.0,0.0,-0.0,-0.0,-0.0,-0.0,-0.0,-0.0,-0.0,-0.99990781756997882,2.3108031076841295E-19,
        8.5600255046274665E-25,0.0,9.13109398653475E-23,0.0,0.0,0.0,0.0,0.0,0.0,0.0,0.0,1.0,-0.0,-0.0,-0.0,-0.0,
        -0.0,-0.0,-1.0,-0.0,-0.99897637109651882,-3.6722326320306756E-9,0.99983610538248491,0.99949819932038086,
        2.4609503764964777E-9,0.0,0.0,0.0,0.0,0.0,0.0,0.0,-0.0,-0.0,-0.0,-0.0,-0.0,-0.0,-0.0,-0.99983610538248369,
        -3.8968556945292835E-15,6.1028847754872359E-24,-2.4518315687132678E-14,0.0,0.0,0.0,0.0,0.0,0.0,0.0,1.0,-0.0,
        -0.0,-0.0,-0.0,-0.0,-0.0,-0.0,-0.9991706919990615,-1.2259255300422005E-9,0.9999078175762055,
        -1.1176480635111456E-5,4.7948112225350524E-8,0.0,0.0,0.0,0.0,0.0,0.0,0.0,-0.0,-0.0,-0.0,-0.0,-0.0,-0.0,-0.0,
        -0.99963122917267211,2.4811359075780219E-24,-9.13108380663039E-23,0.0,-1.826524320052037E-22,0.0,0.0,0.0,
        0.0,0.0,0.0,-0.0,-0.0,-0.0,-0.0,-0.0,-0.99990781756997793,3.7168385022272627E-25,0.0,0.0,0.0,0.0,0.0,0.0,
        0.0,1.0,-0.0,-0.0,-0.0,-0.0,-0.0,-0.0,-0.0,-0.0,1.9473353260585005E-7,0.99963122917267289,
        -2.147154320450922E-9,0.99897637109651327,-0.99963122917267289,-0.99897637109651327,0.0,0.0,0.0,0.0,0.0,0.0,
        0.0,0.0,-0.0,-0.0,-0.0,-0.0,-0.0,-0.0,-0.0,-0.0,-9.6090976992104252E-25,0.99963122917267311,
        1.6542089162214075E-24,0.0,0.0,0.0,0.0,0.0,0.0,0.0,0.0,0.0,-0.0,-0.0,-0.0,-0.0,-0.0,-0.0,-1.0,
        -1.0724620018496892E-24,0.99990781756997849,1.2898465579145756E-14,1.6542089162214064E-24,0.0,0.0,0.0,0.0,
        0.0,0.0,0.0,-0.0,-0.0,-0.0,-0.0,-1.0,9.9658601061337922E-10,4.0460291731222033E-12,0.0033333300699559354,
        -0.99949819932037587,0.0,0.0,0.0,0.0,0.0,0.0,0.0,0.0,-0.0,-0.0,-0.0,-0.0,-0.0,-0.0,-0.0,
        -1.0374965720834998E-24,1.4234533912291339E-24,0.99983610538248313,-6.1283679522514479E-15,0.0,
        -2.4518315687102531E-14,0.0,0.0,0.0,0.0,0.0,0.0,-0.0,-0.0,-0.0,-0.0,-0.0,-0.0,-1.0,3.2686787101151743E-9,
        0.99897637109651383,-9.9658596963912323E-10,-8.93116960368229E-8,-0.99949819932037809,0.0,0.0,0.0,0.0,0.0,
        0.0,-0.0,-0.0,-0.0,-0.0,5.7482270196104745E-10,4.7948113514096212E-8,-1.1176480597035165E-5,
        -5.0744974286051676E-8,-0.999907817569978,0.0,0.0,0.0,0.0,0.0,0.0,1.0,0.0,-0.0,-0.0,-0.0,-0.0,-0.0,-0.0,
        -1.2203212349743148E-24,0.99990781756997882,1.1681206084644741E-18,0.0,0.0,0.0,0.0,0.0,0.0,0.0,0.0,0.0,-0.0,
        -0.0,-0.0,-0.0,-0.0,-0.0,-0.0,-0.0,-1.0,-0.99917069199905928,1.8763240227980709E-9,0.99990781757620528,
        -5.7482268641578688E-10,-1.1176480635104424E-5,-5.074497412877029E-8,0.0,0.0,0.0,0.0,0.0,0.0,-0.0,-0.0,-0.0,
        -0.0,-0.0,-0.0,5.7482270969642023E-10,-0.99917069199905617,5.07449728538431E-8,0.99990781757620484,
        -1.1176480635091554E-5,0.0,0.0,0.0,0.0,0.0,0.0,0.0,0.0,-0.0,-0.0,-0.0,-0.0,-0.0,-0.0,1.1176480597229996E-5,
        -1.2259255630878439E-9,0.99990781756997882,4.7948113514096192E-8,4.8647446853876592E-8,0.0,0.0,0.0,0.0,0.0,
        0.0,0.0,0.0,-0.0,-0.0,-0.0,-0.0,-0.0,-1.0,-0.0,-0.99990781756997849,-1.3398073766419519E-24,
        5.1011863363418432E-15,0.0,0.0,0.0,0.0,0.0,0.0,0.0,0.0,0.0,1.0,-0.0,-0.0,-0.0,-0.0,-0.0,-1.0,
        -1.3940092230708362E-22,0.99963122917267289,1.6542089162111081E-24,0.0,0.0,0.0,0.0,0.0,0.0,0.0,0.0,0.0,-0.0,
        -0.0,-0.0,-0.0,-0.0,-0.0,-1.0,-0.0,-0.99990781757620517,0.0,-0.99963122917267289,1.8259103138972109E-22,0.0,
        0.0,0.0,0.0,0.0,0.0,0.0,0.0,1.0,-0.0,-0.0,-0.0,-0.0,-0.0,-0.0,-0.0,-0.0,0.99983610538248313,0.0,
        -9.3797093753698854E-25,0.99990781756997793,0.0,0.0,0.0,0.0,0.0,0.0,0.0,0.0,-0.0,-0.0,-0.0,-0.0,-0.0,-0.0,
        -0.0,-1.0,0.99963122917267155,8.2710533781282186E-25,3.653049195283498E-22,0.0,0.0,0.0,0.0,0.0,0.0,0.0,0.0,
        0.0,-0.0,-0.0,-0.0,-0.0,-0.0,-0.0,-0.0,-1.0,-0.0,0.99990781756997826,1.1681206084644739E-18,
        -2.4325725010341474E-26,0.0,0.0,0.0,0.0,0.0,0.0,0.0,0.0,-0.0,-0.0,-0.0,-0.0,-0.0,-0.0,-0.0,-0.0,-1.0,
        0.99983610538248335,1.7747356371655138E-24,-1.1106359513858438E-22,2.4518315687110833E-14,
        -3.6530486400967496E-22,0.0,0.0,0.0,0.0,0.0,0.0,0.0,-0.0,-0.0,-0.0,-0.0,-0.0,-0.0,-1.0,-0.0,
        -3.2686787101151743E-9,0.99897637109651383,9.9658596963912323E-10,0.0,0.0,0.0,0.0,0.0,0.0,0.0,-0.0,-0.0,
        -0.0,-0.0,-0.0,-0.0,-0.0,-0.0,-1.0,-0.0033333300699559354,-9.9658601061337922E-10,0.99983610538248313,
        0.99949819932037587,0.0,0.0,0.0,0.0,0.0,0.0,0.0,-0.0,-0.0,-0.0,-0.0,-0.0,-0.0,-0.0,-0.0,
        -1.1176480597257946E-5,-5.0744975560979747E-8,-0.99990781756997837,5.7482272524168214E-10,0.0,0.0,0.0,0.0,
        0.0,0.0,1.0,0.0,-0.0,-0.0,-0.0,-0.0,-0.0,-0.0,-0.0,-0.0,-0.99949819932037753,-1.4173965603573214E-9,
        0.99990781756997837,5.74822725241682E-10,0.0,0.0,0.0,0.0,0.0,0.0,0.0,-0.0,-0.0,-0.0,-0.0,-0.0,-0.0,-0.0,
        1.2259255630878439E-9,1.117648059705322E-5,0.99990781756997882,-4.7948113514096212E-8,0.0,0.0,0.0,0.0,0.0,
        0.0,0.0,0.0,-0.0,-0.0,-0.0,-0.0,-0.0,-0.0,-0.0,-1.0,-0.99990781757620484,-8.2710550537587568E-25,
        -4.1595572192614484E-35,8.2718002562972932E-27,0.0,0.0,0.0,0.0,0.0,0.0,0.0,0.0,1.0,0.0,-0.0,-0.0,-0.0,-0.0,
        -0.0,-0.0,-0.99949819932038086,-2.1056109700059616E-9,0.999907817569979,1.4173965603573227E-9,0.0,0.0,0.0,
        0.0,0.0,0.0,0.0,-0.0,-0.0,-0.0,-0.0,-0.0,-0.0,-0.0,-0.99990781756997815,2.3108031076841295E-19,
        1.8300038227672562E-24,-8.2718061255302767E-25,0.0,0.0,0.0,0.0,0.0,0.0,0.0,0.0,1.0,-0.0,-0.0,-0.0,-0.0,-0.0,
        -0.0,-1.0,-0.0,-0.99990781756997826,-1.1681206084644741E-18,3.1030314338004435E-26,0.0,0.0,0.0,0.0,0.0,0.0,
        0.0,0.0,1.0,-0.0,-0.0,-0.0,-0.0,-0.0,-0.0,-0.0,-0.999907817576205,-1.6589186258530995E-31,
        2.4811359075780197E-24,0.0,-1.8265243200475341E-22,0.0,0.0,0.0,0.0,0.0,0.0,0.0,1.0,-0.0,-0.0,-0.0,-0.0,-0.0,
        -0.0,-0.0,1.8763240733251471E-9,-1.1176480597046237E-5,-5.7482270196104807E-10,-5.0744975560979072E-8,
        -0.99990781756997837,0.0,0.0,0.0,0.0,0.0,0.0,1.0,-0.0,-0.0,-0.0,-0.0,-9.6090976992103922E-25,
        0.9998361053824838,-6.12836795225911E-15,1.6542089162214068E-24,0.0,-2.4518315687140125E-14,0.0,0.0,0.0,0.0,
        0.0,-0.0,-0.0,-0.0,-0.0,-0.0,-0.0,-1.0,-9.3797097128994911E-25,-2.8271430567041626E-27,0.99990781756997793,
        1.1681206084644741E-18,0.0,0.0,0.0,0.0,0.0,0.0,0.0,0.0,-0.0,-0.0,-0.0,-0.0,-0.0,-0.0,-1.0,
        3.373234635669438E-27,0.99990781756997826,1.1681206084644741E-18,1.6542089162111069E-24,0.0,0.0,0.0,0.0,0.0,
        0.0,0.0,-0.0,-0.0,-0.0,-0.0,-0.0,-0.0,-0.0,-1.0,-0.0,8.93116960368232E-8,0.99897637109651327,
        -9.9658601061338025E-10,-0.99949819932037753,0.0,0.0,0.0,0.0,0.0,0.0,0.0,-0.0,-0.0,-0.0,-0.0,-0.0,-0.0,-0.0,
        -0.0,5.748227252416807E-10,2.298866341239155E-12,-5.0628697867095692E-10,-0.99990781756997793,0.0,0.0,0.0,
        0.0,0.0,0.0,0.0,1.0,0.0,-0.0,-0.0,-0.0,-0.0,-0.0,-0.0,-0.0,5.7482272524168008E-10,5.0628697867350495E-10,
        2.2988663412391542E-12,0.99990781756997782,0.0,0.0,0.0,0.0,0.0,0.0,0.0,0.0,0.0,-0.0,-0.0,-0.0,-0.0,-0.0,
        -1.0,1.1176480597260384E-5,-7.8555494783415347E-10,0.99990781756997815,4.654921224045972E-8,0.0,0.0,0.0,0.0,
        0.0,0.0,0.0,0.0,-0.0,-0.0,-0.0,-0.0,-0.0,-0.0,-1.0,-0.0,6.3503510448242124E-23,0.99983610538248369,
        1.6542089162111072E-24,0.0,0.0,0.0,0.0,0.0,0.0,0.0,0.0,0.0,-0.0,-0.0,-0.0,-0.0,-0.0,-0.0,-1.0,-0.0,
        -0.0049999982279884773,-5.7482272524168142E-10,-4.2161617423001322E-12,0.99990781756997782,0.0,0.0,0.0,0.0,
        0.0,0.0,0.0,-0.0,-0.0,-0.0,-0.0,-0.0,-0.0,-0.0,-0.0,5.7482270196104776E-10,4.7948113514096205E-8,
        1.1176480597084896E-5,0.999907817569978,-5.0744974286051676E-8,0.0,0.0,0.0,0.0,0.0,0.0,0.0,0.0,-0.0,-0.0,
        -0.0,-0.0,-0.0,-1.0,-0.99917069199905717,-7.85554926779473E-10,0.99990781757620484,-1.1176480635095745E-5,
        4.6549211023469635E-8,0.0,0.0,0.0,0.0,0.0,0.0,0.0,-0.0,-0.0,-0.0,-0.0,-0.0,-0.0,-0.0,5.0744975560979284E-8,
        -1.1176480597044428E-5,-5.7482272524168049E-10,-0.99990781756997837,0.0,0.0,0.0,0.0,0.0,0.0,0.0,1.0,-0.0,
        -0.0,-0.0,-0.0,-0.0,-0.0,-0.0,-0.0,-4.6005888522010356E-9,0.999631120487158,-7.3971927480498425E-9,
        0.99897611086126492,4.6005888522010356E-9,-0.999631120487158,7.3971927480498425E-9,-0.99897611086126492,0.0,
        0.0,0.0,0.0,0.0,0.0,0.0,0.0,-0.0,-0.0,-0.0,-0.0,-0.0,-0.0,-0.0,-0.0,4.6005888522010356E-9,
        0.99963112048714808,-1.5821451349744818E-7,-1.54695266131476E-7,0.99897611086123783,-0.99963112048714808,
        -0.99897611086123783,0.0,0.0,0.0,0.0,0.0,0.0,0.0,0.0,-0.0,-0.0,-0.0,-0.0,-0.0,-0.0,-0.0,-0.0,
        -0.99963112048715808,-8.2687674506154525E-25,-8.1708213259091664E-15,8.2633597939288586E-25,
        -1.2255546890460897E-14,8.2687674506154525E-25,-8.2633597939288586E-25,0.0,0.0,0.0,0.0,0.0,0.0,0.0,1.0,-0.0,
        -0.0,-0.0,-0.0,-0.0,-0.0,-0.0,-0.0,7.3971927480498417E-9,-3.2005225839515484E-9,0.99963112048715,
        -5.4431996987624587E-9,-0.998976110861243,0.0,0.0,0.0,0.0,0.0,0.0,0.0,-0.0,-0.0,-0.0,-0.0,-0.0,-0.0,-0.0,
        -1.0,-4.6005888522010356E-9,0.99963112048714808,0.99897611086123783,-0.99963112048714808,
        1.5821451349744818E-7,1.5469526613147609E-7,-0.99897611086123783,0.0,0.0,0.0,0.0,0.0,0.0,0.0,0.0,-0.0,-0.0,
        -0.0,-0.0,-0.0,-0.0,-0.0,-0.0,0.99963112048715808,-8.2687674506154525E-25,8.2633597939288586E-25,
        8.2687674506154525E-25,8.1708213259091664E-15,-8.2633597939288586E-25,1.2255546890460905E-14,0.0,0.0,0.0,
        0.0,0.0,0.0,0.0,0.0,-0.0,-0.0,-0.0,-0.0,-0.0,-0.0,-0.0,-1.0,-7.3971927480498417E-9,0.99963112048715,
        0.998976110861243,-0.99963112048715,5.4431996987624587E-9,-0.998976110861243,0.0,0.0,0.0,0.0,0.0,0.0,0.0,
        -0.0,-0.0,-0.0,-0.0,-0.0,-0.0,-0.0,-0.0,0.99897611086126514,-1.9550980048176465E-9,2.8616875269971646E-9,
        -0.99949804568895317,3.1381363662704186E-9,0.0,0.0,0.0,0.0,0.0,0.0,0.0,-0.0,-0.0,-0.0,-0.0,-0.0,-0.0,-0.0,
        -0.0,6.5654885534357305E-25,-0.99963112048714819,0.0,-8.1708213258030141E-15,4.565989935595539E-23,0.0,0.0,
        0.0,0.0,0.0,0.0,0.0,1.0,-0.0,-0.0,-0.0,-0.0,-0.0,-0.0,-0.0,-0.0,1.5469526613147607E-7,2.4525266900696403E-9,
        0.99963112048714609,0.99897611086123228,-0.99963112048714609,-0.99897611086123228,0.0,0.0,0.0,0.0,0.0,0.0,
        0.0,0.0,0.0,-0.0,-0.0,-0.0,-0.0,-0.0,-0.0,-0.0,6.5654885534357305E-25,-0.0,8.67546784372977E-25,
        0.99963112048714631,1.8260330585353678E-22,8.1708213257832058E-15,0.0,0.0,0.0,0.0,0.0,0.0,0.0,0.0,-0.0,-0.0,
        -0.0,-0.0,-0.0,-0.0,-1.0,1.9550980048176465E-9,0.99897611086123783,-6.6850293817222149E-8,
        -6.54405645365157E-8,-0.99949804568893963,0.0,0.0,0.0,0.0,0.0,0.0,0.0,-0.0,-0.0,-0.0,-0.0,-0.0,-0.0,-0.0,
        -0.0,-0.99990778299963512,0.0,-8.2687674506154332E-25,8.2633597939288108E-25,-4.9013936600840107E-14,
        8.2687674506154332E-25,-8.2633597939288108E-25,0.0,0.0,0.0,0.0,0.0,0.0,0.0,1.0,-0.0,-0.0,-0.0,-0.0,-0.0,
        -0.0,-0.99963112048714819,-6.0883884625797955E-23,-0.0,-0.99990778299340188,-9.2478336911751012E-25,0.0,0.0,
        0.0,0.0,0.0,0.0,0.0,0.0,1.0,-0.0,-0.0,-0.0,-0.0,-0.0,-0.0,-0.0,-0.99963112048715,-8.2633597939288577E-25,
        -8.17082132582398E-15,-1.2255546890334395E-14,-2.4802982728761848E-24,0.0,0.0,0.0,0.0,0.0,0.0,1.0,-0.0,-0.0,
        -0.0,-0.0,-0.0,-0.0,-0.0,-0.0,3.3893748116090727E-8,1.1179883994384877E-5,-5.7482274508681107E-10,
        0.99990778299340177,0.0,0.0,0.0,0.0,0.0,0.0,0.0,0.0,-0.0,-0.0,-0.0,-0.0,-0.0,-0.0,-1.0,
        -6.5654885534357305E-25,0.99963112048714819,8.1708213258030141E-15,-9.1319798711910828E-23,
        1.2255546890303109E-14,0.0,0.0,0.0,0.0,0.0,0.0,0.0,0.0,-0.0,-0.0,-0.0,-0.0,-0.0,-0.0,-0.0,-1.0,
        -2.4525266239754055E-9,-1.5821451349744813E-7,0.9996311204871462,1.4414030326781142E-7,0.0,0.0,0.0,0.0,0.0,
        0.0,-0.0,-0.0,-0.0,-0.0,-0.0,-0.0,-0.0,-0.0,-1.0,-1.9550980048176465E-9,0.99897611086123783,
        6.6850293817222149E-8,-0.99949804568893963,6.5440564536515741E-8,0.0,0.0,0.0,0.0,0.0,0.0,0.0,-0.0,-0.0,-0.0,
        -0.0,-0.0,-0.0,-0.0,-0.0,0.99990778299340222,-0.0,0.99963112048715,-8.2633597939288577E-25,
        -2.4802982728761848E-24,0.0,0.0,0.0,0.0,0.0,0.0,0.0,-0.0,-0.0,-0.0,-0.0,-0.0,-0.0,-0.0,-1.0,
        0.999836048837159,-1.653753490123087E-24,0.0,1.653753490123087E-24,0.0,0.0,0.0,0.0,0.0,0.0,0.0,0.0,0.0,0.0,
        -0.0,-0.0,-0.0,-0.0,-0.0,-0.0,-0.0,-1.0,-1.4414029772121643E-7,0.99963112048714764,0.99897611086123661,
        2.45252669006964E-9,-0.99963112048714764,-0.99897611086123661,0.0,0.0,0.0,0.0,0.0,0.0,0.0,0.0,-0.0,-0.0,
        -0.0,-0.0,-0.0,-0.0,-0.0,-0.0,-3.1381363662704182E-9,0.998976110861243,2.3083266524056644E-9,
        -0.99949804568894218,0.0,0.0,0.0,0.0,0.0,0.0,-0.0,-0.0,-0.0,-0.0,-0.0,-0.0,-0.0,-0.0,0.99949804568895306,
        -1.0732815899129811E-9,-1.7242506299916647E-9,1.0732815899129811E-9,-0.99990778299340444,
        1.7242506299916647E-9,0.0,0.0,0.0,0.0,0.0,0.0,0.0,-0.0,-0.0,-0.0,-0.0,-0.0,-0.0,-0.0,-0.0,
        1.1736711083188498E-24,-0.99963112048714631,-3.0441942312898983E-23,-8.1708213257832058E-15,
        1.8260330585353678E-22,0.0,0.0,0.0,0.0,0.0,0.0,-3.5063349747690686E-32,6.5654885534357122E-25,
        -0.99990778299340188,-6.0883884625634808E-23,0.0,0.0,0.0,0.0,0.0,0.0,0.0,0.0,1.0,-0.0,-0.0,-0.0,-0.0,-0.0,
        -0.0,-0.0,6.5440564536515675E-8,1.0474815505067268E-9,0.99897611086123228,-0.99949804568893685,0.0,0.0,0.0,
        0.0,0.0,0.0,0.0,0.0,-0.0,-0.0,-0.0,-0.0,-0.0,-0.0,-0.0,6.5654885534357122E-25,0.99990778299340188,
        1.2257594733752547E-14,-6.0883884625634808E-23,4.56598993558439E-23,0.0,0.0,0.0,0.0,0.0,0.0,0.0,-0.0,-0.0,
        -0.0,-0.0,-0.0,-0.0,-0.0,-0.0,-1.0,1.0732815899129813E-9,0.99949804568893963,-3.6713869361265483E-8,
        -3.6008700290680974E-8,-0.99990778299340188,0.0,0.0,0.0,0.0,0.0,0.0,0.0,-0.0,-0.0,-0.0,-0.0,-0.0,-0.0,-0.0,
        -0.0,-0.99917046997485948,-1.0732815452487715E-9,0.99990778299963523,-1.7242505575001712E-9,
        -1.1179883991598272E-5,1.0732815452487715E-9,1.7242505575001712E-9,0.0,0.0,0.0,0.0,0.0,0.0,0.0,-0.0,-0.0,
        -0.0,-0.0,-0.0,-0.99990778299340455,1.1102231372380358E-18,-8.2687674506154295E-25,8.2633597939288053E-25,
        8.2687674506154295E-25,-8.2633597939288053E-25,0.0,0.0,0.0,0.0,0.0,0.0,0.0,0.0,1.0,-0.0,-0.0,-0.0,-0.0,-0.0,
        -0.0,-0.0,-0.99990778299963312,8.0210898815735369E-32,-8.26335979392881E-25,-4.9013936600353614E-14,
        -2.480298272876176E-24,0.0,0.0,0.0,0.0,0.0,0.0,1.0,-0.0,-0.0,-0.0,-0.0,-0.0,-0.0,-0.99963112048714664,
        -8.2704575403369328E-25,-5.089086563781989E-29,-8.17082132578696E-15,-1.8267568712810435E-22,0.0,0.0,0.0,
        0.0,0.0,-0.0,-0.0,-0.99963112048714764,7.7525629785265257E-23,-8.1708213257987353E-15,
        -1.2255546890296826E-14,0.0,0.0,0.0,0.0,0.0,0.0,0.0,0.0,1.0,-0.0,-0.0,-0.0,-0.0,-0.0,-0.0,-0.0,-0.0,
        1.5711765311757415E-9,1.1179884015962847E-5,-5.7482272954512609E-10,0.99990778299340177,
        -3.3893748116090668E-8,0.0,0.0,0.0,0.0,0.0,0.0,0.0,-0.0,-0.0,-0.0,-0.0,-0.0,-0.0,-1.0,-0.99917046997483627,
        3.3893746683251984E-8,-5.74822721802599E-10,0.99990778299963246,-1.1179883991454058E-5,0.0,0.0,0.0,0.0,0.0,
        0.0,0.0,-0.0,-0.0,-0.0,-0.0,-0.0,-0.0,-0.0,5.7482274508681158E-10,1.5353640561060077E-12,
        5.0647488691030916E-10,0.99990778299340122,0.0,0.0,0.0,0.0,0.0,0.0,0.0,0.0,0.0,-0.0,-0.0,-0.0,-0.0,-0.0,
        -0.0,-1.0,-1.1735869340295751E-24,0.99963112048714664,6.8489849033933118E-23,0.0,8.1708213257869577E-15,0.0,
        0.0,0.0,0.0,0.0,0.0,0.0,-0.0,-0.0,-0.0,-0.0,-0.0,-0.0,-0.0,-1.0,-1.1733464545733572E-24,0.99983604883715449,
        -6.1277734451515543E-15,0.0,-4.5659899355866823E-23,0.0,0.0,0.0,0.0,0.0,0.0,0.0,-0.0,-0.0,-0.0,-0.0,-0.0,
        -0.0,-1.0,-6.7462254585841681E-9,0.99963112048714775,-0.99963112048714775,1.4414029772121662E-7,
        -0.998976110861237,0.0,0.0,0.0,0.0,0.0,0.0,0.0,0.0,-0.0,-0.0,-0.0,-0.0,-0.0,-0.0,-0.0,-0.0,
        0.99990778299340133,-0.0,-4.6236181525834039E-25,0.99963112048714609,0.0,0.0,0.0,0.0,0.0,0.0,0.0,-0.0,-0.0,
        -0.0,-0.0,-0.0,-0.0,-0.0,-0.0,-1.0,-1.0732815899129813E-9,0.99949804568893963,-0.99990778299340188,
        3.6713869361265483E-8,3.6008700290680947E-8,0.0,0.0,0.0,0.0,0.0,0.0,0.0,-0.0,-0.0,-0.0,-0.0,-0.0,-0.0,-0.0,
        -0.0,-1.3628313725542006E-9,0.99897611086123372,-0.99983604883715371,6.9670305139362366E-8,
        -0.99949804568893752,0.0,0.0,0.0,0.0,0.0,0.0,0.0,-0.0,-0.0,-0.0,-0.0,-0.0,-0.0,-0.0,-0.0,
        -1.7242506299916662E-9,-1.1179883994595749E-5,-0.99990778299340233,1.2647726762421167E-9,0.0,0.0,0.0,0.0,
        0.0,0.0,1.0,-0.0,-0.0,-0.0,-0.0,-0.0,-0.0,-0.0,-0.0,0.99990778299340455,1.110222912088726E-18,
        -8.2687674506154295E-25,8.2633597939288053E-25,8.2687674506154295E-25,-8.2633597939288053E-25,0.0,0.0,0.0,
        0.0,0.0,0.0,0.0,-0.0,-0.0,-0.0,-0.0,-0.0,-0.0,-0.0,-0.0,-1.0,0.99990778299963312,-8.26335979392881E-25,
        -2.480298272876176E-24,4.9013936600353727E-14,0.0,0.0,0.0,0.0,0.0,0.0,0.0,-0.0,-0.0,-0.0,-0.0,-0.0,-0.0,
        -0.0,-1.0,0.99990778299340177,2.319246843608249E-18,3.5775740920850787E-27,0.0,0.0,0.0,0.0,0.0,0.0,0.0,0.0,
        -0.0,-0.0,-0.0,-0.0,-0.0,-0.0,-0.0,-0.0,-1.0,0.99963112048714764,7.7525629785265257E-23,0.0,
        8.1708213257987353E-15,0.0,0.0,0.0,0.0,0.0,0.0,0.0,0.0,-0.0,-0.0,-0.0,-0.0,-0.0,-0.0,-0.0,-1.0,
        -2.4525266900696403E-9,-1.4414030326781142E-7,0.99963112048714609,0.99897611086123228,-0.99963112048714609,
        -0.99897611086123228,0.0,0.0,0.0,0.0,0.0,0.0,0.0,-0.0,-0.0,-0.0,-0.0,-0.0,-0.0,-0.0,-0.0,-0.0,
        1.7242506299916666E-9,0.99949804568894218,-7.4738609228964772E-10,-1.2647726762421143E-9,
        -0.99990778299340233,0.0,0.0,0.0,0.0,0.0,0.0,0.0,-0.0,-0.0,-0.0,-0.0,-0.0,-0.0,-0.0,-0.99963112048714786,
        1.6529929340294675E-24,0.0,-8.170821325800201E-15,5.478100006651387E-22,0.0,0.0,0.0,0.0,0.0,0.0,
        -0.99963112048714609,-0.0,4.3355204953827373E-25,-0.99990778299340133,0.0,0.0,0.0,0.0,0.0,0.0,0.0,0.0,0.0,
        1.0,-0.0,-0.0,-0.0,-0.0,-0.0,-0.0,1.0732815452487704E-9,-0.99917046997483738,0.99990778299963268,
        -3.671386778656412E-8,-1.1179884040473105E-5,0.0,0.0,0.0,0.0,0.0,0.0,0.0,-0.0,-0.0,-0.0,-0.0,
        5.4431996987624562E-9,-2.45252669006964E-9,0.99963112048714764,0.99897611086123661,-0.99963112048714764,
        -0.99897611086123661,0.0,0.0,0.0,0.0,0.0,0.0,0.0,0.0,-0.0,-0.0,-0.0,-0.0,-0.0,-0.0,-0.0,
        7.97243578611214E-25,-6.81071288059573E-27,0.99963112048714609,8.1708213257817385E-15,
        1.2255546890271567E-14,0.0,0.0,0.0,0.0,0.0,0.0,0.0,0.0,0.0,-0.0,-0.0,-0.0,-0.0,-0.0,-0.0,-0.0,-1.0,
        3.1381363662704182E-9,0.998976110861243,-1.3628313725542002E-9,-2.3083266524056644E-9,-0.99949804568894218,
        0.0,0.0,0.0,0.0,0.0,0.0,0.0,-0.0,-0.0,-0.0,-0.0,-0.0,-0.0,-0.0,7.4738609228964782E-10,3.6008700290680987E-8,
        0.99949804568893752,-3.812448381630912E-8,-0.99990778299340144,0.0,0.0,0.0,0.0,0.0,0.0,0.0,-0.0,-0.0,-0.0,
        -0.0,-0.0,-0.0,-0.0,3.3450102398249045E-26,0.99963112048714786,-1.654208973331164E-24,
        1.8260333355504667E-22,8.170821325800201E-15,0.0,0.0,0.0,0.0,0.0,0.0,0.0,-0.0,-0.0,-0.0,-0.0,-0.0,-0.0,-1.0,
        1.1733464545733572E-24,0.99983604883715449,-6.1277734451515543E-15,0.0,0.0,0.0,0.0,0.0,0.0,0.0,0.0,-0.0,
        -0.0,-0.0,-0.0,-1.0,8.0913566202880005E-25,0.99990778299340133,0.0,0.0,0.0,0.0,0.0,0.0,0.0,0.0,-0.0,-0.0,
        -0.0,-0.0,-0.0,-0.0,-0.0,-1.0,1.1179884016105246E-5,-1.0732815899129811E-9,0.99990778299340444,
        -1.7242506299916647E-9,1.0732815899129811E-9,1.7242506299916647E-9,0.0,0.0,0.0,0.0,0.0,0.0,0.0,0.0,-0.0,
        -0.0,-0.0,-0.0,-0.0,-0.0,-0.0,-1.0,-0.99917046997483738,-1.0732815452487708E-9,0.99990778299963268,
        -1.1179884040473105E-5,3.6008698751452126E-8,0.0,0.0,0.0,0.0,0.0,0.0,0.0,-0.0,-0.0,-0.0,-0.0,-0.0,-0.0,-0.0,
        -0.99917046997483283,-5.7482272180259841E-10,-3.8124482170648835E-8,0.99990778299963212,
        -1.1179883991431714E-5,0.0,0.0,0.0,0.0,0.0,0.0,-0.0,-0.0,-0.0,-0.0,-0.0,-0.99990778299340222,
        1.5536028954057082E-18,-1.6329679215747038E-27,2.480298272876176E-24,0.0,0.0,0.0,0.0,0.0,0.0,0.0,1.0,-0.0,
        -0.0,-0.0,-0.0,-0.0,-0.0,-0.0,-0.99990778299963223,1.4945020319951258E-31,-8.2704575403369217E-25,
        -5.0890865637707383E-29,-4.9013936600139971E-14,-1.8267568712757923E-22,0.0,0.0,0.0,0.0,0.0,1.0,-0.0,-0.0,
        -0.0,-0.0,-0.0,-0.0,-0.0,-0.99917046997484149,-1.7242505575001691E-9,0.99990778299963312,
        -1.1179884040501237E-5,1.2647726231750714E-9,0.0,0.0,0.0,0.0,0.0,0.0,-0.0,-0.0,-0.0,-0.0,
        -0.99990778299963246,-5.6348491829692715E-15,8.3371555091865783E-23,-2.4506968300103951E-14,0.0,0.0,0.0,0.0,
        0.0,0.0,0.0,0.0,1.0,-0.0,-0.0,-0.0,-0.0,-0.0,-0.0,-0.99963112048714609,-1.4276505770110116E-24,
        -9.7856279789920354E-28,-8.1708213257817385E-15,-1.2255546890271561E-14,0.0,0.0,0.0,0.0,0.0,0.0,1.0,-0.0,
        -0.0,-0.0,-0.0,-0.0,-0.0,-0.0,-0.0,-0.0,1.5711764651554684E-9,-0.99917046997483661,-5.74822706260914E-10,
        0.99990778299963246,-3.3893746683251839E-8,-1.1179884040469817E-5,0.0,0.0,0.0,0.0,0.0,0.0,-0.0,-0.0,-0.0,
        -0.0,-0.0,-0.0,-0.99990778299340177,1.7977133271998997E-24,2.4506968300107927E-14,0.0,
        5.4781000066416455E-22,0.0,0.0,0.0,0.0,0.0,0.0,0.0,1.0,-0.0,-0.0,-0.0,-0.0,-0.0,-0.0,
        -1.6495737869470529E-22,0.99963112048714764,0.0,8.1708213257987322E-15,1.2255546890296834E-14,0.0,0.0,0.0,
        0.0,0.0,0.0,0.0,0.0,-0.0,-0.0,-0.0,-0.0,-0.0,-0.0,-1.0,5.7482272180259882E-10,-0.99917046997483283,
        3.3893747966548331E-8,0.99990778299963212,-1.1179883991431702E-5,0.0,0.0,0.0,0.0,0.0,0.0,0.0,0.0,-0.0,-0.0,
        -0.0,-0.0,-0.0,-0.0,1.1179884016175223E-5,-1.0732815899129815E-9,0.99990778299340188,3.6008700290680947E-8,
        0.0,0.0,0.0,0.0,0.0,0.0,0.0,0.0,-0.0,-0.0,-0.0,-0.0,-0.0,-0.0,-0.0,-1.0,5.7482272954512681E-10,
        -3.3893749399387173E-8,1.0732815899129813E-9,1.1179884015966133E-5,0.99990778299340188,0.0,0.0,0.0,0.0,0.0,
        0.0,0.0,0.0,-0.0,-0.0,-0.0,-0.0,-0.0,-0.0,-0.0,-1.0,-1.4401415297832177E-24,0.0,-0.99990778299340133,
        -1.3993198655389351E-24,0.0,0.0,0.0,0.0,0.0,0.0,0.0,1.0,-0.0,-0.0,-0.0,-0.0,-0.0,-0.0,-0.0,-0.0,
        -6.5654885534357122E-25,0.99990778299340188,1.2257594733752547E-14,6.0883884625634808E-23,
        -4.5659899355843924E-23,0.0,0.0,0.0,0.0,0.0,0.0,0.0,-0.0,-0.0,-0.0,-0.0,-0.0,-0.0,-0.0,-0.0,-1.0,
        -5.7482274508681158E-10,-3.452658377048904E-12,-5.0647488691030916E-10,-0.99990778299340122,0.0,0.0,0.0,0.0,
        0.0,0.0,1.0,-0.0,-0.0,-0.0,-0.0,-0.0,-0.0,-0.0,-0.0,-0.0,-4.6232865522438129E-25,0.99983604883715382,
        -4.3490670241533566E-15,3.6535137425528218E-22,0.0,0.0,0.0,0.0,0.0,0.0,0.0,0.0,-0.0,-0.0,-0.0,-0.0,-0.0,
        -0.0,-0.0,-1.0,0.99917046997484149,-1.7242505575001691E-9,-0.99990778299963312,0.0,0.0,0.0,0.0,0.0,0.0,0.0,
        -0.0,-0.0,-0.0,-0.0,-0.0,-0.0,-0.0,-0.0,-0.0,-7.2645124913565716E-29,0.99990778299340222,
        -1.2405680237842904E-24,-2.480298272876176E-24,0.0,0.0,0.0,0.0,0.0,0.0,0.0,-0.0,-0.0,-0.0,-0.0,-0.0,-0.0,
        -0.0,-1.0,-3.3893748116090793E-8,-1.11798839943849E-5,5.7482274508681107E-10,-0.99990778299340177,0.0,0.0,
        0.0,0.0,0.0,0.0,0.0,1.0,-0.0,-0.0,-0.0,-0.0,-0.0,-0.0,-0.0,-0.0,1.2647726762421169E-9,0.99949804568893885,
        -5.7482274508681107E-10,-0.99990778299340177,0.0,0.0,0.0,0.0,0.0,0.0,0.0,-0.0,-0.0,-0.0,-0.0,-0.0,-0.0,-0.0,
        -0.99963112048714764,-7.7525629785265093E-23,0.0,-8.1708213257987353E-15,0.0,0.0,0.0,0.0,0.0,0.0,0.0,1.0,
        -0.0,-0.0,-0.0,-0.0,-0.0,-0.0,-0.0,-0.0,1.1736711083188487E-24,-0.99990778299340133,-3.6669282854287522E-27,
        1.1102231372380358E-18,8.2718061255302767E-25,0.0,0.0,0.0,0.0,0.0,0.0,0.0,0.0,1.0,-0.0,-0.0,-0.0,-0.0,-0.0,
        -0.0,2.3083266524056639E-9,0.99897611086123661,-1.0474815505067272E-9,-0.99949804568893907,0.0,0.0,0.0,0.0,
        0.0,0.0,0.0,-0.0,-0.0,-0.0,-0.0,-0.0,-0.0,-0.0,7.9724357861121341E-25,-6.81071288059573E-27,
        0.99983604883715349,0.0,0.0,0.0,0.0,0.0,0.0,0.0,0.0,0.0,0.0,-0.0,-0.0,-0.0,-0.0,-0.0,-0.0,-0.0,-1.0,
        5.7482274508681158E-10,3.4526583770489028E-12,0.0049999982273354181,-0.99990778299340122,0.0,0.0,0.0,0.0,
        0.0,0.0,0.0,0.0,-0.0,-0.0,-0.0,-0.0,-0.0,-0.0,-0.0,1.4568589678256487E-24,-2.08457155049481E-23,
        0.9998360488371536,1.8260330585328007E-22,0.0,0.0,0.0,0.0,0.0,0.0,0.0,0.0,0.0,-0.0,-0.0,-0.0,-0.0,-0.0,-0.0,
        -1.0,-0.99917046997483627,-3.3893746683252037E-8,0.99990778299963246,-1.1179883991454058E-5,
        5.7482272180259737E-10,0.0,0.0,0.0,0.0,0.0,0.0,0.0,-0.0,-0.0,-0.0,-0.0,-0.99917046997483394,
        -7.4738606155649931E-10,-3.6008698751452106E-8,0.99990778299963223,-1.1179884040452532E-5,
        3.81244821706486E-8,0.0,0.0,0.0,0.0,0.0,-0.0,-0.0,-0.0,-0.0,-0.0,-0.0,-0.0,-0.999907782999632,
        -7.6564426326769119E-19,-1.3278959384951088E-24,-3.6140763870788811E-28,-1.1102230246251565E-16,0.0,0.0,0.0,
        0.0,0.0,0.0,1.0,-0.0,-0.0,-0.0,-0.0,-0.0,-0.0,-0.0,5.0647488692188814E-10,-5.7482274508681158E-10,
        -3.4526583770489133E-12,0.99990778299340122,0.0,0.0,0.0,0.0,0.0,0.0,0.0,-0.0,-0.0,-0.0,-0.0,-0.0,-0.0,-0.0,
        -0.0,-1.0,1.1179883994595727E-5,-1.7242506299916662E-9,0.99990778299340233,1.2647726762421167E-9,0.0,0.0,
        0.0,0.0,0.0,0.0,0.0,-0.0,-0.0,-0.0,-0.0,-0.0,-0.0,-0.0,-1.0,-0.99990778299340177,1.5536028954057082E-18,
        3.5775740920850794E-27,0.0,0.0,0.0,0.0,0.0,0.0,0.0,0.0,0.0,1.0,-0.0,-0.0,-0.0,-0.0,-0.0,-0.0,-0.0,
        -0.99990778299340177,-3.5775740920850787E-27,1.5536028954057082E-18,0.0,0.0,0.0,0.0,0.0,0.0,0.0,0.0,0.0,1.0,
        -0.0,-0.0,-0.0,-0.0,-0.0,-0.0,-1.4213196200012445E-22,0.99983604883715416,-1.6542089733208698E-24,
        -2.4515194437399741E-14,0.0,0.0,0.0,0.0,0.0,0.0,0.0,0.0,-0.0,-0.0,-0.0,-0.0,-0.0,-0.0,-0.0,-1.0,
        1.1179883994613772E-5,-7.4738609228964824E-10,0.99990778299340144,3.8124483816308815E-8,0.0,0.0,0.0,0.0,0.0,
        0.0,0.0,0.0,-0.0,-0.0,-0.0,-0.0,-0.0,-0.0,-0.0,-1.0,9.4420602018476818E-27,0.99990778299340177,
        2.319246843608249E-18,0.0,0.0,0.0,0.0,0.0,0.0,0.0,0.0,-0.0,-0.0,-0.0,-0.0,-0.0,-0.0,-0.0,-1.0,
        -0.99990778299963246,-5.6348491829692715E-15,-8.3371555091865689E-23,0.0,-2.4506968300103951E-14,0.0,0.0,
        0.0,0.0,0.0,0.0,0.0,1.0,-0.0,-0.0,-0.0,-0.0,-0.0,-0.0,9.6852328378879643E-25,0.99983604883715438,
        -1.6542089733311629E-24,1.8260333355478996E-22,0.0,0.0,0.0,0.0,0.0,0.0,0.0,0.0,-0.0,-0.0,-0.0,-0.0,-0.0,
        -0.0,-1.0,1.1179883994611302E-5,-3.3893748116090767E-8,0.99990778299340177,5.7482274508680952E-10,0.0,0.0,
        0.0,0.0,0.0,0.0,0.0,0.0,-0.0,-0.0,-0.0,-0.0,-0.0,-0.0,-0.0,-1.0;
    Explicit_b_G: ARRAY [0..201] OF LREAL := 0.0,0.0,150.328,-6.91852455976248E-7,-6.9185245628696185E-7,150.328,
        50.109284275633563,-3.7104784955705769E-7,0.0,0.0,0.0,0.0,0.0,0.0,0.0,0.0,150.32800000000003,150.328,
        150.32800000000006,-6.9185269075425606E-7,150.32800000000003,0.0,150.32800000000003,-2.9401439680058069E-7,
        -6.9185275549905575E-7,150.32799999999997,1.0587911840678754E-22,150.328,-3.2080502011972351E-7,150.328,
        75.163965609645246,75.16396561995829,0.0,0.0,0.0,0.0,0.0,0.0,0.0,0.0,0.0,0.0,0.0,0.0,0.0,0.0,0.0,0.0,
        150.32800000000003,150.328,150.32800000000003,150.328,150.32800000000003,-2.9401449611845737E-7,
        150.32800000000003,7.9282982220735976E-24,150.32800000000003,-1.6140379585977151E-7,-5.3044909714511956E-7,
        75.163965738154118,-6.9185279582694362E-7,150.32799999999997,-3.2080515874285942E-7,150.32799999999997,
        2.6016506436444134E-24,150.328,-1.8435894428542776E-7,150.328,75.163965609647164,75.1639656199583,
        75.163965609645231,75.163965619960209,150.32799999999997,75.163965576748325,0.0,0.0,0.0,0.0,0.0,0.0,0.0,0.0,
        0.0,0.0,0.0,0.0,0.0,0.0,0.0,0.0,0.0,0.0,0.0,0.0,0.0,0.0,0.0,0.0,50.109284275633563,-8.64894981308275E-8,
        75.163965566437255,150.32799999999997,150.328,150.32800000000003,150.328,75.163965576750329,
        75.163965750794262,-5.0749395296266035E-7,150.32800000000003,-1.0322514419702163E-22,50.109284275633563,
        -1.5741089761767257E-7,150.32800000000003,-1.6140385050947835E-7,75.1639657507962,7.9409338805090657E-23,
        150.32800000000003,-2.0520544064205554E-23,150.32800000000003,-1.6307686042414295E-22,-5.304491307562495E-7,
        75.163965738152186,0.0,75.163965738154118,-7.574505465679009E-23,75.163965738154118,-3.2080517723865736E-7,
        150.32799999999997,5.1735997275741694E-23,150.32799999999997,-2.4589082840120078E-7,75.163965738154118,
        -1.8435902369178403E-7,150.32799999999997,-1.220985151366895E-22,150.328,75.163965609647164,
        75.163965619960237,75.16396556643717,150.32799999999997,75.163965750794262,-2.9798554896119714E-23,150.328,
        75.163965576750272,8.28551526588557E-23,75.163965738152186,150.328,75.163965576748339,
        -1.1418256732094804E-23,150.328,0.0,0.0,0.0,0.0,0.0,0.0,0.0,0.0,50.109284275633563,-8.2376137384543772E-24,
        0.0,0.0,75.163965750794262,-1.1819388395491361E-7,75.163965566435323,150.32799999999997,150.328,150.328,
        75.163965750794262,-2.152743225402716E-7,150.32800000000003,-1.2569896466053958E-22,150.32800000000003,
        -1.614038636547713E-7,150.32800000000003,-7.5445647233378886E-23,-1.4114904573254368E-7,75.163965738154118,
        2.2027905792789105E-23,75.163965738154118,6.9032271182804478E-24,150.32799999999997,-1.2349344840906095E-22,
        75.163965738152186,-2.4589084381645556E-7,75.163965738152186,-1.8435903420069689E-7,150.328,
        75.163965566435238,150.32799999999995,75.163965750794262,-2.2257723062585332E-23,4.3569393640531692E-23,
        75.163965738152186,75.163965750794262,1.2959911821950123E-23,75.163965566435252,150.32799999999997,
        75.1639657507962,-1.1810916980833994E-22,-1.4114905449115833E-7,75.163965738152186;
    Explicit_b_F: ARRAY [0..2019] OF LREAL := -0.0029164395371222415,-3.0087605677823286E-6,1.4746159915543362E-20,
        -3.0087739900712996E-6,-0.0029164395371360889,5.9942806311391553E-22,-0.0012961974435727582,
        -3.0087725653064055E-6,1.4746159915543362E-20,-3.0087739900712996E-6,-0.0029164395371360889,
        5.9942806311391553E-22,-0.0012961974435727582,-3.0087725653064055E-6,-0.0029164395371336187,
        -1.5758035741956111E-6,3.90002488989466E-19,4.6091650798319766E-22,9.2865808078981142E-20,
        -3.0087767144956264E-6,3.90002488989466E-19,4.6091650798319766E-22,4.4077773510571569E-19,
        -1.5758092782242111E-6,-0.0029164395371387279,-3.5258573610072805E-23,5.1189790559257405E-20,
        -2.0082515478174017E-22,-0.0012961974435791795,-3.9336234756661114E-22,-0.00072911137556484859,
        -9.66878533608266E-7,3.90002488989466E-19,4.6091650798319766E-22,1.3569901251104168E-19,
        -3.0087771245688761E-6,4.4077773510571569E-19,-1.5758092782242111E-6,-0.001296197443580489,
        -4.29778489358118E-23,-0.0029164395371382417,-9.1186969011167945E-23,-0.00072911137556096433,
        -3.0087756536188372E-6,-0.0012961974435780257,-1.5758086639462633E-6,-0.0029164395371368414,
        -9.6687501944711621E-7,1.5247546214998093E-19,4.5283685575240474E-22,2.9211082452448389E-19,
        4.2369741938614614E-22,-1.7508198924691168E-19,-1.5758104307343709E-6,2.6324605330918856E-19,
        2.1442516727484835E-22,2.4709234988577E-19,-9.66878150762717E-7,-0.0029164395371366518,
        -9.6687500855267628E-7,-0.0029164395371389178,-4.3032778898364151E-23,-0.0012961974435804022,
        -1.9152623913583765E-22,-5.6555354446597829E-19,2.4312062010187407E-23,-0.00072911137556465431,
        5.0948146112479365E-22,-0.0007291113509555661,-9.6687845897825868E-7,-0.00072911137556479916,
        -9.66878522713679E-7,-3.5237188618896909E-19,-9.6687895275670673E-7,1.1207185239798877E-19,
        6.8605251308477482E-22,-1.2992910071087124E-19,1.7723233196872259E-22,-0.00072911135095168151,
        -3.0087753362390236E-6,3.3881248386625513E-19,6.6174183497744866E-22,2.4709234988577E-19,
        -9.66878150762717E-7,-1.7508198924691168E-19,-1.5758104307343709E-6,-0.0012961974435795251,
        -9.6687781601321224E-7,-0.0029164395371389178,-4.3032778898364151E-23,-0.0012961974435804022,
        -1.9152543134227071E-22,-0.00072911137556540392,4.5971148192970549E-22,-0.00072911137556465431,
        5.0948146112479365E-22,1.1837218885155262E-19,-3.0087774419487986E-6,-0.0012961974435795251,
        -9.6687781601321287E-7,-0.00072911135095537181,1.8516688428005278E-22,-2.0572240624510263E-19,
        7.3697155875947467E-22,2.7584732516084758E-19,-9.6687813986814716E-7,-0.00072911137556096433,
        -3.0087756536188372E-6,-2.0572240624194719E-19,7.522800742885925E-23,-0.0012961974435780257,
        -1.5758086639462633E-6,-3.7259654887668772E-19,-9.6687878493195554E-7,-0.00072911135095537181,
        1.8516688428005278E-22,-1.2992910071087124E-19,1.7723233196872259E-22,3.1911761139338214E-19,
        -2.0268802772131424E-22,-0.0029164395371368414,-9.6687501944711579E-7,2.7584732516084758E-19,
        -9.6687813986814716E-7,-3.2293715608882783E-19,-9.6687894186210247E-7,-0.001296197443580489,
        -4.29778489358118E-23,-3.2910435045709359E-19,-2.1660883523469598E-23,-0.0012961974435794388,
        -9.6687780511865541E-7,-0.00072911137556535481,-2.3167640669055387E-22,-5.4453539641500664E-19,
        7.36972214559144E-22,-0.000729111350955516,-9.6687844808367475E-7,-0.00072911135095612175,
        -1.2430165849456523E-22,-0.00072911137556465463,-1.5226020164014417E-22,3.5468897875806594E-19,
        -9.6687894186210247E-7,2.4709234988577E-19,-9.66878150762717E-7,6.1643146140530539E-21,
        -9.668788781266734E-7,-3.58507371889038E-19,4.5905858277922113E-22,2.6324605330918856E-19,
        2.1442516727484835E-22,-1.3559453738203046E-20,-9.66878952756707E-7,-4.1191914752465146E-19,
        1.1673566199815429E-22,-0.0012961974435794388,-9.6687780511865583E-7,-0.0012961974435804888,
        -4.2979464522945694E-23,-0.00072911137556484827,-9.6687853360826639E-7,-0.00072911137556484859,
        -9.668785336082666E-7,-0.00072911137556465463,5.0948327866031928E-22,3.5878681390286741E-19,
        1.1796118581340772E-22,-0.000729111375563985,-1.5758099736233452E-6,-5.3159669650882034E-20,
        -1.838773844869355E-22,-3.5237188618896909E-19,-9.6687895275670673E-7,-3.7211006004588216E-19,
        2.5498948049391836E-22,-0.0007291113755647984,-9.6687852271367865E-7,-4.4900563865746895E-21,
        -9.6687877403735827E-7,-6.48080476023491E-19,6.6291516313847638E-22,-3.5237246966599333E-19,
        -9.66878952756706E-7,-0.0012961974435795251,-9.6687781601321224E-7,-0.00072911137556540392,
        4.59711078032922E-22,-0.00072911137556540425,4.5971269362005591E-22,-0.00072911137556522264,
        -6.3298057671059772E-22,-3.7259613528835359E-19,-9.6687878493195512E-7,-0.00072911137556540425,
        -8.63773459187304E-22,-0.00072911137556535481,-2.3167681058733735E-22,-0.00072911135095594026,
        4.2740398016807932E-22,-0.00072911137556484794,-9.6687853360826575E-7,-5.5801566790146211E-6,
        -0.0029177101087786779,-1.6389065185832384E-21,-0.0029177101088043592,-5.5801701071511332E-6,
        5.0983324695593649E-20,-2.9222208231492036E-6,-0.0029177101087983592,-1.6389065185832384E-21,
        -0.0029177101088043592,-5.5801701071511332E-6,5.0983324695593649E-20,-2.9222208231492036E-6,
        -0.0029177101087983592,-5.5801695483969938E-6,-0.0012967620736893976,-7.5797128311776815E-22,
        -5.0191577480533521E-19,-8.8508002425747183E-22,-0.0029177101088077133,-7.5797128311776815E-22,
        -5.0191577480533521E-19,-5.2748919921594441E-23,-0.0012967620737003112,-5.5801736885504331E-6,
        -6.5108391653930784E-21,-7.5797451429203594E-22,1.7570962175689255E-19,-2.922227049640943E-6,
        2.1700171146092924E-19,-1.7928626865170363E-6,-0.00072942895215362825,-7.5797128311776815E-22,
        -5.0191577480533521E-19,-9.1544013767758217E-22,-0.0029177101088086466,-5.2748919921594441E-23,
        -0.0012967620737003112,-2.9222289056339786E-6,-3.5069394866058623E-19,-5.5801733527413591E-6,
        2.3574492714806121E-21,-1.7928584653930106E-6,-0.0029177101088045097,-2.9222267817484178E-6,
        -0.0012967620736977473,-5.5801725512051323E-6,-0.000729428952147611,-7.3014602591073535E-22,
        -6.5371512426678573E-19,-1.0998200290750375E-21,-5.8700007318659363E-19,-1.1378208598965013E-21,
        -0.0012967620737017304,-3.6435840824989949E-22,-7.3623072774625E-19,1.8257689615603115E-22,
        -0.00072942895215360255,-5.580172122209582E-6,-0.000729428927518466,-5.580174117546102E-6,
        1.8654226966123439E-19,-2.9222287088813688E-6,1.367563509935531E-19,-1.3738936830751605E-21,
        -2.8792811603551195E-20,-1.7928620436083493E-6,-1.0045747739090933E-19,-1.7928626663050662E-6,
        -0.00072942895215356645,-1.7928625747264864E-6,-0.00072942892752448285,-1.9551940507532338E-21,
        -0.00072942895215465889,-7.1214757744560448E-22,-7.064182081689344E-19,-7.6414777370483555E-22,
        -5.7585938452643967E-19,-1.7928584451811547E-6,-0.002917710108804249,-1.3234867026511342E-21,
        -3.3881266388849837E-19,1.8257689615603115E-22,-0.00072942895215360255,-1.1378208598965013E-21,
        -0.0012967620737017304,-2.922228178628247E-6,-0.00072942895215219916,-5.580174117546102E-6,
        1.8654226966123439E-19,-2.9222287088813688E-6,1.367563509935531E-19,-1.7928631058480436E-6,
        2.1203101473829483E-21,-1.7928620436083493E-6,-1.0045747739090933E-19,-1.4430424279928991E-21,
        -0.0029177101088089072,-2.9222281786282466E-6,-0.00072942895215219884,-1.7928620233963966E-6,
        3.5992481455209706E-19,-2.0783890320610825E-21,-9.7827432441169576E-20,-8.32683302331066E-22,
        -0.00072942892752445715,-1.7928584653930112E-6,-0.0029177101088045097,-2.0783874164739486E-21,
        -4.3664013072233664E-19,-2.9222267817484178E-6,-0.0012967620736977473,-1.880650658447036E-21,
        -0.0007294289521543834,-1.7928620233963966E-6,-3.1770058201091956E-19,-7.6414777370483555E-22,
        -5.7585938452643967E-19,-2.0582834472508008E-21,-2.6819878620026619E-19,-5.5801725512051323E-6,
        -0.000729428952147611,-1.4944265806831377E-21,-0.00072942892752445715,-2.8131592722458021E-21,
        -0.00072942892752551414,-2.9222289056339786E-6,-3.5069394866058623E-19,-1.8201829175835839E-21,
        -1.1839167802605035E-19,-2.9222279818756914E-6,-0.00072942892752305365,-1.7928629940574621E-6,
        -1.8723254121306615E-19,-2.7401335221035047E-21,-9.7827432441311156E-20,-1.7928625545145193E-6,
        -0.00072942892752442126,-1.7928630856360625E-6,1.241877027010887E-19,-1.79286204360835E-6,
        -1.0045747738775389E-19,-1.4896787739934107E-21,-0.00072942892752551306,-1.8026535447453592E-21,
        -0.00072942895215360255,4.1215263567574113E-22,-0.0007294289521545972,-2.0582836641582989E-21,
        7.0614281179398917E-20,-3.6435840824989949E-22,-7.3623072774625E-19,-1.9551942527016255E-21,
        -0.00072942895215465889,-1.8525203581942851E-21,-4.4570690558405966E-19,-2.9222279818756914E-6,
        -0.00072942892752305365,-2.9222289056339786E-6,-3.5069404305883759E-19,-1.7928626865170357E-6,
        -0.00072942895215362825,-1.7928626865170363E-6,-0.00072942895215362825,-1.79286204360835E-6,
        -1.0045747738696503E-19,-1.0049913038232996E-21,-5.5539026188194611E-19,-1.7928618819771793E-6,
        -0.0012967620737003554,-2.2737919734988914E-21,-8.5484454210397229E-19,-1.9551966760823263E-21,
        -0.00072942895215465857,-1.055605347214035E-21,-3.9388775174516995E-19,-1.7928625747264864E-6,
        -0.00072942892752448317,-1.9223960163480794E-21,-0.00072942892752523756,-3.2250957726552871E-21,
        1.4998492264970375E-19,-2.6169387427440476E-21,-0.00072942895215465889,-2.922228178628247E-6,
        -0.00072942895215219916,-1.7928631058480436E-6,2.1202586323992547E-21,-1.7928631058480444E-6,
        2.1203101513272529E-21,-1.7928629008220827E-6,-1.7598440052001331E-19,-2.5423977738185507E-21,
        -0.00072942895215438307,-1.7928631058480444E-6,-3.3669272290815531E-19,-1.7928629940574628E-6,
        -1.8723254120912184E-19,-1.7928628806101064E-6,-5.40081611373621E-20,-1.7928626865170363E-6,
        -0.00072942895215362858,-1.0698028313139132E-5,-1.2162732220465626E-8,2.2051104858713465E-21,
        -1.2162781455851999E-8,-1.0698028313195108E-5,-1.4002849047524719E-24,-4.329828358931141E-6,
        -1.2162779375537441E-8,2.2051104858713465E-21,-1.2162781455851999E-8,-1.0698028313195108E-5,
        -1.4002849047524719E-24,-4.329828358931141E-6,-1.2162779375537441E-8,-1.0698028313186529E-5,
        -6.1928203495312775E-9,2.4928031530932895E-21,-3.4295191429067938E-24,3.3238397175753927E-21,
        -1.2162793235522465E-8,2.4928031530932895E-21,-3.4295191429067938E-24,3.7276985366953231E-21,
        -6.1928412729410324E-9,-1.0698028313206726E-5,-1.6982218914363436E-24,2.4928031530809635E-21,
        -8.445828841222032E-25,-4.3298283589570983E-6,-8.2960714869748751E-25,-2.2920794507502355E-6,
        -3.7151729700733621E-9,2.4928031530932895E-21,-3.4295191429067938E-24,2.1601509362507816E-21,
        -1.2162794597864248E-8,3.7276985366953231E-21,-6.1928412729410324E-9,-4.3298283589628895E-6,
        -1.2801666324362788E-24,-1.0698028313204698E-5,-1.673773514261734E-24,-2.29207945073414E-6,
        -1.2162790472980387E-8,-4.3298283589530851E-6,-6.19284035428859E-9,-1.0698028313199644E-5,
        -3.7151593998661597E-9,2.3661681426070936E-21,-2.2009201506295862E-24,4.8306963647989115E-21,
        -2.38191186077329E-24,2.1293539687975141E-21,-6.1928462560817878E-9,3.1038150383602712E-21,
        -1.6021670321730123E-24,4.2279500917169585E-21,-3.7151708860987843E-9,-1.0698028313198748E-5,
        -3.7151593484790163E-9,-1.0698028313207622E-5,-2.7602558618045291E-25,-4.3298283589624787E-6,
        -1.7737695226075495E-24,2.2148361989266378E-21,-1.4229591337512394E-25,-2.2920794507490565E-6,
        3.2090309421757106E-25,-2.2920793346729468E-6,-3.7151726180578695E-9,-2.292079450750003E-6,
        -3.7151729186856475E-9,1.1347909684699084E-21,-3.71517428773423E-9,2.214836198937423E-21,
        -2.7272317777292619E-24,4.4603707999340415E-21,-4.2586498196175278E-25,-2.2920793346568523E-6,
        -1.2162788975960414E-8,1.3234879748306531E-21,-2.5849413087365402E-24,4.2279500917169585E-21,
        -3.7151708860987843E-9,2.1293539687975141E-21,-6.1928462560817878E-9,-4.3298283589591871E-6,
        -3.7151703914902866E-9,-1.0698028313207622E-5,-2.7602558618045291E-25,-4.3298283589624787E-6,
        -1.7737695226075495E-24,-2.2920794507523713E-6,-1.4027106520360265E-24,-2.2920794507490565E-6,
        3.2090309421757106E-25,1.8663263797776173E-21,-1.2162796094884658E-8,-4.3298283589591871E-6,
        -3.7151703914902879E-9,-2.2920793346717677E-6,-2.298642859061781E-24,2.0630415433417094E-21,
        -1.5632739395369735E-24,3.3074148719158428E-21,-3.7151708347111624E-9,-2.29207945073414E-6,
        -1.2162790472980387E-8,2.0630415433417094E-21,-1.5632739395369735E-24,-4.3298283589530851E-6,
        -6.19284035428859E-9,1.2898398633043176E-21,-3.7151736280742449E-9,-2.2920793346717677E-6,
        -2.298642859061781E-24,4.4603707999340415E-21,-4.2586498196175278E-25,1.4806022601830657E-21,
        -3.2847036078003939E-24,-1.0698028313199644E-5,-3.7151593998661597E-9,3.3074148719158428E-21,
        -3.7151708347111624E-9,2.1718080623884192E-22,-3.7151742363464611E-9,-4.3298283589628895E-6,
        -1.2801666324362788E-24,1.8863514816444509E-21,-8.49070319381553E-25,-4.3298283589587788E-6,
        -3.7151703401026796E-9,-2.292079450752138E-6,-1.1242435413539145E-24,2.0630415433417094E-21,
        -1.5632739395369735E-24,-2.2920793346727159E-6,-3.71517256667017E-9,-2.2920793346750838E-6,
        -3.2743738686769774E-24,-2.2920794507490565E-6,-2.2640323757061143E-24,1.5406685798826504E-21,
        -3.7151742363464611E-9,1.5809758852109242E-21,-3.7151708860987843E-9,2.7630471405797742E-21,
        -3.7151739357186338E-9,1.4806022601761576E-21,-6.9976616572444551E-25,3.1038150383602712E-21,
        -1.6021670321730123E-24,1.1347909684575824E-21,-3.7151742877342286E-9,1.942950394120331E-22,
        -1.5492719363256804E-24,-4.3298283589587788E-6,-3.7151703401026796E-9,-4.3298283589628895E-6,
        -1.2801666324362788E-24,-2.2920794507502355E-6,-3.7151729700733638E-9,-2.2920794507502355E-6,
        -3.7151729700733621E-9,-2.2920794507490565E-6,3.2090309421757106E-25,1.6293586887755402E-21,
        -2.4744992819277224E-24,-2.2920794507467216E-6,-6.1928450604402566E-9,1.3616791324040542E-21,
        -1.2778138200937181E-24,1.1347909684591232E-21,-3.7151742877342286E-9,2.9905214339681706E-21,
        -9.6589647792503236E-25,-2.2920794507500047E-6,-3.7151729186856475E-9,1.6951459367374617E-21,
        -3.7151735766865038E-9,1.7298074573895735E-21,-2.3755817470024252E-24,-1.8869690576445074E-22,
        -3.71517428773423E-9,-4.3298283589591871E-6,-3.7151703914902879E-9,-2.2920794507523713E-6,
        -1.4027082854533108E-24,-2.2920794507523713E-6,-1.402709074314216E-24,-2.2920794507515891E-6,
        -3.7748650922726379E-24,-1.3571343432125019E-21,-3.7151736280742437E-9,-2.2920794507523713E-6,
        -1.4027106520360265E-24,-2.292079450752138E-6,-1.1242443302148198E-24,-2.292079334674302E-6,
        -2.860078320751196E-24,-2.2920794507502355E-6,-3.7151729700733621E-9,-4.178067495524499E-8,
        -1.9827341852663573E-5,3.0999330567054551E-24,-1.982734185285586E-5,-4.1780766206343672E-8,
        1.1483344185991915E-21,-2.1271108785988041E-8,-1.9827341852815443E-5,3.0999330567054551E-24,
        -1.982734185285586E-5,-4.1780766206343672E-8,1.1483344185991915E-21,-2.1271108785988041E-8,
        -1.9827341852815443E-5,-4.1780768652100644E-8,-8.0258637655188359E-6,6.5835554359359267E-24,
        -1.7415634159483883E-21,7.069304426934817E-24,-1.9827341852883534E-5,6.5835554359359267E-24,
        -1.7415634159483883E-21,1.0218405606140887E-23,-8.0258637656005542E-6,-4.1780794019391373E-8,
        4.7650071065816442E-22,6.58353019238696E-24,3.5523849946940161E-21,-2.1271151098204015E-8,
        -3.8728504547781949E-22,-1.2759918411572972E-8,-4.2489662642285167E-6,6.5835554359359267E-24,
        -1.7415634159483883E-21,8.783189940505229E-24,-1.9827341852890815E-5,1.0218405606140887E-23,
        -8.0258637656005542E-6,-2.1271165702455609E-8,-3.5403737218960277E-22,-4.1780792197784326E-8,
        -5.1762496666617975E-22,-1.2759888180732203E-8,-1.9827341852861796E-5,-2.1271152168179534E-8,
        -8.0258637655832629E-6,-4.17807886426461E-8,-4.2489662641823483E-6,6.8274018080706041E-24,
        -2.0408099337760396E-21,1.4513540242624887E-23,-2.6245608513973591E-21,4.0969207122727369E-24,
        -8.02586376561226E-6,1.2183166214388439E-23,-1.7477145252994458E-21,1.1506364606598939E-23,
        -4.24896626422721E-6,-4.1780784895364554E-8,-4.248966049046449E-6,-4.1780797766673767E-8,
        -1.2651754897199195E-21,-2.1271163983819168E-8,1.4115926631244706E-21,1.8357550570961957E-24,
        3.0650926316371844E-21,-1.2759912496547035E-8,1.7943261545190228E-21,-1.2759918235021132E-8,
        -4.2489662642279814E-6,-1.2759917435081107E-8,-4.2489660490926225E-6,8.6415767862435738E-25,
        -4.24896626423585E-6,7.0056465073271022E-24,-2.2288557790360349E-21,1.5834724486689037E-23,
        -9.5788948871376226E-22,-1.275988800418117E-8,-1.9827341852859519E-5,5.1699104354313342E-24,
        -2.6469672307959184E-21,1.1506364606598939E-23,-4.24896626422721E-6,4.0969207122727369E-24,
        -8.02586376561226E-6,-2.1271161467604748E-8,-4.2489662642177484E-6,-4.1780797766673767E-8,
        1.3818031415731842E-21,-2.1271163983819168E-8,1.4115969040406971E-21,-1.2759920854200594E-8,
        -8.7624833390359249E-22,-1.2759912496547035E-8,1.7943261545190228E-21,7.7961166887947649E-24,
        -1.9827341852893092E-5,-2.1271161467604748E-8,-4.2489662642177458E-6,-1.2759912319995349E-8,
        -3.0713008667882647E-22,4.2534559594175527E-24,-2.5876045648300193E-21,9.69029951769706E-24,
        -4.2489660490913079E-6,-1.2759888180732203E-8,-1.9827341852861796E-5,4.2534496485303109E-24,
        -2.5876045648312851E-21,-2.1271152168179534E-8,-8.0258637655832629E-6,2.9723821369402697E-24,
        -4.2489662642336506E-6,-1.2759912319995349E-8,-3.0713008667882647E-22,1.5834724486689037E-23,
        -9.5788948871376226E-22,5.9142405958192544E-24,-2.2757050939522553E-21,-4.17807886426461E-8,
        -4.2489662641823458E-6,9.6903184503587853E-24,-4.2489660490913104E-6,7.4658111614478646E-25,
        -4.2489660490999561E-6,-2.1271165702455609E-8,2.292932407159698E-21,3.5665750477189872E-24,
        2.1463268111786541E-21,-2.1271159748968694E-8,-4.2489660490818491E-6,-1.2759919877708509E-8,
        -1.7508389234842942E-21,4.2534559594175527E-24,-2.5876045648244631E-21,-1.2759917258529288E-8,
        -4.2489660490920846E-6,-1.2759920677648682E-8,-3.2670583055042819E-22,-1.2759912496547035E-8,
        1.7943261545190228E-21,7.4658584931021778E-25,-4.2489660490999561E-6,1.1506336207606351E-23,
        -4.2489662642272046E-6,7.1509878182268318E-24,-4.2489662642353124E-6,-4.4255354188322139E-24,
        3.01824056750065E-21,1.2183166214388439E-23,-1.7477145252994458E-21,8.64170300398841E-25,
        -4.2489662642358528E-6,-3.1154933380609395E-24,1.1681640746618562E-21,-2.1271159748968694E-8,
        -4.2489660490818516E-6,-2.1271165702455609E-8,-3.0010125162244673E-21,-1.2759918411572972E-8,
        -4.2489662642285218E-6,-1.2759918411572977E-8,-4.2489662642285218E-6,-1.2759912496547035E-8,
        1.7943261545190228E-21,4.8700899088737231E-24,-2.0961503398396257E-21,-1.2759913055522955E-8,
        -8.0258637656029175E-6,1.6393160699216802E-25,-1.8478891562861802E-21,1.1203913757815393E-23,
        -4.2489662642358528E-6,1.3646239742154129E-23,-1.2977603354642251E-21,-1.2759917435081107E-8,
        -4.2489660490926174E-6,6.81774930603432E-24,-4.2489660490977479E-6,4.0291922703940817E-24,
        -8.7040605759657524E-22,6.0340428179680221E-24,-4.2489662642358528E-6,-2.1271161467604748E-8,
        -4.2489662642177458E-6,-1.2759920854200594E-8,-8.7625296111514349E-22,-1.2759920854200594E-8,
        -8.7625168683361062E-22,-1.2759919361313784E-8,-8.3557908379380824E-23,2.9723442716168191E-24,
        -4.2489662642336446E-6,-1.2759920854200599E-8,-3.5232231428821135E-21,-1.2759919877708504E-8,
        -1.750838923515109E-21,-1.2759919184761911E-8,4.6528859010301811E-22,-1.2759918411572972E-8,
        -4.2489662642285142E-6,-0.019097634712978588,-1.9705949370788169E-5,4.8688115523384709E-18,
        -1.9706037263565827E-5,-0.019097634713069283,-3.7095690051764795E-21,-0.0084864283463426012,
        -1.9706027944357129E-5,4.8688115523384709E-18,-1.9706037263565827E-5,-0.019097634713069283,
        -3.7095690051764795E-21,-0.0084864283463426046,-1.9706027944357129E-5,-0.019097634713053105,
        -1.0320169370790202E-5,8.1421669077312929E-18,-6.4597506714592294E-21,6.2474553412857983E-18,
        -1.970605510981498E-5,8.1421669077312929E-18,-6.4597506714592294E-21,6.6664748607846E-18,
        -1.0320206722311879E-5,-0.019097634713086568,-6.4665102880274361E-21,5.4316653202643806E-18,
        -6.4597377467621582E-21,-0.00848642834638466,-3.8826500860046649E-21,-0.0047731377301323081,
        -6.3319463279187473E-6,8.1421669077312929E-18,-6.4597506714592294E-21,4.7954262503134087E-18,
        -1.9706057794609424E-5,6.6664748607846E-18,-1.0320206722311879E-5,-0.0084864283463932377,
        -3.4546875165850422E-21,-0.019097634713083383,-7.0346282724865125E-21,-0.004773137730106871,
        -1.970604816668707E-5,-0.0084864283463771065,-1.0320202704323961E-5,-0.019097634713074216,
        -6.3319233139652047E-6,5.229456703948615E-18,-6.2450140997643232E-21,4.9161993963896509E-18,
        -5.288630945146067E-21,-1.9351312724486906E-19,-1.0320214271790599E-5,5.7439423917783E-18,
        -8.8634567521816331E-21,6.7823735013844217E-18,-6.3319438186664894E-6,-0.019097634713072971,
        -6.3319232425871977E-6,-0.019097634713087813,-3.3911044693435638E-21,-0.0084864283463926687,
        -4.94551254964995E-21,1.2763973429718635E-18,-5.0106974515346828E-21,-0.0047731377301310383,
        -5.2588556742684258E-21,-0.0047731375688976167,-6.3319458389590979E-6,-0.0047731377301319855,
        -6.3319462565397721E-6,3.7659262455952018E-18,-6.3319490718798243E-6,6.69740196547176E-18,
        -5.0107176463738564E-21,6.3123784754145422E-18,-5.3129552250339545E-21,-0.0047731375688721779,
        -1.9706046087283249E-5,2.7105055694445983E-18,-5.2939536887208516E-21,6.7823735013844217E-18,
        -6.3319438186664894E-6,2.5169930097154123E-18,-1.0320214271790599E-5,-0.0084864283463869285,
        -6.33194162909236E-6,-0.019097634713087813,-6.0380824295132524E-21,-0.0084864283463926687,
        -4.9455060873014142E-21,-0.0047731377301359519,-7.0201186844370227E-21,-0.0047731377301310383,
        -5.2588556742684258E-21,4.7296674346768351E-18,-1.9706059874013961E-5,-0.0084864283463869251,
        -6.3319416290923626E-6,-0.0047731375688963469,-7.35150791734108E-21,5.1502136035375756E-18,
        -5.8109876162706659E-21,5.9539113998961089E-18,-6.3319437472876285E-6,-0.004773137730106871,
        -1.970604816668707E-5,-2.7078806088538766E-19,-5.81095886920263E-21,-0.0084864283463771048,
        -1.0320202704323961E-5,5.3183074545448137E-18,-6.3319479727705775E-6,-0.0047731375688963443,
        -2.0575778463958446E-21,6.3123784754145422E-18,-5.3129552250339545E-21,4.2663504849142025E-18,
        -5.5967411830378648E-21,-0.019097634713074216,-6.3319233139652022E-6,5.9539113998961089E-18,
        -6.3319437472876285E-6,2.3142137821508769E-19,-6.3319490005007373E-6,-0.0084864283463932377,
        -6.1016590144061952E-21,6.1526402695137655E-18,-5.2412788940452409E-21,-0.00848642834638636,
        -6.3319415577135814E-6,-0.0047731377301356267,-7.9909056061474987E-21,2.4397153806633983E-18,
        -5.8109673616377915E-21,-0.0047731375688972915,-6.331945767580143E-6,-0.0047731375689012579,
        -5.7393022073196845E-21,-0.0047731377301310383,-2.6118841764472728E-21,2.9419194635277004E-18,
        -6.3319490005007373E-6,4.0718719139017322E-18,-6.3319438186664868E-6,3.8473851895529522E-18,
        -6.3319485829200054E-6,-1.1546481405436232E-18,-2.9497325267126323E-21,5.7439423917783E-18,
        -8.8634567521816331E-21,6.4764298931487022E-18,-6.3319490718798243E-6,2.1305194015399455E-18,
        -9.1307604902455708E-21,-0.00848642834638636,-6.3319415577135839E-6,-0.0084864283463932343,
        -6.1016784014518019E-21,-0.0047731377301323107,-6.3319463279187473E-6,-0.0047731377301323081,
        -6.3319463279187473E-6,-0.0047731377301310383,-5.2588605210298275E-21,8.2146077167090343E-18,
        -7.6481252722591485E-21,-0.0047731377301266529,-1.0320211280114997E-5,3.2868157645701836E-18,
        -6.3549205181106827E-21,3.7659262455920463E-18,-6.3319490718798243E-6,6.0796869129044207E-18,
        -4.3719641729370769E-21,-0.0047731377301319855,-6.33194625653977E-6,1.7828764048777283E-18,
        -6.3319479013915345E-6,4.597720374387205E-18,-6.6111019074067265E-22,1.0554249332230198E-18,
        -6.3319490718798217E-6,-0.0084864283463869285,-6.33194162909236E-6,-0.0047731377301359519,
        -4.37314718661587E-21,-0.0047731377301359519,-7.0201251467855583E-21,-0.004773137730134761,
        -3.3661662663447971E-21,-1.0268951653126124E-19,-6.3319479727705775E-6,-0.0047731377301359493,
        -4.3731633424872087E-21,-0.0047731377301356267,-5.3439324927392118E-21,-0.004773137568900067,
        -3.0421214925514163E-21,-0.0047731377301323107,-6.3319463279187448E-6,-3.6535670676475959E-5,
        -0.01910040755447192,2.4094220280021159E-21,-0.019100407554640066,-3.6535758582015063E-5,
        -9.1772683720778245E-19,-1.9132097398897662E-5,-0.019100407554600789,2.4094220280021159E-21,
        -0.019100407554640066,-3.6535758582015063E-5,-9.1772683720778245E-19,-1.9132097398897662E-5,
        -0.019100407554600789,-3.6535754933752659E-5,-0.0084878806162073227,9.5894596048875008E-21,
        -2.9635443265168115E-18,5.073215019061359E-21,-0.019100407554662031,9.5894596048875008E-21,
        -2.9635443265168115E-18,1.2784690290117922E-20,-0.0084878806162787812,-3.6535782032491541E-5,
        -2.2854837212386326E-18,4.2954972221995882E-21,-2.5304274024265693E-19,-1.9132138159811332E-5,
        -2.6799900119830713E-18,-1.1737622548725761E-5,-0.0047740288164251033,9.5894596048875008E-21,
        -2.9635443265168115E-18,8.5218860891597851E-21,-0.019100407554668141,1.2784690290117922E-20,
        -0.0084878806162787812,-1.9132150312873025E-5,-3.9694314746272033E-18,-3.6535779834867094E-5,
        -2.529287210793528E-18,-1.1737594913325115E-5,-0.019100407554641059,-1.9132136410508959E-5,
        -0.0084878806162619943,-3.6535774590606786E-5,-0.0047740288163857069,4.09262794579669E-21,
        -4.4611413024616849E-18,1.0138752364165677E-20,-4.5119467335133523E-18,-1.4407159825200937E-21,
        -0.0084878806162880724,1.0192679423238228E-20,-4.2885469058092407E-18,9.6192930369019622E-21,
        -0.0047740288164249351,-3.6535771780970351E-5,-0.0047740286550811339,-3.6535784842128748E-5,
        -2.0393520496314678E-18,-1.9132149024273884E-5,-1.4862170137645196E-18,2.4886181093055328E-21,
        -1.774286451758123E-18,-1.1737618337643748E-5,-2.8135328811439596E-18,-1.1737622416350756E-5,
        -0.0047740288164247026,-1.1737621816571777E-5,-0.00477402865512053,-3.8499651426988831E-21,
        -0.004774028816431854,7.7825837231677132E-21,-4.4847880380196558E-18,9.30286979541272E-21,
        -4.7408821129718168E-18,-1.1737594780950858E-5,-0.019100407554639352,5.29396286494622E-21,
        -2.7105015862681542E-18,9.6192930369019622E-21,-0.0047740288164249351,-1.4407159825200937E-21,
        -0.0084878806162880724,-1.9132145554703909E-5,-0.0047740288164157462,-3.6535784842128748E-5,
        -2.0393499890258091E-18,-1.9132149024273884E-5,-1.4862170137645196E-18,-1.17376252931991E-5,
        -1.4406120465869775E-18,-1.1737618337643748E-5,-2.8135328811439596E-18,4.4985054390960007E-21,
        -0.019100407554669848,-1.9132145554703909E-5,-0.0047740288164157462,-1.173761820526886E-5,
        -5.12953211008561E-19,-1.0192706915985939E-21,-4.0523201089203269E-18,9.4907989297949456E-21,
        -0.0047740286551203621,-1.1737594913325115E-5,-0.019100407554641059,-6.3132201495894354E-21,
        -4.0523201088961788E-18,-1.9132136410508959E-5,-0.0084878806162619943,2.2374863984518603E-21,
        -0.004774028816430049,-1.173761820526886E-5,-3.2234547972574721E-18,9.30286979541272E-21,
        -4.7408821129718168E-18,4.56750735693109E-21,-3.1326245098744425E-18,-3.6535774590606786E-5,
        -0.0047740288163857069,4.1968510873912379E-21,-0.0047740286551203621,-7.0416108400791964E-21,
        -0.004774028655127281,-1.9132150312873025E-5,-3.96943484008453E-18,7.6151018634488161E-21,
        -3.3522552392188485E-18,-1.9132144266105121E-5,-0.0047740286551111732,-1.1737624561044909E-5,
        -4.3730138752696916E-18,-6.3132233807637032E-21,-4.0523201089062622E-18,-1.1737621684196789E-5,
        -0.00477402865512013,-1.1737625160824026E-5,-1.8472759683862393E-18,-1.1737618337643748E-5,
        -2.8135328811439596E-18,-7.0416108400791964E-21,-0.004774028655127281,4.3253419633239867E-21,
        -0.0047740288164249351,6.487638936564484E-21,-0.0047740288164314507,-1.1314362810880367E-20,
        -4.2212656357647628E-19,1.0192679423238228E-20,-4.2885469058092407E-18,-3.8499602959374814E-21,
        -0.004774028816431854,8.47518431188035E-22,-3.5788545959929338E-18,-1.9132144266105121E-5,
        -0.0047740286551111732,-1.9132150312873025E-5,-3.9694322988795642E-18,-1.1737622548725761E-5,
        -0.0047740288164251033,-1.1737622548725761E-5,-0.0047740288164251033,-1.1737618337643748E-5,
        -2.8135328811439596E-18,1.1326233098153039E-20,-5.8265666453926312E-18,-1.1737617282081378E-5,
        -0.0084878806162790726,1.330429542412047E-21,-3.1548321734536232E-18,1.4439665438334856E-21,
        -0.0047740288164318505,3.0916537784894305E-21,-3.5609902498679662E-18,-1.1737621816571777E-5,
        -0.00477402865512053,5.2102265015382576E-21,-0.0047740286551254734,2.1771870320600187E-21,
        -2.1846348687197825E-19,-3.8499861453316237E-21,-0.0047740288164318505,-1.9132145554703909E-5,
        -0.0047740288164157462,-1.17376252931991E-5,-1.4406149314260643E-18,-1.17376252931991E-5,
        -4.1511156934352363E-18,-1.1737623950871349E-5,-4.6012459133564567E-18,-3.0564646751261151E-21,
        -0.004774028816430049,-1.1737625293199105E-5,-1.4406117719939627E-18,-1.1737624561044915E-5,
        -4.3730138752381371E-18,-1.173762381849631E-5,-5.0085045062929107E-18,-1.1737622548725761E-5,
        -0.0047740288164251033,0.019097634712978588,1.9705949370788169E-5,-4.8688115523384709E-18,
        1.9706037263565827E-5,0.019097634713069283,3.7095690051764795E-21,0.0084864283463426012,
        1.9706027944357129E-5,-4.8688115523384709E-18,1.9706037263565827E-5,0.019097634713069283,
        3.7095690051764795E-21,0.0084864283463426046,1.9706027944357129E-5,0.019097634713053105,
        1.0320169370790202E-5,-8.1421669077312929E-18,6.4597506714592294E-21,-6.2474553412857983E-18,
        1.970605510981498E-5,-8.1421669077312929E-18,6.4597506714592294E-21,-6.6664748607846E-18,
        1.0320206722311879E-5,0.019097634713086568,6.4665102880274361E-21,-5.4316653202643806E-18,
        6.4597377467621582E-21,0.00848642834638466,3.8826500860046649E-21,0.0047731377301323081,
        6.3319463279187473E-6,-8.1421669077312929E-18,6.4597506714592294E-21,-4.7954262503134087E-18,
        1.9706057794609424E-5,-6.6664748607846E-18,1.0320206722311879E-5,0.0084864283463932377,
        3.4546875165850422E-21,0.019097634713083383,7.0346282724865125E-21,0.004773137730106871,
        1.970604816668707E-5,0.0084864283463771065,1.0320202704323961E-5,0.019097634713074216,6.3319233139652047E-6,
        -5.229456703948615E-18,6.2450140997643232E-21,-4.9161993963896509E-18,5.288630945146067E-21,
        1.9351312724486906E-19,1.0320214271790599E-5,-5.7439423917783E-18,8.8634567521816331E-21,
        -6.7823735013844217E-18,6.3319438186664894E-6,0.019097634713072971,6.3319232425871977E-6,
        0.019097634713087813,3.3911044693435638E-21,0.0084864283463926687,4.94551254964995E-21,
        -1.2763973429718635E-18,5.0106974515346828E-21,0.0047731377301310383,5.2588556742684258E-21,
        0.0047731375688976167,6.3319458389590979E-6,0.0047731377301319855,6.3319462565397721E-6,
        -3.7659262455952018E-18,6.3319490718798243E-6,-6.69740196547176E-18,5.0107176463738564E-21,
        -6.3123784754145422E-18,5.3129552250339545E-21,0.0047731375688721779,1.9706046087283249E-5,
        -2.7105055694445983E-18,5.2939536887208516E-21,-6.7823735013844217E-18,6.3319438186664894E-6,
        -2.5169930097154123E-18,1.0320214271790599E-5,0.0084864283463869285,6.33194162909236E-6,
        0.019097634713087813,6.0380824295132524E-21,0.0084864283463926687,4.9455060873014142E-21,
        0.0047731377301359519,7.0201186844370227E-21,0.0047731377301310383,5.2588556742684258E-21,
        -4.7296674346768351E-18,1.9706059874013961E-5,0.0084864283463869251,6.3319416290923626E-6,
        0.0047731375688963469,7.35150791734108E-21,-5.1502136035375756E-18,5.8109876162706659E-21,
        -5.9539113998961089E-18,6.3319437472876285E-6,0.004773137730106871,1.970604816668707E-5,
        2.7078806088538766E-19,5.81095886920263E-21,0.0084864283463771048,1.0320202704323961E-5,
        -5.3183074545448137E-18,6.3319479727705775E-6,0.0047731375688963443,2.0575778463958446E-21,
        -6.3123784754145422E-18,5.3129552250339545E-21,-4.2663504849142025E-18,5.5967411830378648E-21,
        0.019097634713074216,6.3319233139652022E-6,-5.9539113998961089E-18,6.3319437472876285E-6,
        -2.3142137821508769E-19,6.3319490005007373E-6,0.0084864283463932377,6.1016590144061952E-21,
        -6.1526402695137655E-18,5.2412788940452409E-21,0.00848642834638636,6.3319415577135814E-6,
        0.0047731377301356267,7.9909056061474987E-21,-2.4397153806633983E-18,5.8109673616377915E-21,
        0.0047731375688972915,6.331945767580143E-6,0.0047731375689012579,5.7393022073196845E-21,
        0.0047731377301310383,2.6118841764472728E-21,-2.9419194635277004E-18,6.3319490005007373E-6,
        -4.0718719139017322E-18,6.3319438186664868E-6,-3.8473851895529522E-18,6.3319485829200054E-6,
        1.1546481405436232E-18,2.9497325267126323E-21,-5.7439423917783E-18,8.8634567521816331E-21,
        -6.4764298931487022E-18,6.3319490718798243E-6,-2.1305194015399455E-18,9.1307604902455708E-21,
        0.00848642834638636,6.3319415577135839E-6,0.0084864283463932343,6.1016784014518019E-21,
        0.0047731377301323107,6.3319463279187473E-6,0.0047731377301323081,6.3319463279187473E-6,
        0.0047731377301310383,5.2588605210298275E-21,-8.2146077167090343E-18,7.6481252722591485E-21,
        0.0047731377301266529,1.0320211280114997E-5,-3.2868157645701836E-18,6.3549205181106827E-21,
        -3.7659262455920463E-18,6.3319490718798243E-6,-6.0796869129044207E-18,4.3719641729370769E-21,
        0.0047731377301319855,6.33194625653977E-6,-1.7828764048777283E-18,6.3319479013915345E-6,
        -4.597720374387205E-18,6.6111019074067265E-22,-1.0554249332230198E-18,6.3319490718798217E-6,
        0.0084864283463869285,6.33194162909236E-6,0.0047731377301359519,4.37314718661587E-21,0.0047731377301359519,
        7.0201251467855583E-21,0.004773137730134761,3.3661662663447971E-21,1.0268951653126124E-19,
        6.3319479727705775E-6,0.0047731377301359493,4.3731633424872087E-21,0.0047731377301356267,
        5.3439324927392118E-21,0.004773137568900067,3.0421214925514163E-21,0.0047731377301323107,
        6.3319463279187448E-6,3.6535670676475959E-5,0.01910040755447192,-2.4094220280021159E-21,
        0.019100407554640066,3.6535758582015063E-5,9.1772683720778245E-19,1.9132097398897662E-5,
        0.019100407554600789,-2.4094220280021159E-21,0.019100407554640066,3.6535758582015063E-5,
        9.1772683720778245E-19,1.9132097398897662E-5,0.019100407554600789,3.6535754933752659E-5,
        0.0084878806162073227,-9.5894596048875008E-21,2.9635443265168115E-18,-5.073215019061359E-21,
        0.019100407554662031,-9.5894596048875008E-21,2.9635443265168115E-18,-1.2784690290117922E-20,
        0.0084878806162787812,3.6535782032491541E-5,2.2854837212386326E-18,-4.2954972221995882E-21,
        2.5304274024265693E-19,1.9132138159811332E-5,2.6799900119830713E-18,1.1737622548725761E-5,
        0.0047740288164251033,-9.5894596048875008E-21,2.9635443265168115E-18,-8.5218860891597851E-21,
        0.019100407554668141,-1.2784690290117922E-20,0.0084878806162787812,1.9132150312873025E-5,
        3.9694314746272033E-18,3.6535779834867094E-5,2.529287210793528E-18,1.1737594913325115E-5,
        0.019100407554641059,1.9132136410508959E-5,0.0084878806162619943,3.6535774590606786E-5,
        0.0047740288163857069,-4.09262794579669E-21,4.4611413024616849E-18,-1.0138752364165677E-20,
        4.5119467335133523E-18,1.4407159825200937E-21,0.0084878806162880724,-1.0192679423238228E-20,
        4.2885469058092407E-18,-9.6192930369019622E-21,0.0047740288164249351,3.6535771780970351E-5,
        0.0047740286550811339,3.6535784842128748E-5,2.0393520496314678E-18,1.9132149024273884E-5,
        1.4862170137645196E-18,-2.4886181093055328E-21,1.774286451758123E-18,1.1737618337643748E-5,
        2.8135328811439596E-18,1.1737622416350756E-5,0.0047740288164247026,1.1737621816571777E-5,
        0.00477402865512053,3.8499651426988831E-21,0.004774028816431854,-7.7825837231677132E-21,
        4.4847880380196558E-18,-9.30286979541272E-21,4.7408821129718168E-18,1.1737594780950858E-5,
        0.019100407554639352,-5.29396286494622E-21,2.7105015862681542E-18,-9.6192930369019622E-21,
        0.0047740288164249351,1.4407159825200937E-21,0.0084878806162880724,1.9132145554703909E-5,
        0.0047740288164157462,3.6535784842128748E-5,2.0393499890258091E-18,1.9132149024273884E-5,
        1.4862170137645196E-18,1.17376252931991E-5,1.4406120465869775E-18,1.1737618337643748E-5,
        2.8135328811439596E-18,-4.4985054390960007E-21,0.019100407554669848,1.9132145554703909E-5,
        0.0047740288164157462,1.173761820526886E-5,5.12953211008561E-19,1.0192706915985939E-21,
        4.0523201089203269E-18,-9.4907989297949456E-21,0.0047740286551203621,1.1737594913325115E-5,
        0.019100407554641059,6.3132201495894354E-21,4.0523201088961788E-18,1.9132136410508959E-5,
        0.0084878806162619943,-2.2374863984518603E-21,0.004774028816430049,1.173761820526886E-5,
        3.2234547972574721E-18,-9.30286979541272E-21,4.7408821129718168E-18,-4.56750735693109E-21,
        3.1326245098744425E-18,3.6535774590606786E-5,0.0047740288163857069,-4.1968510873912379E-21,
        0.0047740286551203621,7.0416108400791964E-21,0.004774028655127281,1.9132150312873025E-5,
        3.96943484008453E-18,-7.6151018634488161E-21,3.3522552392188485E-18,1.9132144266105121E-5,
        0.0047740286551111732,1.1737624561044909E-5,4.3730138752696916E-18,6.3132233807637032E-21,
        4.0523201089062622E-18,1.1737621684196789E-5,0.00477402865512013,1.1737625160824026E-5,
        1.8472759683862393E-18,1.1737618337643748E-5,2.8135328811439596E-18,7.0416108400791964E-21,
        0.004774028655127281,-4.3253419633239867E-21,0.0047740288164249351,-6.487638936564484E-21,
        0.0047740288164314507,1.1314362810880367E-20,4.2212656357647628E-19,-1.0192679423238228E-20,
        4.2885469058092407E-18,3.8499602959374814E-21,0.004774028816431854,-8.47518431188035E-22,
        3.5788545959929338E-18,1.9132144266105121E-5,0.0047740286551111732,1.9132150312873025E-5,
        3.9694322988795642E-18,1.1737622548725761E-5,0.0047740288164251033,1.1737622548725761E-5,
        0.0047740288164251033,1.1737618337643748E-5,2.8135328811439596E-18,-1.1326233098153039E-20,
        5.8265666453926312E-18,1.1737617282081378E-5,0.0084878806162790726,-1.330429542412047E-21,
        3.1548321734536232E-18,-1.4439665438334856E-21,0.0047740288164318505,-3.0916537784894305E-21,
        3.5609902498679662E-18,1.1737621816571777E-5,0.00477402865512053,-5.2102265015382576E-21,
        0.0047740286551254734,-2.1771870320600187E-21,2.1846348687197825E-19,3.8499861453316237E-21,
        0.0047740288164318505,1.9132145554703909E-5,0.0047740288164157462,1.17376252931991E-5,
        1.4406149314260643E-18,1.17376252931991E-5,4.1511156934352363E-18,1.1737623950871349E-5,
        4.6012459133564567E-18,3.0564646751261151E-21,0.004774028816430049,1.1737625293199105E-5,
        1.4406117719939627E-18,1.1737624561044915E-5,4.3730138752381371E-18,1.173762381849631E-5,
        5.0085045062929107E-18,1.1737622548725761E-5,0.0047740288164251033,-1.4180920718254179E-6,
        -4.6022795145665838E-9,-0.99999999999999989,-8.2718061255302767E-25,-1.418092071846599E-6,
        -1.0766988945962442E-24,-0.3333335808704333,-2.1340306865294098E-9,-0.99999999999999989,
        -8.2718061255302767E-25,-1.418092071846599E-6,-1.0766988945962442E-24,-0.3333335808704333,
        -2.1340306865294098E-9,-1.4180920718464292E-6,-1.955816480370227E-9,-0.99999999999999989,
        -2.481541837659083E-24,-0.99999999999999989,-8.2718061255302767E-25,-0.99999999999999989,
        -2.481541837659083E-24,-0.99999999999999989,-8.2718061255302767E-25,-1.4180920718526257E-6,
        -2.1093793506811558E-24,-0.99999999999999989,-1.6543612251060553E-24,-0.33333358087043324,
        -1.2407709188295415E-24,-0.50000007594345175,-2.874378256066275E-10,-0.99999999999999989,
        -2.481541837659083E-24,-0.99999999999999989,-8.2718061255302767E-25,-0.99999999999999989,
        -8.2718061255302767E-25,-0.3333335808704333,-8.2718061255302767E-25,-1.4180920718521672E-6,
        -2.0803445362035913E-24,-0.50000007594345175,-1.2263762091205498E-9,-0.3333335808704333,
        -9.0870284252294989E-10,-1.4180920718510982E-6,-1.0736760082907264E-9,-0.99999999999999989,
        -2.481541837659083E-24,-0.99999999999999989,-2.481541837659083E-24,-0.99999999999999989,0.0,
        -0.99999999999999989,-2.481541837659083E-24,-0.99999999999999989,-1.6543612251060553E-24,
        -1.41809207185032E-6,-1.0736759636101028E-9,-1.4180920718534039E-6,-1.9064101729332208E-24,
        -0.33333358087043324,-1.2407709188295415E-24,-0.99999999999999989,-1.6543612251060553E-24,
        -0.50000007594345175,-4.1359030627651384E-25,-0.5000000759434492,-2.8743781783328083E-10,
        -0.50000007594345175,-2.874378139634491E-10,-0.99999999999999989,-8.2718061255302767E-25,
        -0.99999999999999989,-1.6543612251060553E-24,-0.99999999999999989,-2.481541837659083E-24,
        -0.50000007594344908,-1.22637617606276E-9,-0.99999999999999989,-8.2718061255302767E-25,-0.99999999999999989,
        -1.6543612251060553E-24,-0.99999999999999989,0.0,-0.3333335808704333,-4.9833888491491584E-10,
        -1.4180920718534039E-6,-1.2601768970979784E-24,-0.33333358087043324,-1.2407709188295415E-24,
        -0.50000007594345175,-1.2407709188295415E-24,-0.50000007594345175,-4.1359030627651384E-25,
        -0.99999999999999989,0.0,-0.3333335808704333,-4.9833888491491584E-10,-0.5000000759434492,
        -8.2718061255302767E-25,-0.99999999999999989,-8.2718061255302767E-25,-0.99999999999999989,
        -1.6543612251060553E-24,-0.50000007594345175,-1.2263762091205498E-9,-0.99999999999999989,
        -8.2718061255302767E-25,-0.3333335808704333,-9.0870284252294989E-10,-0.99999999999999989,
        -1.6543612251060553E-24,-0.5000000759434492,-8.2718061255302767E-25,-0.99999999999999989,
        -2.481541837659083E-24,-0.99999999999999989,-1.6543612251060553E-24,-1.4180920718510982E-6,
        -1.0736760082907264E-9,-0.99999999999999989,-1.6543612251060553E-24,-0.99999999999999989,
        -8.2718061255302767E-25,-0.3333335808704333,-1.2407709188295415E-24,-0.99999999999999989,
        -1.6543612251060553E-24,-0.33333358087043324,-4.9833886442279871E-10,-0.50000007594345175,0.0,
        -0.99999999999999989,-8.2718061255302767E-25,-0.5000000759434492,-2.8743780619010325E-10,
        -0.5000000759434492,-8.2718061255302767E-25,-0.50000007594345175,-4.1359030627651384E-25,
        -0.99999999999999989,-8.2718061255302767E-25,-0.99999999999999989,-1.6543612251060553E-24,
        -0.99999999999999989,-1.6543612251060553E-24,-0.99999999999999989,-1.6543612251060553E-24,
        -0.99999999999999989,-2.481541837659083E-24,-0.99999999999999989,-8.2718061255302767E-25,
        -0.99999999999999989,-1.6543612251060553E-24,-0.33333358087043324,-4.9833886442279871E-10,
        -0.3333335808704333,-1.2407709188295415E-24,-0.50000007594345175,-2.874378256066275E-10,
        -0.50000007594345175,-2.874378256066275E-10,-0.50000007594345175,-4.1359030627651384E-25,
        -0.99999999999999989,-2.481541837659083E-24,-0.50000007594345175,-5.23788979844978E-10,-0.99999999999999989,
        -8.2718061255302767E-25,-0.99999999999999989,-8.2718061255302767E-25,-0.99999999999999989,
        -2.481541837659083E-24,-0.50000007594345175,-2.8743781396344868E-10,-0.99999999999999989,
        -1.6543612251060553E-24,-0.99999999999999989,-8.2718061255302767E-25,-0.99999999999999989,
        -8.2718061255302767E-25,-0.3333335808704333,-4.9833888491491584E-10,-0.50000007594345175,
        -4.1359030627651384E-25,-0.50000007594345175,-1.2407709188295415E-24,-0.50000007594345175,
        -8.2718061255302767E-25,-0.99999999999999989,-1.6543612251060553E-24,-0.50000007594345175,
        -1.2407709188295415E-24,-0.50000007594345175,0.0,-0.5000000759434492,-8.2718061255302767E-25,
        -0.50000007594345175,-2.8743782560662668E-10,-4.602279514566583E-9,-1.4185411752855009E-6,
        1.1021570137295366E-24,-1.4185411753066819E-6,0.0,-1.0,-2.1340306865294098E-9,-1.4185411753037778E-6,
        1.1021570137295366E-24,-1.4185411753066819E-6,0.0,-1.0,-2.1340306865294098E-9,-1.4185411753037778E-6,
        -1.955816480370227E-9,-0.33333358095885846,8.2718061255302767E-25,-1.0,1.6676850857952382E-24,
        -1.4185411753106089E-6,8.2718061255302767E-25,-1.0,8.2718061255302767E-25,-0.33333358095885846,0.0,-1.0,
        8.2718061255302767E-25,-1.0,0.0,-1.0,-2.8743782560662585E-10,-0.50000007597137852,8.2718061255302767E-25,
        -1.0,1.0500275073907217E-24,-1.4185411753113024E-6,8.2718061255302767E-25,-0.33333358095885846,
        -8.2718061255302767E-25,-0.99999999999999978,0.0,-1.0,-1.22637620912055E-9,-1.4185411753087207E-6,
        -9.087028425229503E-10,-0.33333358095885846,-1.0736760082907253E-9,-0.50000007597137863,
        8.2718061255302767E-25,-1.0,8.2718061255302767E-25,-1.0,4.1359030627651384E-25,-0.33333358095885846,
        8.2718061255302767E-25,-1.0,8.2718061255302767E-25,-0.50000007597137863,-1.0736759636101013E-9,
        -0.500000075971376,0.0,-1.0,0.0,-1.0,8.2718061255302767E-25,-1.0,8.2718061255302767E-25,-1.0,
        -2.8743781783327917E-10,-0.50000007597137863,-2.8743781396344744E-10,-0.500000075971376,
        8.2718061255302767E-25,-0.50000007597137852,8.2718061255302767E-25,-1.0,1.6543612251060553E-24,-1.0,
        -1.2263761760627599E-9,-1.4185411753082944E-6,0.0,-0.99999999999999978,8.2718061255302767E-25,
        -0.50000007597137863,4.1359030627651384E-25,-0.33333358095885846,-4.9833888491491543E-10,
        -0.50000007597137852,0.0,-1.0,0.0,-1.0,0.0,-0.99999999999999978,8.2718061255302767E-25,-1.0,
        1.0851507503347821E-24,-1.4185411753117287E-6,-4.9833888491491584E-10,-0.50000007597137852,
        8.2718061255302767E-25,-1.0,8.2718061255302767E-25,-1.0,8.2718061255302767E-25,-0.50000007597137608,
        -1.22637620912055E-9,-1.4185411753087207E-6,8.2718061255302767E-25,-1.0,-9.087028425229503E-10,
        -0.33333358095885846,8.2718061255302767E-25,-0.50000007597137852,0.0,-1.0,1.6543612251060553E-24,-1.0,0.0,
        -0.99999999999999978,-1.0736760082907253E-9,-0.50000007597137863,1.2407709188295415E-24,
        -0.50000007597137608,8.2718061255302767E-25,-0.500000075971376,-8.2718061255302767E-25,-0.99999999999999978,
        8.2718061255302767E-25,-1.0,-4.9833886442279747E-10,-0.50000007597137608,0.0,-0.99999999999999978,
        1.6543612251060553E-24,-1.0,-2.8743780619010118E-10,-0.50000007597137608,8.2718061255302767E-25,-1.0,0.0,
        -1.0,8.2718061255302767E-25,-0.500000075971376,1.6543612251060553E-24,-0.50000007597137863,
        1.2407709188295415E-24,-0.50000007597137863,8.2718061255302767E-25,-0.99999999999999978,
        8.2718061255302767E-25,-1.0,8.2718061255302767E-25,-0.50000007597137852,0.0,-1.0,-4.9833886442279747E-10,
        -0.50000007597137608,-8.2718061255302767E-25,-0.99999999999999978,-2.8743782560662585E-10,
        -0.50000007597137852,-2.8743782560662585E-10,-0.50000007597137852,8.2718061255302767E-25,-1.0,
        8.2718061255302767E-25,-1.0,-5.2378897984497882E-10,-0.33333358095885846,8.2718061255302767E-25,-1.0,
        8.2718061255302767E-25,-0.50000007597137852,1.6543612251060553E-24,-1.0,-2.8743781396344744E-10,
        -0.500000075971376,8.2718061255302767E-25,-0.50000007597137608,1.6543612251060553E-24,-0.99999999999999978,
        8.2718061255302767E-25,-0.50000007597137852,-4.9833888491491543E-10,-0.50000007597137852,0.0,
        -0.99999999999999978,0.0,-0.99999999999999978,0.0,-0.99999999999999978,8.2718061255302767E-25,
        -0.50000007597137852,-8.2718061255302767E-25,-0.99999999999999978,0.0,-0.99999999999999978,
        8.2718061255302767E-25,-1.0,-2.8743782560662585E-10,-0.50000007597137852;
END_VAR
VAR_TEMP
    new_x: ARRAY [0..5] OF LREAL;
    y_innov: ARRAY [0..1] OF LREAL;
    th: ARRAY [0..9] OF LREAL;
    b_k: DINT;
    du: ARRAY [0..1] OF LREAL;
    found: BOOL;
    regionmin: DINT;
    betamin: LREAL;
    beta: LREAL;
    betah: LREAL;
    b_h: DINT;
    rtb_xest: ARRAY [0..5] OF LREAL;
    i: DINT;
END_VAR
CASE ssMethodType OF
    SS_INITIALIZE:
        (* SystemInitialize for Atomic SubSystem: '<Root>/Explicit Controller' *)
        (* InitializeConditions for Memory: '<S3>/last_x' *)
        FOR i := 0 TO 5 DO
            last_x_PreviousInput[i] := 0.0;
        END_FOR;
        (* End of InitializeConditions for Memory: '<S3>/last_x' *)
